// TIA Portal project "#08-法格800T(增加润滑参数设置与监控）" (V17)

(* hardware
DEVICE "S7-1200 station_1"  S7-1200 Station
   slot 0: "Rack_0"  S7-1200 Rack  Rack  V1.0
   slot 1: "PLC_1"  CPU 1215C DC/DC/DC  6ES7 215-1AG40-0XB0  V4.5
   slot 2: "DI 16x24VDC_1"  6ES7 221-1BH32-0XB0  V2.0
   slot 3: "DI 16x24VDC_2"  6ES7 221-1BH32-0XB0  V2.0
   slot 4: "DI 16x24VDC_3"  6ES7 221-1BH32-0XB0  V2.0
   slot 5: "DQ 16x24VDC_1"  SM 1222 DQ16 x 24VDC  6ES7 222-1BH32-0XB0  V2.0
   slot 101: "CM 1243-5"  CM 1243-5  6GK7 243-5DX30-0XE0  V1.3
DEVICE "ET 200SP station_1"  ET 200SP-Station
   slot 0: "机架_0"  Rack  6ES5 710-8MAx1
   slot 0: "IO device_1"  IM 155-6 PN ST  6ES7 155-6AU01-0BN0  V4.2
   slot 1: "DI 16x24VDC ST_1"  DI 16x24VDC ST  6ES7 131-6BH01-0BA0  V0.0
      slot 1: "DI 16x24VDC ST_1"  DI 16x24VDC ST
   slot 2: "DI 16x24VDC ST_6"  DI 16x24VDC ST  6ES7 131-6BH01-0BA0  V0.0
      slot 1: "DI 16x24VDC ST_6"  DI 16x24VDC ST
   slot 3: "DI 16x24VDC ST_5"  DI 16x24VDC ST  6ES7 131-6BH01-0BA0  V0.0
      slot 1: "DI 16x24VDC ST_5"  DI 16x24VDC ST
   slot 4: "DI 16x24VDC ST_4"  DI 16x24VDC ST  6ES7 131-6BH01-0BA0  V0.0
      slot 1: "DI 16x24VDC ST_4"  DI 16x24VDC ST
   slot 5: "DI 16x24VDC ST_3"  DI 16x24VDC ST  6ES7 131-6BH01-0BA0  V0.0
      slot 1: "DI 16x24VDC ST_3"  DI 16x24VDC ST
   slot 6: "DI 16x24VDC ST_2"  DI 16x24VDC ST  6ES7 131-6BH01-0BA0  V0.0
      slot 1: "DI 16x24VDC ST_2"  DI 16x24VDC ST
   slot 7: "DI 16x24VDC ST_7"  DI 16x24VDC ST  6ES7 131-6BH01-0BA0  V0.0
      slot 1: "DI 16x24VDC ST_7"  DI 16x24VDC ST
   slot 8: "DI 16x24VDC ST_9"  DI 16x24VDC ST  6ES7 131-6BH01-0BA0  V0.0
      slot 1: "DI 16x24VDC ST_9"  DI 16x24VDC ST
   slot 9: "DI 16x24VDC ST_8"  DI 16x24VDC ST  6ES7 131-6BH01-0BA0  V0.0
      slot 1: "DI 16x24VDC ST_8"  DI 16x24VDC ST
   slot 10: "DQ 16x24VDC/0.5A ST_2"  DQ 16x24VDC/0.5A ST  6ES7 132-6BH01-0BA0  V0.0
      slot 1: "DQ 16x24VDC/0.5A ST_2"  DQ 16x24VDC/0.5A ST
   slot 11: "DQ 16x24VDC/0.5A ST_1"  DQ 16x24VDC/0.5A ST  6ES7 132-6BH01-0BA0  V0.0
      slot 1: "DQ 16x24VDC/0.5A ST_1"  DQ 16x24VDC/0.5A ST
   slot 12: "服务器模块_1"  Server module  6ES7 193-6PA00-0AA0  V1.1
      slot 1: "服务器模块_1"  Server module
   slot 127: "BA 2xRJ45"  BA 2xRJ45  6ES7 193-6AR00-0AA0  V0.0
      slot 1: "Port_1"  X1 P1 R  6ES7 193-6AR00-0AA0  V0.0
      slot 2: "Port_2"  X1 P2 R  6ES7 193-6AR00-0AA0  V0.0
DEVICE "HMI_1"  TP900 Comfort
   slot 0: "HMI_1"  TP900 Comfort  6AV2 124-0JC01-0AX0  15.1.0.0
   slot 1: "HMI_RT_1"  TP900 Comfort  6AV2 124-0JC01-0AX0  15.1.0.0
   slot 5: "HMI_1.IE_CP_1"  PROFINET Interface  15.0.1.0
      slot 1: "PROFINET Interface_1"  PROFINET Interface
         slot 1: "Port_1"  Port
         slot 2: "Port_2"  Port
   slot 7: "HMI_1.MPI/DP_CP_1"  MPI/DP Interface  15.0.1.0
DEVICE "GSD device_2"  GSD.Device
   slot 0: "机架_0"  Rail
   slot 0: "横梁站"  P+F  Encoder  4.0
DEVICE "GSD device_1"  GSD.Device
   slot 0: "机架_0"  Rail
   slot 0: "滑块站"  P+F  Encoder  4.0
DEVICE "GSD device_3"  GSD.Device
   slot 0: "机架_0"  Rail
   slot 0: "气垫编码器"  P+F  Encoder  4.0
*)

// ===== PLC "PLC_1"  CPU 1215C DC/DC/DC =====

VAR_GLOBAL   // PLC tag table "默认变量表"
   "Tag_47(1)" AT %I6.1 : Bool;
   "Tag_48(1)" AT %I6.2 : Bool;
   "Tag_49(1)" AT %I6.3 : Bool;
   "Tag_50(1)" AT %I6.4 : Bool;
   "Tag_51(1)" AT %I6.5 : Bool;
   "Tag_52(1)" AT %I6.6 : Bool;
   "Tag_53(1)" AT %I6.7 : Bool;
   "Tag_54(1)" AT %I7.0 : Bool;
   "Tag_55(1)" AT %I7.1 : Bool;
   "Tag_56(1)" AT %I7.2 : Bool;
   "Tag_57(1)" AT %I7.3 : Bool;
   "Tag_58(1)" AT %I7.4 : Bool;
   "Tag_59" AT %I7.5 : Bool;
   "Tag_60" AT %I7.6 : Bool;
   "Tag_61(1)" AT %I7.7 : Bool;
   "左栅栏落下来检测" AT %Q13.1 : Bool;
   "备用(16)" AT %Q13.2 : Bool;
   "双阀控制1" AT %Q13.3 : Bool;
   "Tag_155" AT %Q13.4 : Bool;
   "双阀控制2" AT %Q13.5 : Bool;
   "Tag_157" AT %Q13.6 : Bool;
   "Tag_158" AT %Q13.7 : Bool;
   "过滤器堵塞" AT %M5.0 : Bool;
   "润滑油压正常" AT %M5.1 : Bool;
   "滑块调整允许" AT %M5.2 : Bool;
   "急停故障" AT %M6.0 : Bool;
   "液压保护故障" AT %M6.1 : Bool;
   "气压故障" AT %M6.2 : Bool;
   "设备故障" AT %M6.3 : Bool;
   "滑块调整允许(1)" AT %M6.4 : Bool;
   "滑块调整允许2(1)" AT %M6.5 : Bool;
   "气垫调整允许" AT %M6.6 : Bool;
   "工作台移动允许" AT %M7.0 : Bool;
   "工作台落到位" AT %M7.1 : Bool;
   "润滑油泵启动OK" AT %M5.5 : Bool;
   "10度" AT %M200.0 : Bool;
   "20度" AT %M200.1 : Bool;
   "30度" AT %M200.2 : Bool;
   "40度" AT %M200.3 : Bool;
   "50" AT %M200.4 : Bool;
   "60" AT %M200.5 : Bool;
   "70" AT %M200.6 : Bool;
   "80" AT %M200.7 : Bool;
   "90" AT %M201.0 : Bool;
   "100" AT %M201.1 : Bool;
   "110" AT %M201.2 : Bool;
   "120" AT %M201.3 : Bool;
   "130" AT %M201.4 : Bool;
   "140" AT %M201.5 : Bool;
   "150" AT %M201.6 : Bool;
   "160" AT %M201.7 : Bool;
   "170" AT %M202.0 : Bool;
   "180" AT %M202.1 : Bool;
   "190" AT %M202.2 : Bool;
   "200" AT %M202.3 : Bool;
   "210" AT %M202.4 : Bool;
   "220" AT %M202.5 : Bool;
   "230" AT %M202.6 : Bool;
   "240" AT %M202.7 : Bool;
   "250" AT %M203.0 : Bool;
   "260" AT %M203.1 : Bool;
   "270" AT %M203.2 : Bool;
   "280" AT %M203.3 : Bool;
   "290" AT %M203.4 : Bool;
   "300" AT %M203.5 : Bool;
   "310" AT %M203.6 : Bool;
   "320" AT %M203.7 : Bool;
   "330" AT %M204.0 : Bool;
   "340" AT %M204.1 : Bool;
   "350" AT %M204.2 : Bool;
   "360" AT %M204.3 : Bool;
   "上死点" AT %M204.4 : Bool;
   "制动监控" AT %M204.5 : Bool;
   "下死点" AT %M204.6 : Bool;
   "单次返回" AT %M204.7 : Bool;
   "光电保护位置" AT %M205.0 : Bool;
   "横梁编码器" AT %ID68 : DWord;
   "急停故障(1)" AT %M10.0 : Bool;
   "行程允许" AT %M14.0 : Bool;
   "寸动允许" AT %M14.1 : Bool;
   "寸动开始" AT %M14.2 : Bool;
   "单次允许" AT %M14.3 : Bool;
   "单次开始" AT %M14.4 : Bool;
   "双手按钮开点" AT %M14.5 : Bool;
   "双手按钮闭点" AT %M14.6 : Bool;
   "编码器闭点监控" AT %M14.7 : Bool;
   "编码器开点监控" AT %M15.0 : Bool;
   "编码器故障" AT %M15.1 : Bool;
   "工作台-夹紧OK" AT %M15.2 : Bool;
   "工作台放松OK" AT %M15.3 : Bool;
   "润滑故障" AT %M15.4 : Bool;
   "滑块软限位上" AT %M15.5 : Bool;
   "滑块软限位下" AT %M15.6 : Bool;
   "滑块调整自动向上" AT %M16.0 : Bool;
   "滑块调整自动向下" AT %M16.1 : Bool;
   "滑块调整自动选择" AT %M16.2 : Bool;
   "滑块手动调整" AT %M16.3 : Bool;
   "ECamdata _DB_D{10}滑块设定高度" AT %MD150 : Real;
   "备用(27)" AT %I21.4 : Bool;
   "备用(7)" AT %I21.3 : Bool;
   "润滑过滤检测" AT %I21.2 : Bool;
   "润滑油位检测" AT %I21.1 : Bool;
   "润滑故障复位" AT %I21.0 : Bool;
   "气垫手动润滑" AT %I20.7 : Bool;
   "平衡缸手动润滑" AT %I20.6 : Bool;   // OK
   "润滑启动按钮(1)" AT %I20.5 : Bool;   // OK
   "润滑停止按钮" AT %I20.4 : Bool;   // OK
   "备用(6)" AT %I20.3 : Bool;
   "气垫上调整(1)" AT %I20.2 : Bool;
   "滑块夹紧压力检测" AT %I20.1 : Bool;
   "后右夹紧器检测" AT %I20.0 : Bool;
   "备用(28)" AT %I21.5 : Bool;
   "后中夹紧器检测" AT %I19.7 : Bool;
   "前左夹紧器检测" AT %I19.5 : Bool;
   "前中夹紧器检测" AT %I19.4 : Bool;
   "前右夹紧器检测" AT %I19.3 : Bool;
   "气垫下降调整" AT %I19.2 : Bool;
   "滑块松开压力检测" AT %I19.1 : Bool;
   "150/AR液压保护压力" AT %I19.0 : Bool;
   "90/AR液压保护压力" AT %I18.7 : Bool;
   "100液压保护压力" AT %I18.6 : Bool;
   "135/AR液压保护压力" AT %I18.5 : Bool;
   "100/AR液压保护压力" AT %I18.4 : Bool;
   "液压保护选择开关1位" AT %I18.3 : Bool;   // OK
   "液压保护选择开关0位" AT %I18.2 : Bool;   // OK
   "工作台落下右边后检测" AT %I18.1 : Bool;
   "后左夹紧器检测" AT %I19.6 : Bool;
   "工作台落下左后检测" AT %I18.0 : Bool;
   "备用(8)" AT %I21.6 : Bool;
   "备用(10)" AT %I22.0 : Bool;
   "寸动" AT %I25.4 : Bool;   // OK
   "反转" AT %I25.3 : Bool;   // OK
   "右前双手选择" AT %I25.2 : Bool;   // OK
   "右后双手选择(1)" AT %I25.1 : Bool;   // OK
   "左后双手选择" AT %I25.0 : Bool;   // OK
   "单人/双人选择" AT %I24.7 : Bool;
   "离制油箱油温检测" AT %I24.6 : Bool;
   "左前双手选择" AT %I24.5 : Bool;   // OK
   "备用(15)" AT %I24.4 : Bool;
   "离合冷却过滤器检测" AT %I24.3 : Bool;
   "离制油箱油位检测" AT %I24.2 : Bool;
   "备用(14)" AT %I24.1 : Bool;
   "离制压力检测" AT %I24.0 : Bool;
   "备用(9)" AT %I21.7 : Bool;
   "离制过滤器检测" AT %I23.7 : Bool;
   "栅栏门向上？(1)" AT %I23.5 : Bool;
   "栅栏门向上？" AT %I23.4 : Bool;
   "备用(13)" AT %I23.3 : Bool;
   "备用(12)" AT %I23.2 : Bool;
   "前安全栓" AT %I23.1 : Bool;   // OK
   "后安全栓" AT %I23.0 : Bool;   // OK
   "左后急停按钮" AT %I22.7 : Bool;   // OK
   "右后急停按钮" AT %I22.6 : Bool;   // OK
   "左前急停按钮" AT %I22.5 : Bool;   // OK
   "右前急停按钮" AT %I22.4 : Bool;   // OK
   "备用(11)" AT %I22.3 : Bool;
   "气垫分油器检测" AT %I22.2 : Bool;
   "滑块分油器检测" AT %I22.1 : Bool;
   "备用(29)" AT %I23.6 : Bool;
   "工作台落下右前检测" AT %I17.7 : Bool;
   "工作台落下左前检测" AT %I17.6 : Bool;
   "工作台顶起右后检测" AT %I17.5 : Bool;
   "气垫冷却电机温度监测(启动）" AT %I13.3 : Bool;
   "气垫冷却电机温度监测(停止）" AT %I13.2 : Bool;
   "气垫冷却电机过热" AT %I13.1 : Bool;
   "主电机启动(1)" AT %I13.0 : Bool;   // OK
   "主电机停止" AT %I12.7 : Bool;   // OK
   "备用(26)" AT %I12.6 : Bool;
   "备用(25)" AT %I12.5 : Bool;
   "备用(24)" AT %I12.4 : Bool;
   "IMCO应力机" AT %I12.3 : Bool;
   "滑块调整传动检测？(1)" AT %I12.2 : Bool;
   "气垫压力检测" AT %I12.1 : Bool;
   "气垫排气" AT %I12.0 : Bool;
   "气垫油位检测" AT %I11.7 : Bool;
   "上极限" AT %I13.4 : Bool;
   "气垫左落下到位" AT %I11.6 : Bool;
   "备用" AT %I11.4 : Bool;
   "气垫调整下极限" AT %I11.3 : Bool;
   "气垫调整上极限" AT %I11.2 : Bool;
   "右气垫选择" AT %I11.1 : Bool;
   "气垫排气(1)" AT %I11.0 : Bool;
   "气垫选择开关" AT %I10.7 : Bool;
   "滑块调整传动检测？" AT %I10.6 : Bool;
   "平衡缸气压检测" AT %I10.5 : Bool;
   "滑块调整下极限" AT %I10.4 : Bool;
   "滑块调整上极限" AT %I10.3 : Bool;
   "滑块调整向下" AT %I10.2 : Bool;   // OK
   "滑块调整向上" AT %I10.1 : Bool;   // OK
   "滑块调整选择开关" AT %I10.0 : Bool;   // OK
   "备用(1)" AT %I11.5 : Bool;
   "下极限" AT %I13.5 : Bool;
   "出到位检测（小车）" AT %I13.6 : Bool;
   "移动工作台变速（小车）" AT %I13.7 : Bool;
   "工作台顶起左后检测" AT %I17.4 : Bool;
   "工作台顶起右前检测" AT %I17.3 : Bool;
   "工作台顶起左前检测" AT %I17.2 : Bool;
   "气垫上调整" AT %I17.1 : Bool;
   "外导轨切换检测？(1)" AT %I17.0 : Bool;
   "外导轨切换检测？" AT %I16.7 : Bool;
   "工作台右后落到位" AT %I16.6 : Bool;
   "工作台左后落到为" AT %I16.5 : Bool;
   "工作台右前落到为" AT %I16.4 : Bool;
   "工作台左前落到为" AT %I16.3 : Bool;
   "工作台开进到位" AT %I16.2 : Bool;
   "工作台右后顶起到位" AT %I16.1 : Bool;
   "工作台左后顶起到位" AT %I16.0 : Bool;
   "工作台右前顶起到位" AT %I15.7 : Bool;
   "工作台左前顶起到位" AT %I15.6 : Bool;
   "按钮站插入" AT %I15.5 : Bool;
   "左工作台按钮拔出" AT %I15.4 : Bool;
   "工作台顶起压力" AT %I15.3 : Bool;
   "备用(2)" AT %I15.2 : Bool;
   "循环停止" AT %I15.1 : Bool;   // OK
   "工作台开进" AT %I15.0 : Bool;   // OK
   "工作台开出" AT %I14.7 : Bool;   // OK
   "模具更换自动/手动选择" AT %I14.6 : Bool;   // OK
   "调整开关" AT %I14.5 : Bool;   // OK
   "工作台放松顶起" AT %I14.4 : Bool;   // OK
   "工作台落下夹紧(1)" AT %I14.3 : Bool;   // OK
   "备用(4)" AT %I14.2 : Bool;
   "备用(3)" AT %I14.1 : Bool;
   "工作台停止" AT %I14.0 : Bool;
   "单次" AT %I25.5 : Bool;   // OK
   "连续" AT %I25.6 : Bool;   // OK
   "备用(17)" AT %I25.7 : Bool;
   "左前双手 使用" AT %I26.0 : Bool;
   "模具移出指示" AT %Q12.2 : Bool;
   "飞轮停止指示灯" AT %Q12.1 : Bool;
   "主电机启动指示" AT %Q12.0 : Bool;
   "自动化气压" AT %Q11.7 : Bool;
   "气垫间歇润滑阀" AT %Q11.6 : Bool;
   "备用(35)" AT %Q11.5 : Bool;
   "工作台顶起" AT %Q11.4 : Bool;
   "工作台落下夹紧(2)" AT %Q11.3 : Bool;
   "工作台落下夹紧" AT %Q11.2 : Bool;
   "工作台放松顶起(1)" AT %Q11.1 : Bool;
   "液压保护负荷荷 阀-3#" AT %Q11.0 : Bool;
   "液压保护泵启动（卸载）阀-2#" AT %Q10.7 : Bool;
   "气动泵气源阀-1#" AT %Q10.6 : Bool;
   "模具装入指示" AT %Q12.3 : Bool;
   "右气垫气排阀" AT %Q10.5 : Bool;
   "气垫排气阀" AT %Q10.3 : Bool;
   "气垫进气阀" AT %Q10.2 : Bool;
   "平衡缸排气阀" AT %Q10.1 : Bool;
   "平衡缸进气阀" AT %Q10.0 : Bool;
   "Tag_109" AT %QW572 : Int;
   "Tag_108" AT %QW570 : Int;
   "Tag_20" AT %ID97 : DWord;
   "气垫编码器" AT %ID100 : DWord;
   "气垫编码器1" AT %ID96 : DWord;
   "气垫模拟量1" AT %IW82 : Int;
   "平衡器压力模拟量" AT %IW80 : Int;
   "气垫模拟量2" AT %IW84 : Int;
   "滑块编码器" AT %ID72 : DInt;
   "右气垫进气阀" AT %Q10.4 : Bool;
   "润滑电机工作指示" AT %Q12.4 : Bool;
   "液压保护正常指示" AT %Q12.5 : Bool;
   "液压保护卸荷指示" AT %Q12.6 : Bool;
   "Tag_22" AT %Q20.2 : Bool;
   "Tag_2" AT %Q20.6 : Bool;
   "主电机中间继电器" AT %Q3.7 : Bool;
   "主电机风扇运行" AT %Q3.6 : Bool;
   "滑块向下调整" AT %Q3.5 : Bool;
   "滑块向上调整" AT %Q3.4 : Bool;
   "单次连续继电器" AT %Q3.3 : Bool;
   "离合器油泵电机" AT %Q3.2 : Bool;
   "压机急停2" AT %Q3.1 : Bool;
   "压机急停1" AT %Q3.0 : Bool;
   "安全正常(1)" AT %Q2.7 : Bool;
   "润滑电机" AT %Q2.6 : Bool;
   "工作台变速" AT %Q2.5 : Bool;
   "工作骀电机反转" AT %Q2.4 : Bool;
   "工作台电机正转(1)" AT %Q2.3 : Bool;
   "变频器使能" AT %Q2.2 : Bool;
   "系统泵开始" AT %Q2.1 : Bool;
   "主电机正转运行" AT %Q2.0 : Bool;
   "主电机反转" AT %Q1.1 : Bool;
   "速度控制" AT %Q1.0 : Bool;
   "主电机运行" AT %Q0.7 : Bool;
   "气垫降" AT %Q0.6 : Bool;
   "气垫升" AT %Q0.5 : Bool;
   "单人操作" AT %Q0.4 : Bool;
   "飞轮制动阀" AT %Q0.3 : Bool;
   "平衡器间歇润滑阀" AT %Q0.2 : Bool;
   "气垫降(1)" AT %Q0.1 : Bool;
   "气垫升(1)" AT %Q0.0 : Bool;
   "变频器上电" AT %Q12.7 : Bool;
   "平衡缸压力模拟量(1)" AT %ID85 : DWord;
   "Tag_18(2)" AT %M1101.5 : Bool;
   "平衡缸压力模拟量" AT %ID84 : DWord;
   "备用(22)" AT %I5.6 : Bool;
   "Tag_15" AT %I1.4 : Bool;
   "Tag_14" AT %I1.3 : Bool;
   "Tag_13" AT %I1.2 : Bool;
   "Tag_12" AT %I1.1 : Bool;
   "Tag_11" AT %I1.0 : Bool;
   "Tag_10" AT %I0.7 : Bool;
   "Tag_9" AT %I0.6 : Bool;
   "Tag_8" AT %I0.5 : Bool;
   "1" AT %I0.4 : Bool;
   "Tag_6(1)" AT %I0.3 : Bool;
   "Tag_5(1)" AT %I0.2 : Bool;
   "Tag_4(1)" AT %I0.1 : Bool;
   "Tag_3" AT %I0.0 : Bool;
   "Tag_16" AT %I1.5 : Bool;
   "Tag_43" AT %I27.7 : Bool;
   "后双手1" AT %I27.5 : Bool;
   "前双手2" AT %I27.4 : Bool;
   "前双手1" AT %I27.3 : Bool;
   "Tag_38" AT %I27.2 : Bool;
   "Tag_37" AT %I27.1 : Bool;
   "Tag_36" AT %I27.0 : Bool;
   "右后双手 短接" AT %I26.7 : Bool;   // OK
   "右后双手 使用" AT %I26.6 : Bool;
   "备用(33)" AT %I26.5 : Bool;
   "双手后2" AT %I26.4 : Bool;
   "双手后1" AT %I26.3 : Bool;
   "双手前" AT %I26.2 : Bool;
   "左前双手 短接" AT %I26.1 : Bool;   // OK
   "后双手2" AT %I27.6 : Bool;
   "Tag_17" AT %I1.6 : Bool;
   "Tag_18(1)" AT %I1.7 : Bool;
   "电源接通" AT %I2.0 : Bool;
   "备用(21)" AT %I5.5 : Bool;
   "备用(20)" AT %I5.4 : Bool;
   "气垫调整空开(1)" AT %I5.3 : Bool;
   "离合器准确检测" AT %I5.2 : Bool;
   "横梁1分油器检测" AT %I5.1 : Bool;
   "平衡器分油器检测" AT %I5.0 : Bool;
   "飞轮制动松开检测" AT %I4.7 : Bool;
   "备用(18)" AT %I4.6 : Bool;
   "左后双手未使用" AT %I4.5 : Bool;
   "左后双手使用" AT %I4.4 : Bool;   // OK
   "右前双手未使用" AT %I4.3 : Bool;
   "右前双手使用" AT %I4.2 : Bool;   // OK
   "主电机温度检测(1)" AT %I4.1 : Bool;
   "主电机风扇流量检测(1)" AT %I4.0 : Bool;
   "离合器运行" AT %I3.7 : Bool;
   "离合器油泵空开" AT %I3.6 : Bool;
   "离制双阀反馈2" AT %I3.5 : Bool;
   "离制双阀反馈1" AT %I3.4 : Bool;
   "总复位" AT %I3.3 : Bool;
   "安全正常" AT %I3.2 : Bool;
   "栅栏门未来关闭" AT %I3.1 : Bool;
   "润滑电机空开" AT %I3.0 : Bool;
   "液压保护系统空开" AT %I2.7 : Bool;
   "开工作台变频器正常" AT %I2.6 : Bool;
   "主电机零速" AT %I2.5 : Bool;
   "主电机调速装置正常" AT %I2.4 : Bool;
   "主电机风扇空开" AT %I2.3 : Bool;
   "气垫调整空开" AT %I2.2 : Bool;
   "滑块调整电机空开" AT %I2.1 : Bool;
   "备用(23)" AT %I5.7 : Bool;
   "Tag_19(1)" AT %M1101.6 : Bool;
   "Tag_1" AT %M290.1 : Bool;
   "工作台落到位(1)" AT %M300.1 : Bool;
   "工作台放松顶起到位" AT %M300.2 : Bool;
   "工作台移动条件" AT %M210.3 : Bool;
   "液压保护正常" AT %M207.6 : Bool;
   "润滑正常" AT %M1000.4 : Bool;
   "滑块调整条件" AT %M208.2 : Bool;
   "上调整设定值" AT %M302.2 : Bool;
   "下调整设定值_1" AT %M302.3 : Bool;
   "滑块调整软上极限(2)" AT %M302.0 : Bool;
   "滑块调整软下极限(3)" AT %M302.1 : Bool;
   "滑块调整手动/自动" AT %M301.5 : Bool;
   "滑块调整手动" AT %M301.6 : Bool;
   "滑块调整自动" AT %M301.7 : Bool;
   "平衡器排气(1)" AT %M300.5 : Bool;
   "平衡器进气" AT %M300.4 : Bool;
   "Tag_18" AT %M300.3 : Bool;
   "润滑异常" AT %M1000.6 : Bool;
   "分计时器" AT %M4000.0 : Bool;
   "Tag_24" AT %M6000.0 : Bool;
   "Tag_62" AT %M1000.0 : Bool;
   "Tag_63" AT %M1000.1 : Bool;
   "Tag_64" AT %M1000.2 : Bool;
   "Tag_65" AT %M1000.3 : Bool;
   "Tag_46" AT %M5000.0 : Bool;
   "气垫间歇时间" AT %M1001.3 : Bool;
   "气垫打油时间" AT %M1001.4 : Bool;
   "Tag_14(1)" AT %M1101.1 : Bool;
   "Tag_75" AT %M209.1 : Bool;
   "Tag_4" AT %M1222.0 : Bool;
   "主分油器故障" AT %M1222.1 : Bool;
   "Tag_6" AT %M1222.2 : Bool;
   "滑块分油器故障" AT %M1222.3 : Bool;
   "Tag_7" AT %M1222.4 : Bool;
   "平衡缸润滑故障" AT %M1222.5 : Bool;
   "滑块向下调整条件" AT %M220.1 : Bool;
   "滑块向上调整条件" AT %M220.0 : Bool;
   "滑块调整电机空开(1)" AT %M220.2 : Bool;
   "右栅栏落下检测" AT %Q13.0 : Bool;
   "压机急停故障2" AT %M333.1 : Bool;
   "单次条件1" AT %M3500.2 : Bool;
   "单次条件2" AT %M3500.3 : Bool;
   "单次条件" AT %M3500.4 : Bool;
   "行程条件" AT %M3500.5 : Bool;
   "寸动条件" AT %M3500.6 : Bool;
   "寸动条件1" AT %M3500.7 : Bool;
   "Tag_5" AT %M1001.5 : Bool;
   "手动润滑延时" AT %M30.5 : Bool;
   "Tag_21" AT %M40.0 : Bool;
   "Tag_23" AT %M40.1 : Bool;
   "Tag_25" AT %M40.2 : Bool;
   "离制压力正常" AT %M3501.0 : Bool;
   "气垫编码器(1)" AT %ID78 : DWord;
   "选择关闭" AT %M330.0 : Bool;
   "气垫调整手动" AT %M330.2 : Bool;
   "气垫调整自动" AT %M330.3 : Bool;
   "气垫软上限位" AT %M330.5 : Bool;
   "气垫自动上调条件" AT %M330.6 : Bool;
   "气垫自动下调条件" AT %M330.7 : Bool;
   "Tag_26" AT %IB78 : Byte;
   "Tag_27" AT %M700.7 : Bool;
   "Tag_28" AT %M700.6 : Bool;
   "System_Byte" AT %MB1 : Byte;
   "FirstScan" AT %M1.0 : Bool;
   "DiagStatusUpdate" AT %M1.1 : Bool;
   "AlwaysTRUE" AT %M1.2 : Bool;
   "AlwaysFALSE" AT %M1.3 : Bool;
   "Clock_Byte" AT %MB0 : Byte;
   "Clock_10Hz" AT %M0.0 : Bool;
   "Clock_5Hz" AT %M0.1 : Bool;
   "Clock_2.5Hz" AT %M0.2 : Bool;
   "Clock_2Hz" AT %M0.3 : Bool;
   "Clock_1.25Hz" AT %M0.4 : Bool;
   "Clock_1Hz" AT %M0.5 : Bool;
   "Clock_0.625Hz" AT %M0.6 : Bool;
   "Clock_0.5Hz" AT %M0.7 : Bool;
END_VAR

VAR_GLOBAL   // PLC tag table "变量表"
   "气垫压力模拟量" AT %ID81 : DWord;
   "报警1" AT %M3000.0 : Bool;
   "报警2" AT %M3000.1 : Bool;
   "报警3" AT %M3000.2 : Bool;
   "报警4" AT %M3000.3 : Bool;
   "报警5" AT %M3000.4 : Bool;
   "报警6" AT %M3000.5 : Bool;
   "报警7" AT %M3000.6 : Bool;
   "报警8" AT %M3000.7 : Bool;
   "报警9" AT %M3001.0 : Bool;
   "报警10" AT %M3001.1 : Bool;
   "报警11" AT %M3001.2 : Bool;
   "报警12" AT %M3001.3 : Bool;
   "报警13" AT %M3001.4 : Bool;
   "报警14" AT %M3001.5 : Bool;
   "报警15" AT %M3001.6 : Bool;
   "报警16" AT %M3001.7 : Bool;
   "PLC报警变量组1" AT %MW3000 : Int;
   "PLC报警变量组2" AT %MW3002 : Int;
   "PLC报警变量组3" AT %MW3004 : Int;
   "报警17" AT %M3002.0 : Bool;
   "报警18" AT %M3002.1 : Bool;
   "报警19" AT %M3002.2 : Bool;
   "报警20" AT %M3002.3 : Bool;
   "报警21" AT %M3002.4 : Bool;
   "报警22" AT %M3002.5 : Bool;
   "报警23" AT %M3002.6 : Bool;
   "报警24" AT %M3002.7 : Bool;
   "报警25" AT %M3003.0 : Bool;
   "报警26" AT %M3003.1 : Bool;
   "报警27" AT %M3003.2 : Bool;
   "报警28" AT %M3003.3 : Bool;
   "报警29" AT %M3003.4 : Bool;
   "报警30" AT %M3003.5 : Bool;
   "报警31" AT %M3003.6 : Bool;
   "报警32" AT %M3003.7 : Bool;
   "报警33" AT %M3004.0 : Bool;
   "报警34" AT %M3004.1 : Bool;
   "报警35" AT %M3004.2 : Bool;
   "报警36" AT %M3004.3 : Bool;
   "报警37" AT %M3004.4 : Bool;
   "报警38" AT %M3004.5 : Bool;
   "报警39" AT %M3004.6 : Bool;
   "报警40" AT %M3004.7 : Bool;
   "报警41" AT %M3005.0 : Bool;
   "报警42" AT %M3005.1 : Bool;
   "报警43" AT %M3005.2 : Bool;
   "报警44" AT %M3005.3 : Bool;
   "报警45" AT %M3005.4 : Bool;
   "报警46" AT %M3005.5 : Bool;
   "报警47" AT %M3005.6 : Bool;
   "报警48" AT %M3005.7 : Bool;
   "Tag_1(1)" AT %M100.0 : Bool;
   "Tag_7(2)" AT %M100.1 : Bool;
   "异常报警1" AT %M1008.3 : Bool;
   "异常报警2" AT %M1008.4 : Bool;
   "液压保护开启条件" AT %M205.1 : Bool;
   "液压保护卸载" AT %M207.7 : Bool;
   "液压保护故障(1)" AT %M208.0 : Bool;
   "电动泵启动" AT %M205.2 : Bool;
   "液压保护上升沿" AT %M207.5 : Bool;
   "行程选择" AT %M207.3 : Bool;
   "急停故障(2)" AT %M300.0 : Bool;
   "压机故障2" AT %M388.1 : Bool;
   "Tag_19" AT %M301.0 : Bool;
   "Tag_77" AT %M388.2 : Bool;
   "主电机启动条件" AT %M1001.0 : Bool;
   "变频断电延时" AT %M1101.0 : Bool;
   "正转条件" AT %M1000.7 : Bool;
   "反转条件" AT %M1001.1 : Bool;
   "主电机启动延时" AT %M1100.4 : Bool;
   "Tag_7(1)" AT %M1100.2 : Bool;
   "Tag_11(1)" AT %M1100.6 : Bool;
   "Tag_10(1)" AT %M1100.5 : Bool;
   "主电机启动脉冲" AT %M1100.7 : Bool;
   "主电机调速" AT %M208.3 : Bool;
   "主电机故障报警" AT %M1001.2 : Bool;
   "计数开始" AT %M30.0 : Bool;
   "计数清零" AT %M30.1 : Bool;
   "产量到达" AT %M30.2 : Bool;
END_VAR

VAR_GLOBAL CONSTANT   // PLC tag table "变量表"
   "无(1)" : Pip := 65535;
   "自动更新(1)" : Pip := 0;
   "PIP 1(1)" : Pip := 1;
   "PIP 2(1)" : Pip := 2;
   "PIP 3(1)" : Pip := 3;
   "PIP 4(1)" : Pip := 4;
   "PIP OB 伺服(1)" : Pip := 32768;
   "Local~MC(1)" : Hw_SubModule := 51;
   "Local~Common(1)" : Hw_SubModule := 50;
   "Local~Device(1)" : Hw_Device := 32;
   "Local~Configuration(1)" : Hw_SubModule := 33;
   "Local~Exec(1)" : Hw_SubModule := 52;
   "Local(1)" : Hw_SubModule := 49;
   "Local~PROFINET_接口_1(1)" : Hw_Interface := 64;
   "Local~PROFINET_接口_1~端口_1(1)" : Hw_Interface := 65;
   "Local~HSC_1(1)" : Hw_Hsc := 257;
   "Local~HSC_2(1)" : Hw_Hsc := 258;
   "Local~HSC_3(1)" : Hw_Hsc := 259;
   "Local~HSC_4(1)" : Hw_Hsc := 260;
   "Local~HSC_5(1)" : Hw_Hsc := 261;
   "Local~HSC_6(1)" : Hw_Hsc := 262;
   "Local~AI_2_1" : Hw_SubModule := 263;
   "Local~DI_14_DQ_10_1(1)" : Hw_SubModule := 264;
   "Local~Pulse_1(1)" : Hw_Pwm := 265;
   "Local~Pulse_2(1)" : Hw_Pwm := 266;
   "Local~Pulse_3(1)" : Hw_Pwm := 267;
   "Local~Pulse_4(1)" : Hw_Pwm := 268;
   "Local~CM_1243-5~DP_接口(1)" : Hw_Interface := 269;
   "Local~CM_1243-5(1)" : Hw_SubModule := 271;
   "Local~PROFINET_IO-System(1)" : Hw_IoSystem := 272;
   "Local~DP-Mastersystem(1)" : Hw_IoSystem := 273;
   "Local~DI_16x24VDC_1(1)" : Hw_SubModule := 291;
   "Local~DI_16x24VDC_2(1)" : Hw_SubModule := 292;
   "Local~DQ_16x24VDC_1(1)" : Hw_SubModule := 293;
   "立柱右前操作站~Head" : Hw_Interface := 288;
   "立柱右前操作站~DPSlave" : Hw_DpSlave := 286;
   "立柱右前操作站~DI_32x24VDC_1" : Hw_SubModule := 289;
   "立柱右前操作站~AI_8x12BIT_1" : Hw_SubModule := 294;
   "立柱右前操作站~DI_32x24VDC_2" : Hw_SubModule := 295;
   "立柱右前操作站~DI_32x24VDC_3" : Hw_SubModule := 296;
   "立柱右前操作站~DI_32x24VDC_4" : Hw_SubModule := 297;
   "立柱右前操作站~DO_32x24VDC_0_5A_2" : Hw_SubModule := 299;
   "立柱右前操作站~DO_16x24VDC_0_5A_1" : Hw_SubModule := 290;
   "立柱右前操作站~DI_16x24VDC_1" : Hw_SubModule := 274;
   "横梁站~Head(1)" : Hw_Interface := 280;
   "横梁站~DPSlave(1)" : Hw_DpSlave := 278;
   "横梁站~P+F_Version_2_1_Singleturn_1(1)" : Hw_SubModule := 281;
   "OB_Main(1)" : OB_PCYCLE := 1;
   "OB_Cyclic interrupt" : OB_Cyclic := 30;
   "OB_RackStationFailure" : OB_Any := 86;
   "OB_Startup" : OB_STARTUP := 100;
   "滑块站~Head(1)" : Hw_Interface := 277;
   "滑块站~DPSlave(1)" : Hw_DpSlave := 275;
   "滑块站~32_Bit_Class_2_+_Speed_2_1" : Hw_SubModule := 282;
   "滑块站~32_Bit_Class_2_+_Speed_2_2" : Hw_SubModule := 283;
END_VAR

TYPE "用户数据类型_1"
   STRUCT
      Element_1 : Bool;
   END_STRUCT;
END_TYPE

// folder: 4.1_Line_Operation

TYPE "Operation_Mode"
   STRUCT
      Auto : Bool;
      Auto_Sim : Bool;
      APC : Bool;
      ATC : Bool;
      Man : Bool;
      Setup : Bool;
      工作模式 : UInt;
      零件表 : UInt;
   END_STRUCT;
END_TYPE

TYPE "4.1_Line_Operation"
   STRUCT
      Mode_Act : "Operation_Mode";
      Mode_Seting : "Operation_Mode";
      Recipes_Operation : "HMI_Recipe";
      HMI : Array[1..10] of "HMI_State";
   END_STRUCT;
END_TYPE

TYPE "HMI_Recipe"
   STRUCT
      Recipe : Struct
         Clear : Bool;
         Load : Bool;
         Save : Bool;
         Edit_No : Int;
         Recipe_Edit_Auth : Bool;
         Recipe_Edit_Wizard : Int;
         Load_Active : Bool;
         Save_Active : Bool;
         ii : Int;
         Load_Timer : IEC_TIMER;
         Save_Timer : IEC_TIMER;
      END_STRUCT;
      RecipeExport : Struct
         Done : Bool;
         Busy : Bool;
         Error : Bool;
         Status : Word;
      END_STRUCT;
      RecipeImport : Struct
         Done : Bool;
         Busy : Bool;
         Error : Bool;
         Status : Word;
      END_STRUCT;
   END_STRUCT;
END_TYPE

TYPE "HMI_State"
   STRUCT
      Command : Struct
         Doub_Part_Dropped_Mem : Bool;
         Part_Dropped_Mem : Bool;
         Part_Picker_Mem : Bool;
         Part_Done_Mem : Bool;
         Optim_Auth : Bool;
         Part_No_Chg_Auth : Bool;
      END_STRUCT;
      State : Struct
         Doub_Part_Dropped_Mem_1 : Bool;
         Part_Dropped_Mem_1 : Bool;
         Part_Picker_Mem_1 : Bool;
         Part_Done_Mem_1 : Bool;
      END_STRUCT;
   END_STRUCT;
END_TYPE

// folder: (top level)

DATA_BLOCK "横梁编码器 _DB"   // DB3
{ S7_Optimized_Access := 'TRUE' }
VERSION : 0.1
   VAR
      "0.0" : Struct
         "+0.0" : DWord;
         "+4.0" : DWord;
         "+8.0" : DWord;
         "+12.0" : DWord;
      END_STRUCT;
      横梁 : Int;
      滑块 : Int;
      滑块_1 : DWord;
      "+0.3" : Int;
      "+0.4" : Int;
      "+0.5" : Int;
      "+0.6" : Int;
      "+0.7" : Int;
   END_VAR
   VAR RETAIN
      "+0.8" : Int;
   END_VAR
   VAR
      "+0.9" : Int;
      "+0.10" : Int;
      "0.11" : Real;
      平衡器分油器检测 : Int;
      横梁分油器检测 : Int;
      滑块分油器检测 : Int;
      气垫分油器检测 : Int;
      "+0.15" : Int;
      "+0.16" : Int;
      "+0.17" : Int;
      "+0.18" : Int;
      "+0.19" : Int;
      "+0.20" : Int;
      "+0.21" : Int;
      "+0.22" : Int;
      "+0.23" : Int;
      "+0.24" : Int;
      "+0.25" : Int;
      "+0.26" : Int;
      "+0.27" : Int;
      "+0.28" : Int;
      "+0.29" : Int;
      "+0.30" : Int;
      平衡器打油次数 : Int;
      主分油器打油次数 : Int;
      滑块打油次数 : Int;
      气点垫打油次数 : Int;
      "+0.35" : Int;
      "+0.36" : Int;
      "+0.37" : Int;
      "+0.38" : Int;
      "+0.39" : Int;
      "+0.40" : Int;
      "+0.41" : Int;
      "+0.42" : Int;
      "+0.43" : Int;
      "+0.44" : Int;
      "+0.45" : Int;
      "+0.46" : Int;
      "+0.47" : Int;
      "+0.48" : Int;
   END_VAR
   VAR RETAIN
      AI : Array[0..10] of DInt;
      D : Array[0..10] of Real;
   END_VAR
   VAR
      AQD : Real;
      产量设定 : Int;
      D107 : Real;
   END_VAR
BEGIN
END_DATA_BLOCK

DATA_BLOCK "中间数据"   // DB6
{ S7_Optimized_Access := 'TRUE' }
VERSION : 0.1
   VAR RETAIN
      横梁润滑检测时长 : Time := T#1M;
      滑块润滑检测时长 : Time := T#1M;
      平衡器润滑检测时长 : Time := T#1M;
      横梁打油目标次数 : Int := 25;
      滑块打油目标次数 : Int := 30;
      平衡器打油目标次数 : Int := 2;
      平衡器润滑阀持续时间设定 : Time := T#5M;
      平衡器润滑阀间歇时间设定 : Time := T#100S;
   END_VAR
   VAR
      平衡器手动延时设定 : Time := T#5M;
      气垫润滑阀持续时间设定 : Time := T#5M;
      气垫润滑阀间歇时间设定 : Time := T#100S;
      气垫手动延时设定 : Time := T#5M;
      "当前打油次数-横梁" : Int;
      "当前打油次数-滑块" : Int;
      "当前打油次数-平衡器" : Int;
   END_VAR
BEGIN
END_DATA_BLOCK

DATA_BLOCK "ECamdata _DB"   // DB7
{ S7_Optimized_Access := 'TRUE' }
VERSION : 0.1
   VAR
      "0.0" : Struct
         "+0.0" : DWord;
         "+4.0" : DWord;
         "+8.0" : DWord;
         "+12.0" : DWord;
      END_STRUCT;
      横梁编码器 : Int;
      滑块编码器 : DInt;
      气垫编码器1 : DWord;
      气垫编码器2 : DWord;
      平衡器压力显示_3 : Int;
      电子凸轮编码器 : Int;
      "+0.5" : Real;
      电子凸轮编码器显示 : Int;
      "+0.7" : DInt;
      "+0.8" : Int;
      "+0.9" : Real;
      "+0.10_1" : Int;
      "+0.11" : Int;
      "+0.12" : Int;
      "+0.13" : Int;
      "+0.10" : Int;
      平衡器分油器检测 : Int;
      横梁分油器检测 : Int;
      滑块分油器检测 : Int;
      气垫分油器检测 : Int;
      "+0.15" : Int;
      "+0.16" : Int;
      "+0.17" : Int;
      "+0.18" : Int;
      "+0.19" : Int;
      "+0.20" : Int;
      "+0.21" : Int;
      "+0.22" : Int;
      "+0.23" : Int;
      "+0.24" : Int;
      "+0.25" : Int;
      "+0.26" : Int;
      "+0.27" : Int;
      "+0.28" : Int;
      "+0.29" : Int;
      "+0.30" : Int;
      平衡器打油次数 : Int;
      主分油器打油次数 : Int;
      滑块打油次数 : Int;
      气点垫打油次数 : Int;
      "+0.35" : Int;
      "+0.36" : Int;
      平衡器压力显示_2 : Real;
      平衡器压力显示_1 : Real;
      "+0.39" : Int;
      "+0.40" : Real;
      "+0.41" : Real;
      气垫模拟量 : Int;
      气垫模拟量_1 : Real;
      气垫模拟量_2 : Real;
      "+0.45" : DInt;
      "+0.46" : Int;
      "+0.47" : Real;
      "+0.48" : Int;
   END_VAR
   VAR RETAIN
      AI : Array[0..10] of DInt;
      D : Array[0..20] of Real;
   END_VAR
   VAR
      平衡器压力显示 : Real;
      AQD2 : Real;
      气垫模拟量显示1 : Real;
      气垫模拟量显示2 : Real;
      平衡器设置压力 : Real;
      气垫1压力设置 : Real;
      气垫2压力设置 : Real;
      D100 : Real;
      D101 : Int;
      D102 : Int;
      D103 : Real;
      D104 : Real;
      D105 : Real;
      D106 : Real;
      D107 : Int;
      D108 : Real;
      D109 : Real;
   END_VAR
   VAR RETAIN
      设置产量 : Int;
      当前产量 : Int;
      滑块位置 : Int;
   END_VAR
   VAR
      气垫位置 : Int;
   END_VAR
   VAR RETAIN
      D200 : DInt;
      D201 : Int;
   END_VAR
BEGIN
END_DATA_BLOCK

DATA_BLOCK "气垫编码器数据"   // DB28
{ S7_Optimized_Access := 'TRUE' }
VERSION : 0.1
   VAR
      编码器原始数据 : DInt;
      气垫设定值 : Int;
      "缩放比例（待测量）" : DInt := 10000;
      "高度补偿（待测量）" : Int := 200;
      缩放后值 : Int;
      气垫当前值 : Int;
      气垫高度 : Int;
      气垫设定值_1 : DInt;
      "123" : Bool;
   END_VAR
BEGIN
END_DATA_BLOCK

DATA_BLOCK "Timer"   // DB29
{ S7_Optimized_Access := 'TRUE' }
VERSION : 0.1
   VAR
      横梁润滑检测计时 : IEC_TIMER;
      滑块润滑检测计时 : IEC_TIMER;
      气垫润滑检测计时 : IEC_TIMER;
      平衡器润滑检测计时 : IEC_TIMER;
      润滑初始化计时器 : IEC_TIMER;
      气垫润滑持续计时 : IEC_TIMER;
      气垫润滑间歇计时 : IEC_TIMER;
      气垫手动延时计时 : IEC_TIMER;
      手动润滑持续计时 : IEC_TIMER;
      平衡器润滑持续计时 : IEC_TIMER;
      平衡器润滑间歇计时 : IEC_TIMER;
      平衡器手动延时计时 : IEC_TIMER;
      主电机指示灯延时 : IEC_TIMER;
   END_VAR
BEGIN
END_DATA_BLOCK

DATA_BLOCK "Counter"   // DB30
{ S7_Optimized_Access := 'TRUE' }
VERSION : 0.1
   VAR
      横梁润滑检测计数 : IEC_COUNTER;
   END_VAR
   VAR RETAIN
      滑块润滑检测计数 : IEC_COUNTER;
      气垫润滑检测计数 : IEC_COUNTER;
      平衡器润滑检测计数 : IEC_COUNTER;
   END_VAR
BEGIN
END_DATA_BLOCK

DATA_BLOCK "辅助中继"   // DB31
{ S7_Optimized_Access := 'TRUE' }
VERSION : 0.1
   VAR
      平衡器润滑 : Bool;
      气垫润滑 : Bool;
      横梁润滑故障 : Bool;
      滑块润滑故障 : Bool;
      气垫润滑故障 : Bool;
      平衡器润滑故障 : Bool;
      润滑空开异常 : Bool;
      润滑过滤异常 : Bool;
      分油器检测正常 : Bool;
      润滑初始化成功 : Bool;
      润滑初始化失败 : Bool;
      "打油计数到-横梁" : Bool;
      "打油计数到-滑块" : Bool;
      "打油计数到-平衡器" : Bool;
   END_VAR
BEGIN
END_DATA_BLOCK

// folder: 04_HMI_Comand_Config

DATA_BLOCK "Line_OP"   // DB10
{ S7_Optimized_Access := 'TRUE' }
VERSION : 0.1
BEGIN
END_DATA_BLOCK

// folder: System blocks/Program resources

DATA_BLOCK "IEC_Timer_0_DB"   // DB1
{ S7_Optimized_Access := 'TRUE' }
AUTHOR : Simatic
FAMILY : IEC
NAME : IEC_TMR
VERSION : 1.0
// stored: InstanceOfName IEC_TIMER
"IEC_TIMER"
BEGIN
END_DATA_BLOCK

DATA_BLOCK "当前产量"   // DB2
{ S7_Optimized_Access := 'TRUE' }
AUTHOR : Simatic
FAMILY : IEC
NAME : CNTR
VERSION : 1.0
// stored: InstanceOfName IEC_COUNTER
"IEC_COUNTER"
BEGIN
END_DATA_BLOCK

DATA_BLOCK "IEC_Timer_0_DB_1"   // DB4
{ S7_Optimized_Access := 'TRUE' }
AUTHOR : Simatic
FAMILY : IEC
NAME : IEC_TMR
VERSION : 1.0
// stored: InstanceOfName IEC_TIMER
"IEC_TIMER"
BEGIN
END_DATA_BLOCK

DATA_BLOCK "IEC_Timer_0_DB_2"   // DB5
{ S7_Optimized_Access := 'TRUE' }
AUTHOR : Simatic
FAMILY : IEC
NAME : IEC_TMR
VERSION : 1.0
// stored: InstanceOfName IEC_TIMER
"IEC_TIMER"
BEGIN
END_DATA_BLOCK

DATA_BLOCK "IEC_Timer_0_DB_9"   // DB8
{ S7_Optimized_Access := 'TRUE' }
AUTHOR : Simatic
FAMILY : IEC
NAME : IEC_TMR
VERSION : 1.0
// stored: InstanceOfName IEC_TIMER
"IEC_TIMER"
BEGIN
END_DATA_BLOCK

DATA_BLOCK "IEC_Timer_0_DB_13"   // DB20
{ S7_Optimized_Access := 'TRUE' }
AUTHOR : Simatic
FAMILY : IEC
NAME : IEC_TMR
VERSION : 1.0
// stored: InstanceOfName IEC_TIMER
"IEC_TIMER"
BEGIN
END_DATA_BLOCK

DATA_BLOCK "清零防误触延时"   // DB27
{ S7_Optimized_Access := 'TRUE' }
AUTHOR : Simatic
FAMILY : IEC
NAME : IEC_TMR
VERSION : 1.0
// stored: InstanceOfName IEC_TIMER
"IEC_TIMER"
BEGIN
END_DATA_BLOCK

// folder: (top level)

FUNCTION "行程控制" : Void   // FC1, LAD
{ S7_Optimized_Access := 'TRUE' }
VERSION : 0.1
BEGIN

REGION Network 1
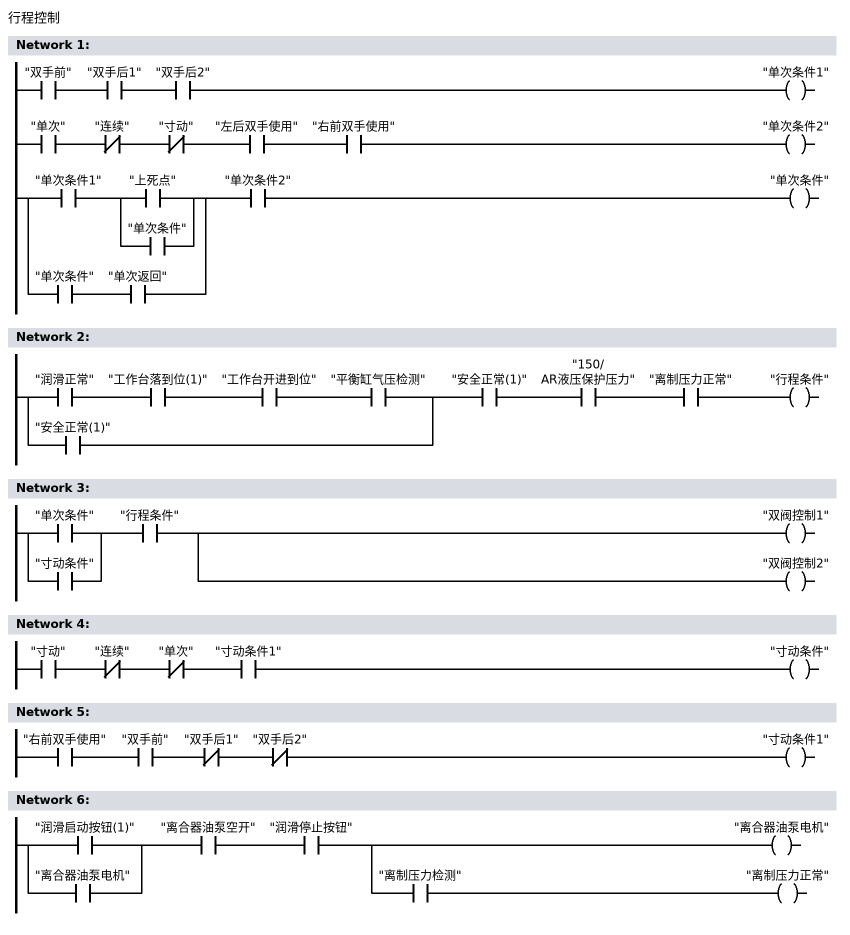
   RUNG wire#powerrail
      Contact( "双手前" )
      Contact( "双手后1" )
      Contact( "双手后2" )
      Coil( "单次条件1" )
   END_RUNG
   RUNG wire#powerrail
      Contact( "单次" )
      I_Contact( "连续" )
      I_Contact( "寸动" )
      Contact( "左后双手使用" )
      Contact( "右前双手使用" )
      Coil( "单次条件2" )
   END_RUNG
   RUNG wire#powerrail
      Contact( "单次条件1" )
      wire#w1
      Contact( "上死点" )
      wire#w2
      Contact( "单次条件2" )
      Coil( "单次条件" )
   END_RUNG
   RUNG wire#w1
      Contact( "单次条件" )
   END_RUNG wire#w2
   RUNG wire#powerrail
      Contact( "单次条件" )
      Contact( "单次返回" )
   END_RUNG wire#w2
   // the same network as SCL:
   "单次条件1" := "双手前" AND "双手后1" AND "双手后2";
   "单次条件2" := "单次" AND NOT "连续" AND NOT "寸动" AND "左后双手使用" AND "右前双手使用";
   "单次条件" := (("单次条件1" AND ("上死点" OR "单次条件")) OR ("单次条件" AND "单次返回")) AND "单次条件2";
END_REGION

REGION Network 2
   RUNG wire#powerrail
      Contact( "润滑正常" )
      Contact( "工作台落到位(1)" )
      Contact( "工作台开进到位" )
      Contact( "平衡缸气压检测" )
      wire#w1
      Contact( "安全正常(1)" )
      Contact( "150/AR液压保护压力" )
      Contact( "离制压力正常" )
      Coil( "行程条件" )
   END_RUNG
   RUNG wire#powerrail
      Contact( "安全正常(1)" )
   END_RUNG wire#w1
   // the same network as SCL:
   "行程条件" := (("润滑正常" AND "工作台落到位(1)" AND "工作台开进到位" AND "平衡缸气压检测") OR "安全正常(1)") AND "安全正常(1)" AND "150/AR液压保护压力" AND "离制压力正常";
END_REGION

REGION Network 3
   RUNG wire#powerrail
      Contact( "单次条件" )
      wire#w1
      Contact( "行程条件" )
      wire#w2
      Coil( "双阀控制1" )
   END_RUNG
   RUNG wire#powerrail
      Contact( "寸动条件" )
   END_RUNG wire#w1
   RUNG wire#w2
      Coil( "双阀控制2" )
   END_RUNG
   // the same network as SCL:
   "双阀控制1" := ("单次条件" OR "寸动条件") AND "行程条件";
   "双阀控制2" := "双阀控制1";
END_REGION

REGION Network 4
   RUNG wire#powerrail
      Contact( "寸动" )
      I_Contact( "连续" )
      I_Contact( "单次" )
      Contact( "寸动条件1" )
      Coil( "寸动条件" )
   END_RUNG
   // the same network as SCL:
   "寸动条件" := "寸动" AND NOT "连续" AND NOT "单次" AND "寸动条件1";
END_REGION

REGION Network 5
   RUNG wire#powerrail
      Contact( "右前双手使用" )
      Contact( "双手前" )
      I_Contact( "双手后1" )
      I_Contact( "双手后2" )
      Coil( "寸动条件1" )
   END_RUNG
   // the same network as SCL:
   "寸动条件1" := "右前双手使用" AND "双手前" AND NOT "双手后1" AND NOT "双手后2";
END_REGION

REGION Network 6
   RUNG wire#powerrail
      Contact( "润滑启动按钮(1)" )
      wire#w1
      Contact( "离合器油泵空开" )
      Contact( "润滑停止按钮" )
      wire#w2
      Coil( "离合器油泵电机" )
   END_RUNG
   RUNG wire#powerrail
      Contact( "离合器油泵电机" )
   END_RUNG wire#w1
   RUNG wire#w2
      Contact( "离制压力检测" )
      Coil( "离制压力正常" )
   END_RUNG
   // the same network as SCL:
   "离合器油泵电机" := ("润滑启动按钮(1)" OR "离合器油泵电机") AND "离合器油泵空开" AND "润滑停止按钮";
   "离制压力正常" := "离合器油泵电机" AND "离制压力检测";
END_REGION
END_FUNCTION

FUNCTION "横梁编码器调制" : Void   // FC2, LAD
{ S7_Optimized_Access := 'TRUE' }
VERSION : 0.1
BEGIN

REGION Network 1
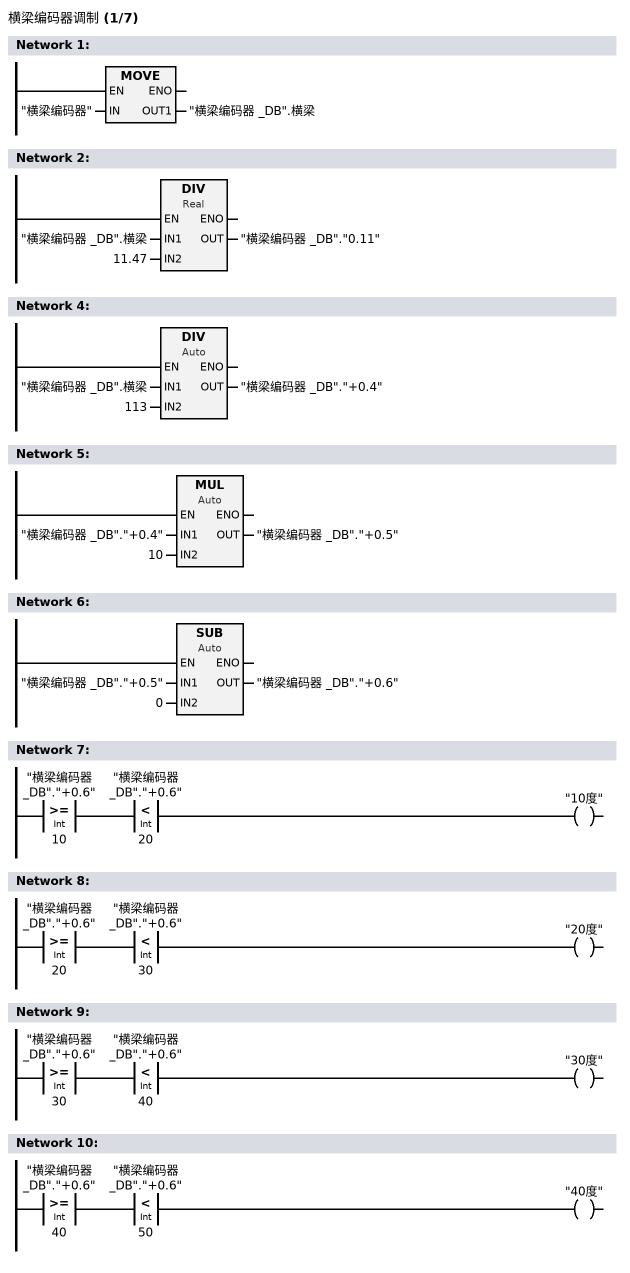
   RUNG wire#powerrail
      Move(in := "横梁编码器", out1 => "横梁编码器 _DB".横梁)
   END_RUNG
   // the same network as SCL:
   "横梁编码器 _DB".横梁 := "横梁编码器";
END_REGION

REGION Network 2
   RUNG wire#powerrail
      { S7_Templates := "SrcType := Real" } Div(in1 := "横梁编码器 _DB".横梁, in2 := 11.47, out => "横梁编码器 _DB"."0.11")
   END_RUNG
   // the same network as SCL:
   "横梁编码器 _DB"."0.11" := "横梁编码器 _DB".横梁 / 11.47;
END_REGION

REGION Network 4
   RUNG wire#powerrail
      Div(in1 := "横梁编码器 _DB".横梁, in2 := 113, out => "横梁编码器 _DB"."+0.4")
   END_RUNG
   // the same network as SCL:
   "横梁编码器 _DB"."+0.4" := "横梁编码器 _DB".横梁 / 113;
END_REGION

REGION Network 5
   RUNG wire#powerrail
      Mul(in1 := "横梁编码器 _DB"."+0.4", in2 := 10, out => "横梁编码器 _DB"."+0.5")
   END_RUNG
   // the same network as SCL:
   "横梁编码器 _DB"."+0.5" := "横梁编码器 _DB"."+0.4" * 10;
END_REGION

REGION Network 6
   RUNG wire#powerrail
      Sub(in1 := "横梁编码器 _DB"."+0.5", in2 := 0, out => "横梁编码器 _DB"."+0.6")
   END_RUNG
   // the same network as SCL:
   "横梁编码器 _DB"."+0.6" := "横梁编码器 _DB"."+0.5" - 0;
END_REGION

REGION Network 7
   RUNG wire#powerrail
      { S7_Templates := "SrcType := Int" } GE_Contact(in1 := "横梁编码器 _DB"."+0.6", in2 := 10)
      { S7_Templates := "SrcType := Int" } LT_Contact(in1 := "横梁编码器 _DB"."+0.6", in2 := 20)
      Coil( "10度" )
   END_RUNG
   // the same network as SCL:
   "10度" := ("横梁编码器 _DB"."+0.6" >= 10) AND ("横梁编码器 _DB"."+0.6" < 20);
END_REGION

REGION Network 8
   RUNG wire#powerrail
      { S7_Templates := "SrcType := Int" } GE_Contact(in1 := "横梁编码器 _DB"."+0.6", in2 := 20)
      { S7_Templates := "SrcType := Int" } LT_Contact(in1 := "横梁编码器 _DB"."+0.6", in2 := 30)
      Coil( "20度" )
   END_RUNG
   // the same network as SCL:
   "20度" := ("横梁编码器 _DB"."+0.6" >= 20) AND ("横梁编码器 _DB"."+0.6" < 30);
END_REGION

REGION Network 9
   RUNG wire#powerrail
      { S7_Templates := "SrcType := Int" } GE_Contact(in1 := "横梁编码器 _DB"."+0.6", in2 := 30)
      { S7_Templates := "SrcType := Int" } LT_Contact(in1 := "横梁编码器 _DB"."+0.6", in2 := 40)
      Coil( "30度" )
   END_RUNG
   // the same network as SCL:
   "30度" := ("横梁编码器 _DB"."+0.6" >= 30) AND ("横梁编码器 _DB"."+0.6" < 40);
END_REGION

REGION Network 10
   RUNG wire#powerrail
      { S7_Templates := "SrcType := Int" } GE_Contact(in1 := "横梁编码器 _DB"."+0.6", in2 := 40)
      { S7_Templates := "SrcType := Int" } LT_Contact(in1 := "横梁编码器 _DB"."+0.6", in2 := 50)
      Coil( "40度" )
   END_RUNG
   // the same network as SCL:
   "40度" := ("横梁编码器 _DB"."+0.6" >= 40) AND ("横梁编码器 _DB"."+0.6" < 50);
END_REGION

REGION Network 11
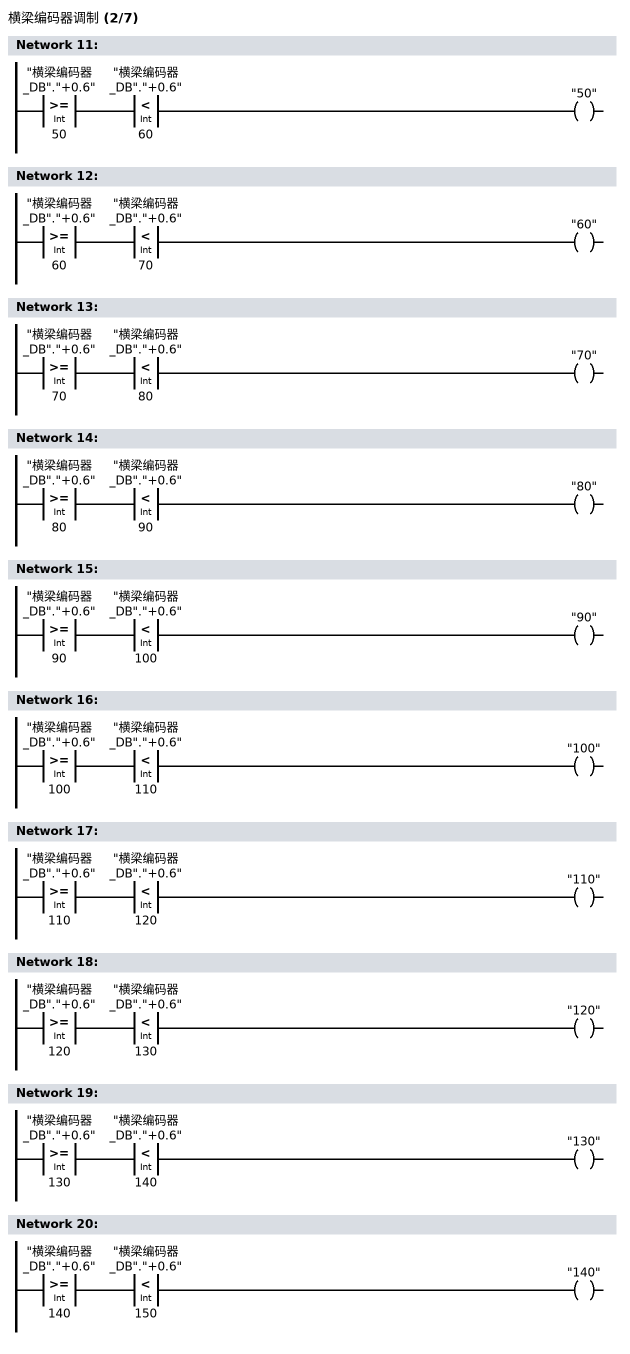
   RUNG wire#powerrail
      { S7_Templates := "SrcType := Int" } GE_Contact(in1 := "横梁编码器 _DB"."+0.6", in2 := 50)
      { S7_Templates := "SrcType := Int" } LT_Contact(in1 := "横梁编码器 _DB"."+0.6", in2 := 60)
      Coil( "50" )
   END_RUNG
   // the same network as SCL:
   "50" := ("横梁编码器 _DB"."+0.6" >= 50) AND ("横梁编码器 _DB"."+0.6" < 60);
END_REGION

REGION Network 12
   RUNG wire#powerrail
      { S7_Templates := "SrcType := Int" } GE_Contact(in1 := "横梁编码器 _DB"."+0.6", in2 := 60)
      { S7_Templates := "SrcType := Int" } LT_Contact(in1 := "横梁编码器 _DB"."+0.6", in2 := 70)
      Coil( "60" )
   END_RUNG
   // the same network as SCL:
   "60" := ("横梁编码器 _DB"."+0.6" >= 60) AND ("横梁编码器 _DB"."+0.6" < 70);
END_REGION

REGION Network 13
   RUNG wire#powerrail
      { S7_Templates := "SrcType := Int" } GE_Contact(in1 := "横梁编码器 _DB"."+0.6", in2 := 70)
      { S7_Templates := "SrcType := Int" } LT_Contact(in1 := "横梁编码器 _DB"."+0.6", in2 := 80)
      Coil( "70" )
   END_RUNG
   // the same network as SCL:
   "70" := ("横梁编码器 _DB"."+0.6" >= 70) AND ("横梁编码器 _DB"."+0.6" < 80);
END_REGION

REGION Network 14
   RUNG wire#powerrail
      { S7_Templates := "SrcType := Int" } GE_Contact(in1 := "横梁编码器 _DB"."+0.6", in2 := 80)
      { S7_Templates := "SrcType := Int" } LT_Contact(in1 := "横梁编码器 _DB"."+0.6", in2 := 90)
      Coil( "80" )
   END_RUNG
   // the same network as SCL:
   "80" := ("横梁编码器 _DB"."+0.6" >= 80) AND ("横梁编码器 _DB"."+0.6" < 90);
END_REGION

REGION Network 15
   RUNG wire#powerrail
      { S7_Templates := "SrcType := Int" } GE_Contact(in1 := "横梁编码器 _DB"."+0.6", in2 := 90)
      { S7_Templates := "SrcType := Int" } LT_Contact(in1 := "横梁编码器 _DB"."+0.6", in2 := 100)
      Coil( "90" )
   END_RUNG
   // the same network as SCL:
   "90" := ("横梁编码器 _DB"."+0.6" >= 90) AND ("横梁编码器 _DB"."+0.6" < 100);
END_REGION

REGION Network 16
   RUNG wire#powerrail
      { S7_Templates := "SrcType := Int" } GE_Contact(in1 := "横梁编码器 _DB"."+0.6", in2 := 100)
      { S7_Templates := "SrcType := Int" } LT_Contact(in1 := "横梁编码器 _DB"."+0.6", in2 := 110)
      Coil( "100" )
   END_RUNG
   // the same network as SCL:
   "100" := ("横梁编码器 _DB"."+0.6" >= 100) AND ("横梁编码器 _DB"."+0.6" < 110);
END_REGION

REGION Network 17
   RUNG wire#powerrail
      { S7_Templates := "SrcType := Int" } GE_Contact(in1 := "横梁编码器 _DB"."+0.6", in2 := 110)
      { S7_Templates := "SrcType := Int" } LT_Contact(in1 := "横梁编码器 _DB"."+0.6", in2 := 120)
      Coil( "110" )
   END_RUNG
   // the same network as SCL:
   "110" := ("横梁编码器 _DB"."+0.6" >= 110) AND ("横梁编码器 _DB"."+0.6" < 120);
END_REGION

REGION Network 18
   RUNG wire#powerrail
      { S7_Templates := "SrcType := Int" } GE_Contact(in1 := "横梁编码器 _DB"."+0.6", in2 := 120)
      { S7_Templates := "SrcType := Int" } LT_Contact(in1 := "横梁编码器 _DB"."+0.6", in2 := 130)
      Coil( "120" )
   END_RUNG
   // the same network as SCL:
   "120" := ("横梁编码器 _DB"."+0.6" >= 120) AND ("横梁编码器 _DB"."+0.6" < 130);
END_REGION

REGION Network 19
   RUNG wire#powerrail
      { S7_Templates := "SrcType := Int" } GE_Contact(in1 := "横梁编码器 _DB"."+0.6", in2 := 130)
      { S7_Templates := "SrcType := Int" } LT_Contact(in1 := "横梁编码器 _DB"."+0.6", in2 := 140)
      Coil( "130" )
   END_RUNG
   // the same network as SCL:
   "130" := ("横梁编码器 _DB"."+0.6" >= 130) AND ("横梁编码器 _DB"."+0.6" < 140);
END_REGION

REGION Network 20
   RUNG wire#powerrail
      { S7_Templates := "SrcType := Int" } GE_Contact(in1 := "横梁编码器 _DB"."+0.6", in2 := 140)
      { S7_Templates := "SrcType := Int" } LT_Contact(in1 := "横梁编码器 _DB"."+0.6", in2 := 150)
      Coil( "140" )
   END_RUNG
   // the same network as SCL:
   "140" := ("横梁编码器 _DB"."+0.6" >= 140) AND ("横梁编码器 _DB"."+0.6" < 150);
END_REGION

REGION Network 21
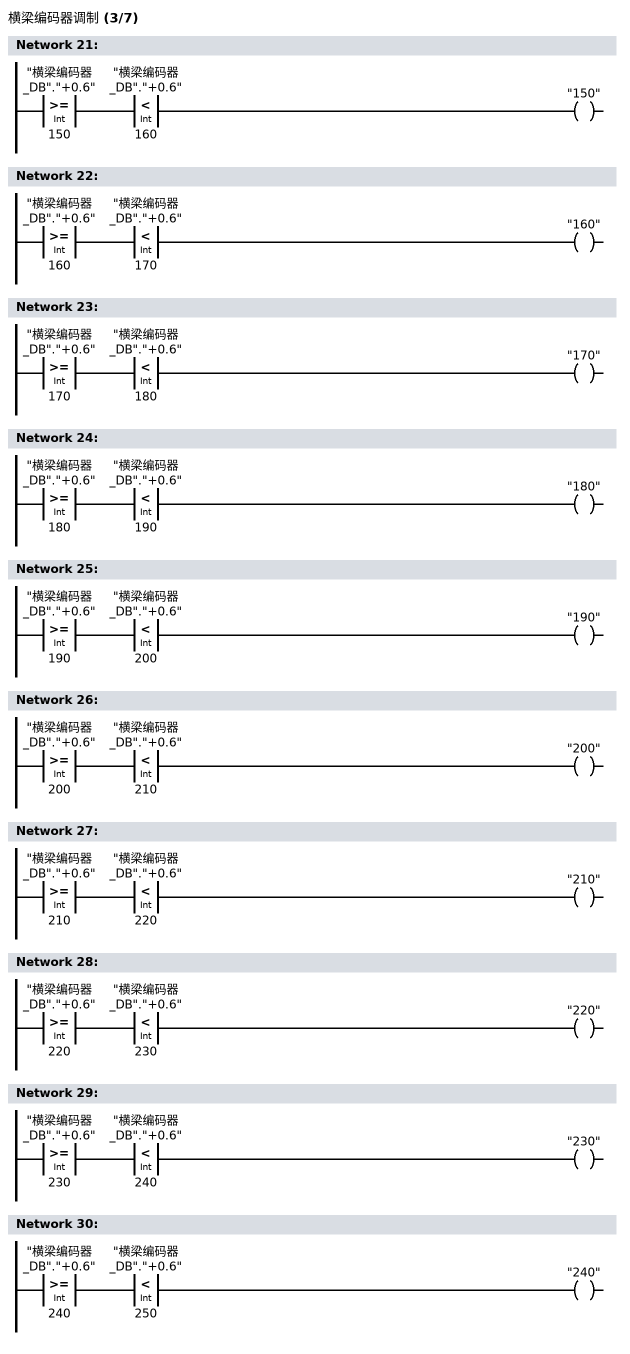
   RUNG wire#powerrail
      { S7_Templates := "SrcType := Int" } GE_Contact(in1 := "横梁编码器 _DB"."+0.6", in2 := 150)
      { S7_Templates := "SrcType := Int" } LT_Contact(in1 := "横梁编码器 _DB"."+0.6", in2 := 160)
      Coil( "150" )
   END_RUNG
   // the same network as SCL:
   "150" := ("横梁编码器 _DB"."+0.6" >= 150) AND ("横梁编码器 _DB"."+0.6" < 160);
END_REGION

REGION Network 22
   RUNG wire#powerrail
      { S7_Templates := "SrcType := Int" } GE_Contact(in1 := "横梁编码器 _DB"."+0.6", in2 := 160)
      { S7_Templates := "SrcType := Int" } LT_Contact(in1 := "横梁编码器 _DB"."+0.6", in2 := 170)
      Coil( "160" )
   END_RUNG
   // the same network as SCL:
   "160" := ("横梁编码器 _DB"."+0.6" >= 160) AND ("横梁编码器 _DB"."+0.6" < 170);
END_REGION

REGION Network 23
   RUNG wire#powerrail
      { S7_Templates := "SrcType := Int" } GE_Contact(in1 := "横梁编码器 _DB"."+0.6", in2 := 170)
      { S7_Templates := "SrcType := Int" } LT_Contact(in1 := "横梁编码器 _DB"."+0.6", in2 := 180)
      Coil( "170" )
   END_RUNG
   // the same network as SCL:
   "170" := ("横梁编码器 _DB"."+0.6" >= 170) AND ("横梁编码器 _DB"."+0.6" < 180);
END_REGION

REGION Network 24
   RUNG wire#powerrail
      { S7_Templates := "SrcType := Int" } GE_Contact(in1 := "横梁编码器 _DB"."+0.6", in2 := 180)
      { S7_Templates := "SrcType := Int" } LT_Contact(in1 := "横梁编码器 _DB"."+0.6", in2 := 190)
      Coil( "180" )
   END_RUNG
   // the same network as SCL:
   "180" := ("横梁编码器 _DB"."+0.6" >= 180) AND ("横梁编码器 _DB"."+0.6" < 190);
END_REGION

REGION Network 25
   RUNG wire#powerrail
      { S7_Templates := "SrcType := Int" } GE_Contact(in1 := "横梁编码器 _DB"."+0.6", in2 := 190)
      { S7_Templates := "SrcType := Int" } LT_Contact(in1 := "横梁编码器 _DB"."+0.6", in2 := 200)
      Coil( "190" )
   END_RUNG
   // the same network as SCL:
   "190" := ("横梁编码器 _DB"."+0.6" >= 190) AND ("横梁编码器 _DB"."+0.6" < 200);
END_REGION

REGION Network 26
   RUNG wire#powerrail
      { S7_Templates := "SrcType := Int" } GE_Contact(in1 := "横梁编码器 _DB"."+0.6", in2 := 200)
      { S7_Templates := "SrcType := Int" } LT_Contact(in1 := "横梁编码器 _DB"."+0.6", in2 := 210)
      Coil( "200" )
   END_RUNG
   // the same network as SCL:
   "200" := ("横梁编码器 _DB"."+0.6" >= 200) AND ("横梁编码器 _DB"."+0.6" < 210);
END_REGION

REGION Network 27
   RUNG wire#powerrail
      { S7_Templates := "SrcType := Int" } GE_Contact(in1 := "横梁编码器 _DB"."+0.6", in2 := 210)
      { S7_Templates := "SrcType := Int" } LT_Contact(in1 := "横梁编码器 _DB"."+0.6", in2 := 220)
      Coil( "210" )
   END_RUNG
   // the same network as SCL:
   "210" := ("横梁编码器 _DB"."+0.6" >= 210) AND ("横梁编码器 _DB"."+0.6" < 220);
END_REGION

REGION Network 28
   RUNG wire#powerrail
      { S7_Templates := "SrcType := Int" } GE_Contact(in1 := "横梁编码器 _DB"."+0.6", in2 := 220)
      { S7_Templates := "SrcType := Int" } LT_Contact(in1 := "横梁编码器 _DB"."+0.6", in2 := 230)
      Coil( "220" )
   END_RUNG
   // the same network as SCL:
   "220" := ("横梁编码器 _DB"."+0.6" >= 220) AND ("横梁编码器 _DB"."+0.6" < 230);
END_REGION

REGION Network 29
   RUNG wire#powerrail
      { S7_Templates := "SrcType := Int" } GE_Contact(in1 := "横梁编码器 _DB"."+0.6", in2 := 230)
      { S7_Templates := "SrcType := Int" } LT_Contact(in1 := "横梁编码器 _DB"."+0.6", in2 := 240)
      Coil( "230" )
   END_RUNG
   // the same network as SCL:
   "230" := ("横梁编码器 _DB"."+0.6" >= 230) AND ("横梁编码器 _DB"."+0.6" < 240);
END_REGION

REGION Network 30
   RUNG wire#powerrail
      { S7_Templates := "SrcType := Int" } GE_Contact(in1 := "横梁编码器 _DB"."+0.6", in2 := 240)
      { S7_Templates := "SrcType := Int" } LT_Contact(in1 := "横梁编码器 _DB"."+0.6", in2 := 250)
      Coil( "240" )
   END_RUNG
   // the same network as SCL:
   "240" := ("横梁编码器 _DB"."+0.6" >= 240) AND ("横梁编码器 _DB"."+0.6" < 250);
END_REGION

REGION Network 31
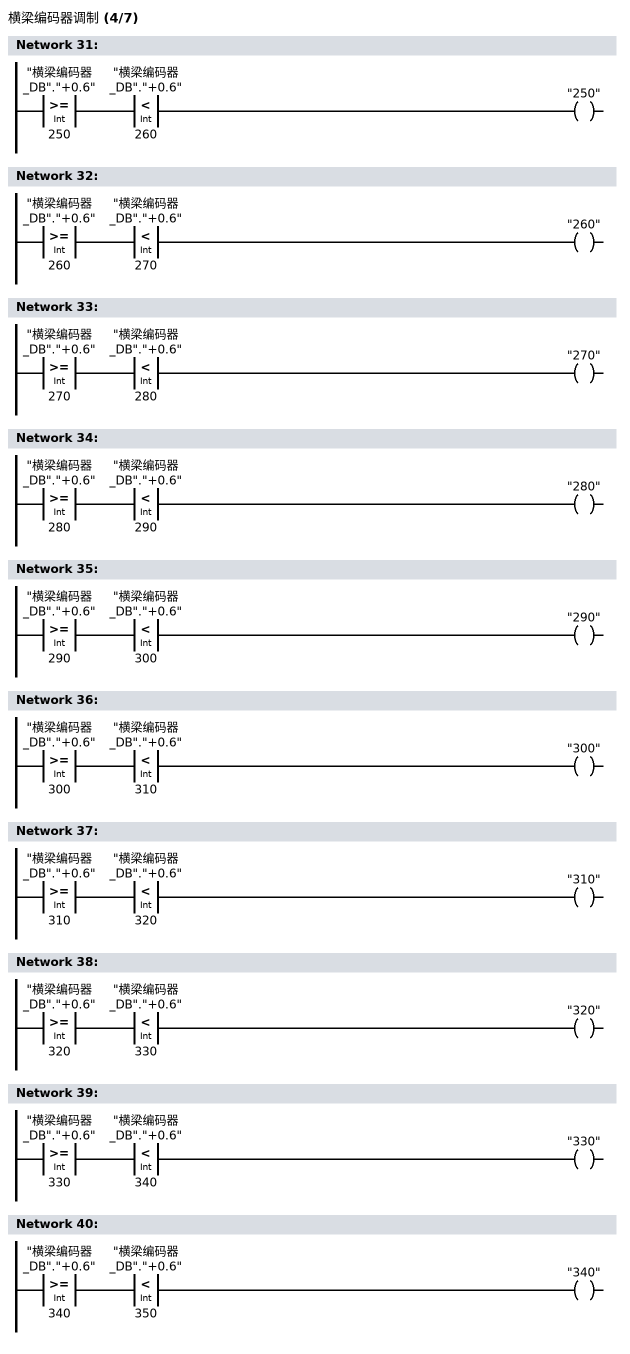
   RUNG wire#powerrail
      { S7_Templates := "SrcType := Int" } GE_Contact(in1 := "横梁编码器 _DB"."+0.6", in2 := 250)
      { S7_Templates := "SrcType := Int" } LT_Contact(in1 := "横梁编码器 _DB"."+0.6", in2 := 260)
      Coil( "250" )
   END_RUNG
   // the same network as SCL:
   "250" := ("横梁编码器 _DB"."+0.6" >= 250) AND ("横梁编码器 _DB"."+0.6" < 260);
END_REGION

REGION Network 32
   RUNG wire#powerrail
      { S7_Templates := "SrcType := Int" } GE_Contact(in1 := "横梁编码器 _DB"."+0.6", in2 := 260)
      { S7_Templates := "SrcType := Int" } LT_Contact(in1 := "横梁编码器 _DB"."+0.6", in2 := 270)
      Coil( "260" )
   END_RUNG
   // the same network as SCL:
   "260" := ("横梁编码器 _DB"."+0.6" >= 260) AND ("横梁编码器 _DB"."+0.6" < 270);
END_REGION

REGION Network 33
   RUNG wire#powerrail
      { S7_Templates := "SrcType := Int" } GE_Contact(in1 := "横梁编码器 _DB"."+0.6", in2 := 270)
      { S7_Templates := "SrcType := Int" } LT_Contact(in1 := "横梁编码器 _DB"."+0.6", in2 := 280)
      Coil( "270" )
   END_RUNG
   // the same network as SCL:
   "270" := ("横梁编码器 _DB"."+0.6" >= 270) AND ("横梁编码器 _DB"."+0.6" < 280);
END_REGION

REGION Network 34
   RUNG wire#powerrail
      { S7_Templates := "SrcType := Int" } GE_Contact(in1 := "横梁编码器 _DB"."+0.6", in2 := 280)
      { S7_Templates := "SrcType := Int" } LT_Contact(in1 := "横梁编码器 _DB"."+0.6", in2 := 290)
      Coil( "280" )
   END_RUNG
   // the same network as SCL:
   "280" := ("横梁编码器 _DB"."+0.6" >= 280) AND ("横梁编码器 _DB"."+0.6" < 290);
END_REGION

REGION Network 35
   RUNG wire#powerrail
      { S7_Templates := "SrcType := Int" } GE_Contact(in1 := "横梁编码器 _DB"."+0.6", in2 := 290)
      { S7_Templates := "SrcType := Int" } LT_Contact(in1 := "横梁编码器 _DB"."+0.6", in2 := 300)
      Coil( "290" )
   END_RUNG
   // the same network as SCL:
   "290" := ("横梁编码器 _DB"."+0.6" >= 290) AND ("横梁编码器 _DB"."+0.6" < 300);
END_REGION

REGION Network 36
   RUNG wire#powerrail
      { S7_Templates := "SrcType := Int" } GE_Contact(in1 := "横梁编码器 _DB"."+0.6", in2 := 300)
      { S7_Templates := "SrcType := Int" } LT_Contact(in1 := "横梁编码器 _DB"."+0.6", in2 := 310)
      Coil( "300" )
   END_RUNG
   // the same network as SCL:
   "300" := ("横梁编码器 _DB"."+0.6" >= 300) AND ("横梁编码器 _DB"."+0.6" < 310);
END_REGION

REGION Network 37
   RUNG wire#powerrail
      { S7_Templates := "SrcType := Int" } GE_Contact(in1 := "横梁编码器 _DB"."+0.6", in2 := 310)
      { S7_Templates := "SrcType := Int" } LT_Contact(in1 := "横梁编码器 _DB"."+0.6", in2 := 320)
      Coil( "310" )
   END_RUNG
   // the same network as SCL:
   "310" := ("横梁编码器 _DB"."+0.6" >= 310) AND ("横梁编码器 _DB"."+0.6" < 320);
END_REGION

REGION Network 38
   RUNG wire#powerrail
      { S7_Templates := "SrcType := Int" } GE_Contact(in1 := "横梁编码器 _DB"."+0.6", in2 := 320)
      { S7_Templates := "SrcType := Int" } LT_Contact(in1 := "横梁编码器 _DB"."+0.6", in2 := 330)
      Coil( "320" )
   END_RUNG
   // the same network as SCL:
   "320" := ("横梁编码器 _DB"."+0.6" >= 320) AND ("横梁编码器 _DB"."+0.6" < 330);
END_REGION

REGION Network 39
   RUNG wire#powerrail
      { S7_Templates := "SrcType := Int" } GE_Contact(in1 := "横梁编码器 _DB"."+0.6", in2 := 330)
      { S7_Templates := "SrcType := Int" } LT_Contact(in1 := "横梁编码器 _DB"."+0.6", in2 := 340)
      Coil( "330" )
   END_RUNG
   // the same network as SCL:
   "330" := ("横梁编码器 _DB"."+0.6" >= 330) AND ("横梁编码器 _DB"."+0.6" < 340);
END_REGION

REGION Network 40
   RUNG wire#powerrail
      { S7_Templates := "SrcType := Int" } GE_Contact(in1 := "横梁编码器 _DB"."+0.6", in2 := 340)
      { S7_Templates := "SrcType := Int" } LT_Contact(in1 := "横梁编码器 _DB"."+0.6", in2 := 350)
      Coil( "340" )
   END_RUNG
   // the same network as SCL:
   "340" := ("横梁编码器 _DB"."+0.6" >= 340) AND ("横梁编码器 _DB"."+0.6" < 350);
END_REGION

REGION Network 41
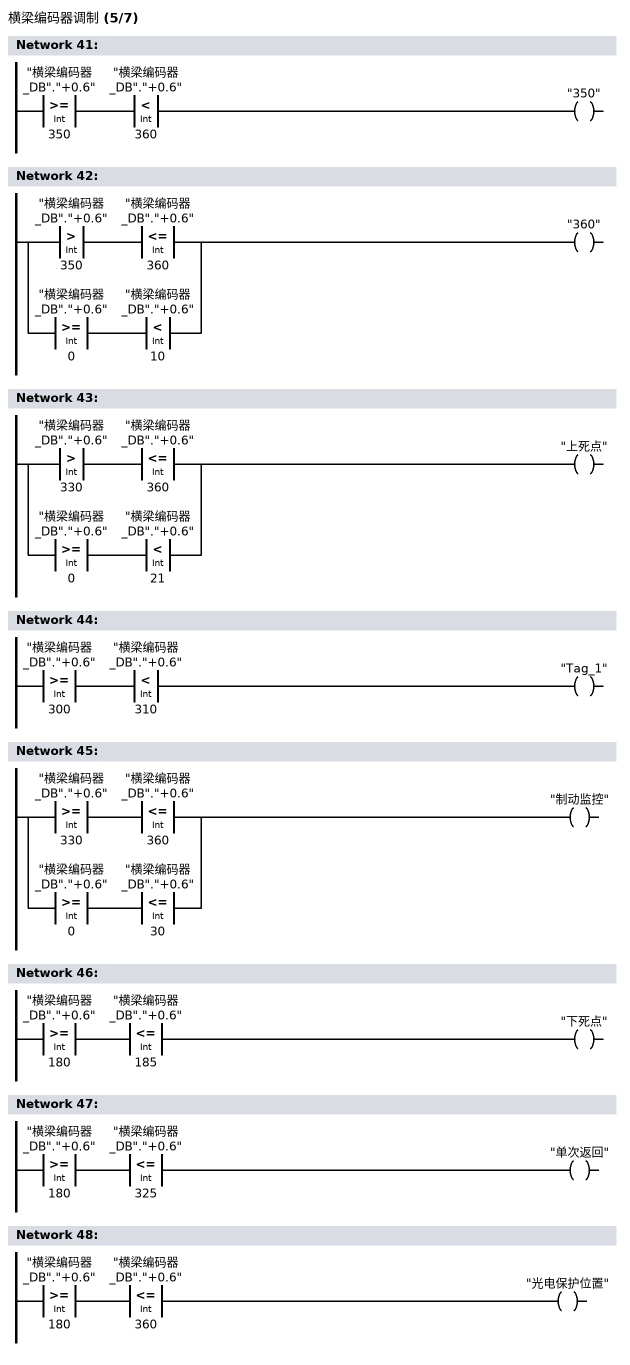
   RUNG wire#powerrail
      { S7_Templates := "SrcType := Int" } GE_Contact(in1 := "横梁编码器 _DB"."+0.6", in2 := 350)
      { S7_Templates := "SrcType := Int" } LT_Contact(in1 := "横梁编码器 _DB"."+0.6", in2 := 360)
      Coil( "350" )
   END_RUNG
   // the same network as SCL:
   "350" := ("横梁编码器 _DB"."+0.6" >= 350) AND ("横梁编码器 _DB"."+0.6" < 360);
END_REGION

REGION Network 42
   RUNG wire#powerrail
      { S7_Templates := "SrcType := Int" } GT_Contact(in1 := "横梁编码器 _DB"."+0.6", in2 := 350)
      { S7_Templates := "SrcType := Int" } LE_Contact(in1 := "横梁编码器 _DB"."+0.6", in2 := 360)
      wire#w1
      Coil( "360" )
   END_RUNG
   RUNG wire#powerrail
      { S7_Templates := "SrcType := Int" } GE_Contact(in1 := "横梁编码器 _DB"."+0.6", in2 := 0)
      { S7_Templates := "SrcType := Int" } LT_Contact(in1 := "横梁编码器 _DB"."+0.6", in2 := 10)
   END_RUNG wire#w1
   // the same network as SCL:
   "360" := (("横梁编码器 _DB"."+0.6" > 350) AND ("横梁编码器 _DB"."+0.6" <= 360)) OR (("横梁编码器 _DB"."+0.6" >= 0) AND ("横梁编码器 _DB"."+0.6" < 10));
END_REGION

REGION Network 43
   RUNG wire#powerrail
      { S7_Templates := "SrcType := Int" } GT_Contact(in1 := "横梁编码器 _DB"."+0.6", in2 := 330)
      { S7_Templates := "SrcType := Int" } LE_Contact(in1 := "横梁编码器 _DB"."+0.6", in2 := 360)
      wire#w1
      Coil( "上死点" )
   END_RUNG
   RUNG wire#powerrail
      { S7_Templates := "SrcType := Int" } GE_Contact(in1 := "横梁编码器 _DB"."+0.6", in2 := 0)
      { S7_Templates := "SrcType := Int" } LT_Contact(in1 := "横梁编码器 _DB"."+0.6", in2 := 21)
   END_RUNG wire#w1
   // the same network as SCL:
   "上死点" := (("横梁编码器 _DB"."+0.6" > 330) AND ("横梁编码器 _DB"."+0.6" <= 360)) OR (("横梁编码器 _DB"."+0.6" >= 0) AND ("横梁编码器 _DB"."+0.6" < 21));
END_REGION

REGION Network 44
   RUNG wire#powerrail
      { S7_Templates := "SrcType := Int" } GE_Contact(in1 := "横梁编码器 _DB"."+0.6", in2 := 300)
      { S7_Templates := "SrcType := Int" } LT_Contact(in1 := "横梁编码器 _DB"."+0.6", in2 := 310)
      Coil( "Tag_1" )
   END_RUNG
   // the same network as SCL:
   "Tag_1" := ("横梁编码器 _DB"."+0.6" >= 300) AND ("横梁编码器 _DB"."+0.6" < 310);
END_REGION

REGION Network 45
   RUNG wire#powerrail
      { S7_Templates := "SrcType := Int" } GE_Contact(in1 := "横梁编码器 _DB"."+0.6", in2 := 330)
      { S7_Templates := "SrcType := Int" } LE_Contact(in1 := "横梁编码器 _DB"."+0.6", in2 := 360)
      wire#w1
      Coil( "制动监控" )
   END_RUNG
   RUNG wire#powerrail
      { S7_Templates := "SrcType := Int" } GE_Contact(in1 := "横梁编码器 _DB"."+0.6", in2 := 0)
      { S7_Templates := "SrcType := Int" } LE_Contact(in1 := "横梁编码器 _DB"."+0.6", in2 := 30)
   END_RUNG wire#w1
   // the same network as SCL:
   "制动监控" := (("横梁编码器 _DB"."+0.6" >= 330) AND ("横梁编码器 _DB"."+0.6" <= 360)) OR (("横梁编码器 _DB"."+0.6" >= 0) AND ("横梁编码器 _DB"."+0.6" <= 30));
END_REGION

REGION Network 46
   RUNG wire#powerrail
      { S7_Templates := "SrcType := Int" } GE_Contact(in1 := "横梁编码器 _DB"."+0.6", in2 := 180)
      { S7_Templates := "SrcType := Int" } LE_Contact(in1 := "横梁编码器 _DB"."+0.6", in2 := 185)
      Coil( "下死点" )
   END_RUNG
   // the same network as SCL:
   "下死点" := ("横梁编码器 _DB"."+0.6" >= 180) AND ("横梁编码器 _DB"."+0.6" <= 185);
END_REGION

REGION Network 47
   RUNG wire#powerrail
      { S7_Templates := "SrcType := Int" } GE_Contact(in1 := "横梁编码器 _DB"."+0.6", in2 := 180)
      { S7_Templates := "SrcType := Int" } LE_Contact(in1 := "横梁编码器 _DB"."+0.6", in2 := 325)
      Coil( "单次返回" )
   END_RUNG
   // the same network as SCL:
   "单次返回" := ("横梁编码器 _DB"."+0.6" >= 180) AND ("横梁编码器 _DB"."+0.6" <= 325);
END_REGION

REGION Network 48
   RUNG wire#powerrail
      { S7_Templates := "SrcType := Int" } GE_Contact(in1 := "横梁编码器 _DB"."+0.6", in2 := 180)
      { S7_Templates := "SrcType := Int" } LE_Contact(in1 := "横梁编码器 _DB"."+0.6", in2 := 360)
      Coil( "光电保护位置" )
   END_RUNG
   // the same network as SCL:
   "光电保护位置" := ("横梁编码器 _DB"."+0.6" >= 180) AND ("横梁编码器 _DB"."+0.6" <= 360);
END_REGION

REGION Network 49
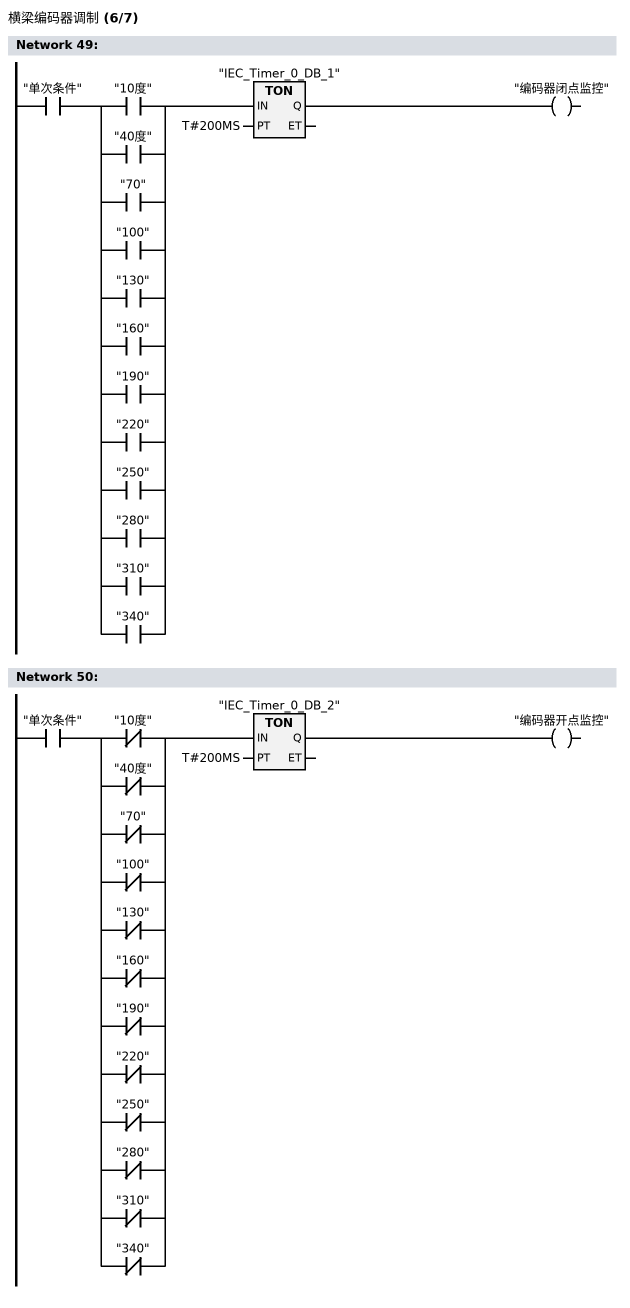
   "IEC_Timer_0_DB_1".TON(IN := "单次条件" AND ("10度" OR "40度" OR "70" OR "100" OR "130" OR "160" OR "190" OR "220" OR "250" OR "280" OR "310" OR "340"),
                          PT := T#200MS);
   "编码器闭点监控" := "IEC_Timer_0_DB_1".Q;
END_REGION

REGION Network 50
   "IEC_Timer_0_DB_2".TON(IN := "单次条件" AND (NOT "10度" OR NOT "40度" OR NOT "70" OR NOT "100" OR NOT "130" OR NOT "160" OR NOT "190" OR NOT "220" OR NOT "250" OR NOT "280" OR NOT "310" OR NOT "340"),
                          PT := T#200MS);
   "编码器开点监控" := "IEC_Timer_0_DB_2".Q;
END_REGION

REGION Network 51
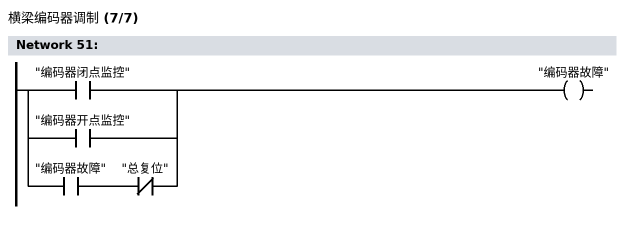
   RUNG wire#powerrail
      Contact( "编码器闭点监控" )
      wire#w1
      Coil( "编码器故障" )
   END_RUNG
   RUNG wire#powerrail
      Contact( "编码器开点监控" )
   END_RUNG wire#w1
   RUNG wire#powerrail
      Contact( "编码器故障" )
      I_Contact( "总复位" )
   END_RUNG wire#w1
   // the same network as SCL:
   "编码器故障" := "编码器闭点监控" OR "编码器开点监控" OR ("编码器故障" AND NOT "总复位");
END_REGION
END_FUNCTION

FUNCTION "10-润滑" : Void   // FC3, LAD
{ S7_Optimized_Access := 'TRUE' }
VERSION : 0.1
   VAR_TEMP
      主分油器打油次数 : DB_ANY;
   END_VAR
BEGIN

REGION Network 1: 润滑启动
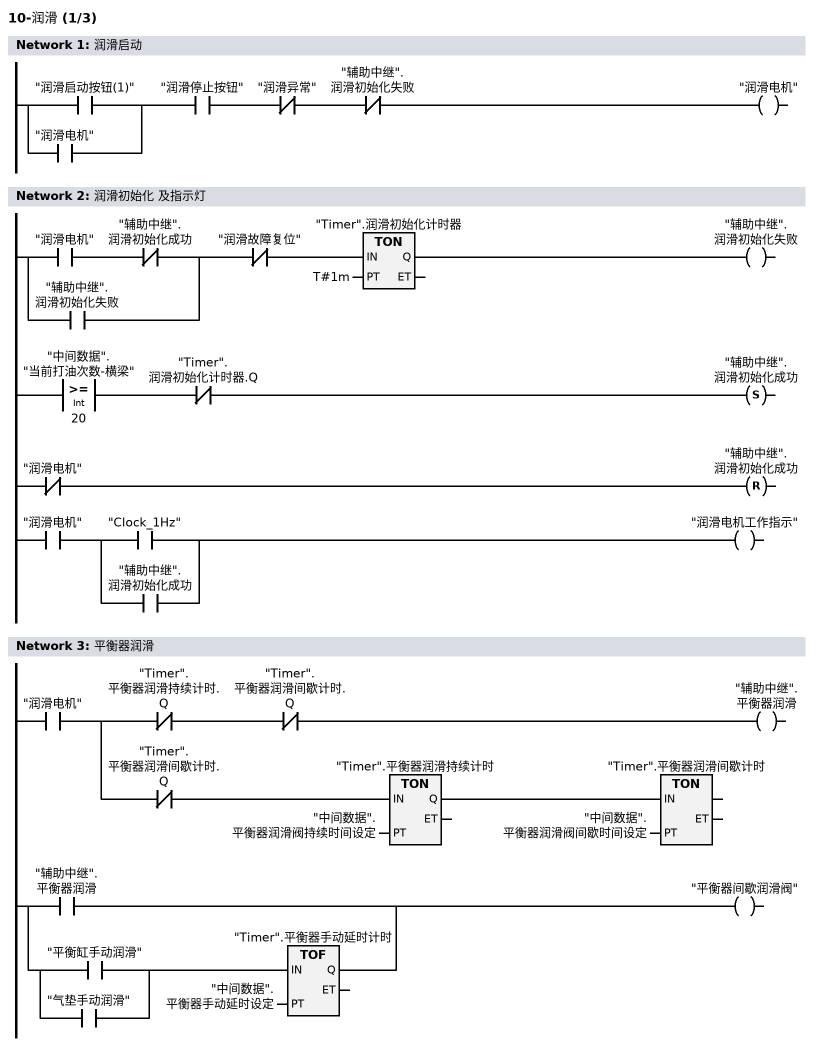
   RUNG wire#powerrail
      Contact( "润滑启动按钮(1)" )
      wire#w1
      Contact( "润滑停止按钮" )
      I_Contact( "润滑异常" )
      I_Contact( "辅助中继".润滑初始化失败 )
      Coil( "润滑电机" )
   END_RUNG
   RUNG wire#powerrail
      Contact( "润滑电机" )
   END_RUNG wire#w1
   // the same network as SCL:
   "润滑电机" := ("润滑启动按钮(1)" OR "润滑电机") AND "润滑停止按钮" AND NOT "润滑异常" AND NOT "辅助中继".润滑初始化失败;
END_REGION

REGION Network 2: 润滑初始化 及指示灯
   "Timer".润滑初始化计时器.TON(IN := (("润滑电机" AND NOT "辅助中继".润滑初始化成功) OR "辅助中继".润滑初始化失败) AND NOT "润滑故障复位", PT := T#1m);
   "辅助中继".润滑初始化失败 := "Timer".润滑初始化计时器.Q;
   IF ("中间数据"."当前打油次数-横梁" >= 20) AND NOT "Timer".润滑初始化计时器.Q THEN "辅助中继".润滑初始化成功 := TRUE; END_IF;
   IF NOT "润滑电机" THEN "辅助中继".润滑初始化成功 := FALSE; END_IF;
   "润滑电机工作指示" := "润滑电机" AND ("Clock_1Hz" OR "辅助中继".润滑初始化成功);
END_REGION

REGION Network 3: 平衡器润滑
   "辅助中继".平衡器润滑 := "润滑电机" AND NOT "Timer".平衡器润滑持续计时.Q AND NOT "Timer".平衡器润滑间歇计时.Q;
   "Timer".平衡器润滑持续计时.TON(IN := "润滑电机" AND NOT "Timer".平衡器润滑间歇计时.Q, PT := "中间数据".平衡器润滑阀持续时间设定);
   "Timer".平衡器润滑间歇计时.TON(IN := "Timer".平衡器润滑持续计时.Q, PT := "中间数据".平衡器润滑阀间歇时间设定);
   "Timer".平衡器手动延时计时.TOF(IN := "平衡缸手动润滑" OR "气垫手动润滑", PT := "中间数据".平衡器手动延时设定);
   "平衡器间歇润滑阀" := "辅助中继".平衡器润滑 OR "Timer".平衡器手动延时计时.Q;
END_REGION

REGION Network 4: 气垫润滑
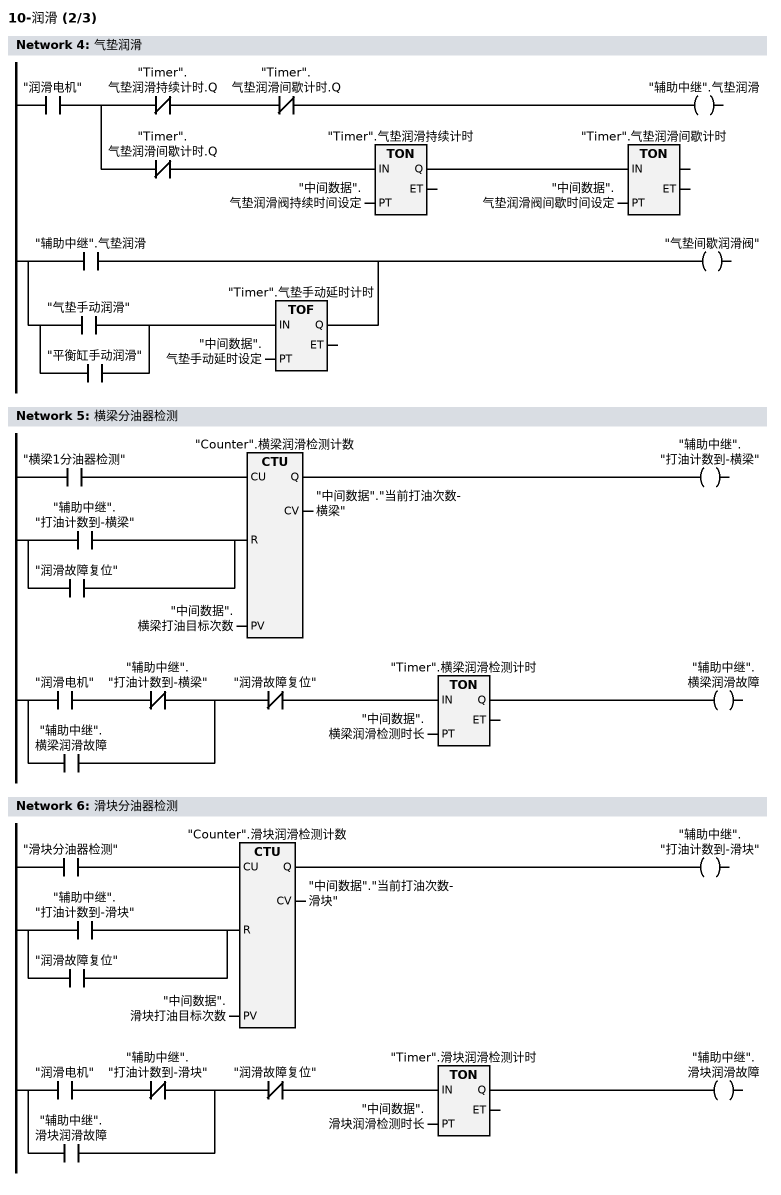
   "辅助中继".气垫润滑 := "润滑电机" AND NOT "Timer".气垫润滑持续计时.Q AND NOT "Timer".气垫润滑间歇计时.Q;
   "Timer".气垫润滑持续计时.TON(IN := "润滑电机" AND NOT "Timer".气垫润滑间歇计时.Q, PT := "中间数据".气垫润滑阀持续时间设定);
   "Timer".气垫润滑间歇计时.TON(IN := "Timer".气垫润滑持续计时.Q, PT := "中间数据".气垫润滑阀间歇时间设定);
   "Timer".气垫手动延时计时.TOF(IN := "气垫手动润滑" OR "平衡缸手动润滑", PT := "中间数据".气垫手动延时设定);
   "气垫间歇润滑阀" := "辅助中继".气垫润滑 OR "Timer".气垫手动延时计时.Q;
END_REGION

REGION Network 5: 横梁分油器检测
   "Counter".横梁润滑检测计数.CTU(CU := "横梁1分油器检测",
                          R := "辅助中继"."打油计数到-横梁" OR "润滑故障复位",
                          PV := "中间数据".横梁打油目标次数,
                          CV => "中间数据"."当前打油次数-横梁");
   "辅助中继"."打油计数到-横梁" := "Counter".横梁润滑检测计数.Q;
   "Timer".横梁润滑检测计时.TON(IN := (("润滑电机" AND NOT "辅助中继"."打油计数到-横梁") OR "辅助中继".横梁润滑故障) AND NOT "润滑故障复位",
                        PT := "中间数据".横梁润滑检测时长);
   "辅助中继".横梁润滑故障 := "Timer".横梁润滑检测计时.Q;
END_REGION

REGION Network 6: 滑块分油器检测
   "Counter".滑块润滑检测计数.CTU(CU := "滑块分油器检测",
                          R := "辅助中继"."打油计数到-滑块" OR "润滑故障复位",
                          PV := "中间数据".滑块打油目标次数,
                          CV => "中间数据"."当前打油次数-滑块");
   "辅助中继"."打油计数到-滑块" := "Counter".滑块润滑检测计数.Q;
   "Timer".滑块润滑检测计时.TON(IN := (("润滑电机" AND NOT "辅助中继"."打油计数到-滑块") OR "辅助中继".滑块润滑故障) AND NOT "润滑故障复位",
                        PT := "中间数据".滑块润滑检测时长);
   "辅助中继".滑块润滑故障 := "Timer".滑块润滑检测计时.Q;
END_REGION

REGION Network 7: 平衡器分油器检测
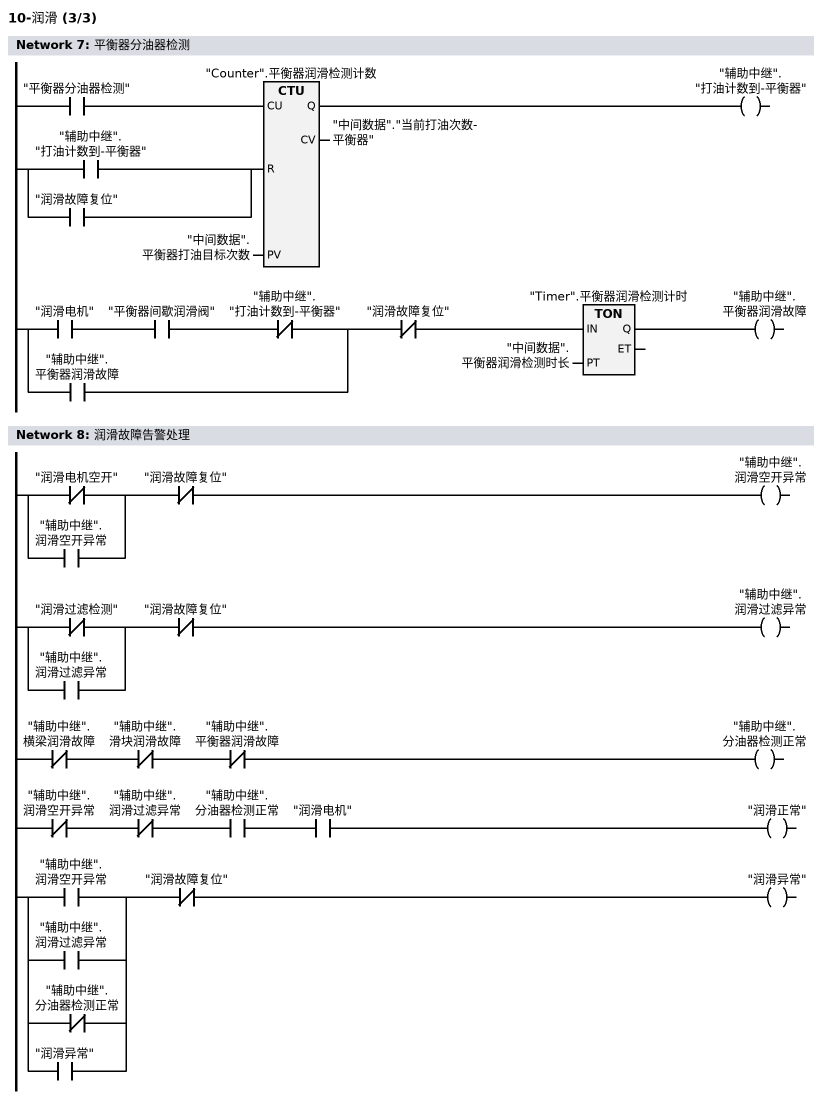
   "Counter".平衡器润滑检测计数.CTU(CU := "平衡器分油器检测",
                           R := "辅助中继"."打油计数到-平衡器" OR "润滑故障复位",
                           PV := "中间数据".平衡器打油目标次数,
                           CV => "中间数据"."当前打油次数-平衡器");
   "辅助中继"."打油计数到-平衡器" := "Counter".平衡器润滑检测计数.Q;
   "Timer".平衡器润滑检测计时.TON(IN := (("润滑电机" AND "平衡器间歇润滑阀" AND NOT "辅助中继"."打油计数到-平衡器") OR "辅助中继".平衡器润滑故障) AND NOT "润滑故障复位",
                         PT := "中间数据".平衡器润滑检测时长);
   "辅助中继".平衡器润滑故障 := "Timer".平衡器润滑检测计时.Q;
END_REGION

REGION Network 8: 润滑故障告警处理
   RUNG wire#powerrail
      I_Contact( "润滑电机空开" )
      wire#w1
      I_Contact( "润滑故障复位" )
      Coil( "辅助中继".润滑空开异常 )
   END_RUNG
   RUNG wire#powerrail
      Contact( "辅助中继".润滑空开异常 )
   END_RUNG wire#w1
   RUNG wire#powerrail
      I_Contact( "润滑过滤检测" )
      wire#w2
      I_Contact( "润滑故障复位" )
      Coil( "辅助中继".润滑过滤异常 )
   END_RUNG
   RUNG wire#powerrail
      Contact( "辅助中继".润滑过滤异常 )
   END_RUNG wire#w2
   RUNG wire#powerrail
      I_Contact( "辅助中继".横梁润滑故障 )
      I_Contact( "辅助中继".滑块润滑故障 )
      I_Contact( "辅助中继".平衡器润滑故障 )
      Coil( "辅助中继".分油器检测正常 )
   END_RUNG
   RUNG wire#powerrail
      I_Contact( "辅助中继".润滑空开异常 )
      I_Contact( "辅助中继".润滑过滤异常 )
      Contact( "辅助中继".分油器检测正常 )
      Contact( "润滑电机" )
      Coil( "润滑正常" )
   END_RUNG
   RUNG wire#powerrail
      Contact( "辅助中继".润滑空开异常 )
      wire#w3
      I_Contact( "润滑故障复位" )
      Coil( "润滑异常" )
   END_RUNG
   RUNG wire#powerrail
      Contact( "辅助中继".润滑过滤异常 )
   END_RUNG wire#w3
   RUNG wire#powerrail
      I_Contact( "辅助中继".分油器检测正常 )
   END_RUNG wire#w3
   RUNG wire#powerrail
      Contact( "润滑异常" )
   END_RUNG wire#w3
   // the same network as SCL:
   "辅助中继".润滑空开异常 := (NOT "润滑电机空开" OR "辅助中继".润滑空开异常) AND NOT "润滑故障复位";
   "辅助中继".润滑过滤异常 := (NOT "润滑过滤检测" OR "辅助中继".润滑过滤异常) AND NOT "润滑故障复位";
   "辅助中继".分油器检测正常 := NOT "辅助中继".横梁润滑故障 AND NOT "辅助中继".滑块润滑故障 AND NOT "辅助中继".平衡器润滑故障;
   "润滑正常" := NOT "辅助中继".润滑空开异常 AND NOT "辅助中继".润滑过滤异常 AND "辅助中继".分油器检测正常 AND "润滑电机";
   "润滑异常" := ("辅助中继".润滑空开异常 OR "辅助中继".润滑过滤异常 OR NOT "辅助中继".分油器检测正常 OR "润滑异常") AND NOT "润滑故障复位";
END_REGION
END_FUNCTION

FUNCTION "移动工作台" : Void   // FC4, LAD
{ S7_Optimized_Access := 'TRUE' }
VERSION : 0.1
BEGIN

REGION Network 1
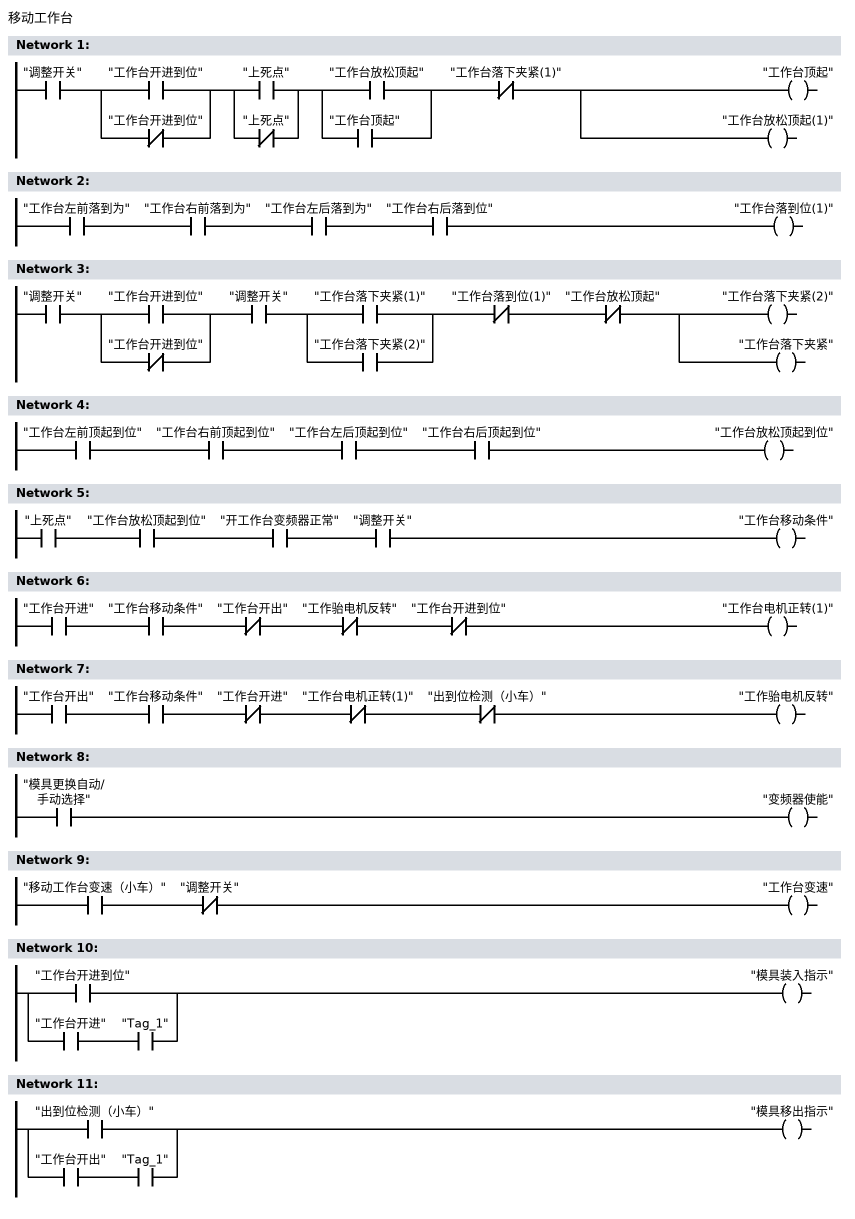
   RUNG wire#powerrail
      Contact( "调整开关" )
      wire#w1
      Contact( "工作台开进到位" )
      wire#w2
      Contact( "上死点" )
      wire#w3
      Contact( "工作台放松顶起" )
      wire#w4
      I_Contact( "工作台落下夹紧(1)" )
      wire#w5
      Coil( "工作台顶起" )
   END_RUNG
   RUNG wire#w1
      I_Contact( "工作台开进到位" )
   END_RUNG wire#w2
   RUNG wire#w2
      I_Contact( "上死点" )
   END_RUNG wire#w3
   RUNG wire#w3
      Contact( "工作台顶起" )
   END_RUNG wire#w4
   RUNG wire#w5
      Coil( "工作台放松顶起(1)" )
   END_RUNG
   // the same network as SCL:
   "工作台顶起" := "调整开关" AND ("工作台开进到位" OR NOT "工作台开进到位") AND ("上死点" OR NOT "上死点") AND ("工作台放松顶起" OR "工作台顶起") AND NOT "工作台落下夹紧(1)";
   "工作台放松顶起(1)" := "工作台顶起";
END_REGION

REGION Network 2
   RUNG wire#powerrail
      Contact( "工作台左前落到为" )
      Contact( "工作台右前落到为" )
      Contact( "工作台左后落到为" )
      Contact( "工作台右后落到位" )
      Coil( "工作台落到位(1)" )
   END_RUNG
   // the same network as SCL:
   "工作台落到位(1)" := "工作台左前落到为" AND "工作台右前落到为" AND "工作台左后落到为" AND "工作台右后落到位";
END_REGION

REGION Network 3
   RUNG wire#powerrail
      Contact( "调整开关" )
      wire#w1
      Contact( "工作台开进到位" )
      wire#w2
      Contact( "调整开关" )
      wire#w3
      Contact( "工作台落下夹紧(1)" )
      wire#w4
      I_Contact( "工作台落到位(1)" )
      I_Contact( "工作台放松顶起" )
      wire#w5
      Coil( "工作台落下夹紧(2)" )
   END_RUNG
   RUNG wire#w1
      I_Contact( "工作台开进到位" )
   END_RUNG wire#w2
   RUNG wire#w3
      Contact( "工作台落下夹紧(2)" )
   END_RUNG wire#w4
   RUNG wire#w5
      Coil( "工作台落下夹紧" )
   END_RUNG
   // the same network as SCL:
   "工作台落下夹紧(2)" := "调整开关" AND ("工作台开进到位" OR NOT "工作台开进到位") AND "调整开关" AND ("工作台落下夹紧(1)" OR "工作台落下夹紧(2)") AND NOT "工作台落到位(1)" AND NOT "工作台放松顶起";
   "工作台落下夹紧" := "工作台落下夹紧(2)";
END_REGION

REGION Network 4
   RUNG wire#powerrail
      Contact( "工作台左前顶起到位" )
      Contact( "工作台右前顶起到位" )
      Contact( "工作台左后顶起到位" )
      Contact( "工作台右后顶起到位" )
      Coil( "工作台放松顶起到位" )
   END_RUNG
   // the same network as SCL:
   "工作台放松顶起到位" := "工作台左前顶起到位" AND "工作台右前顶起到位" AND "工作台左后顶起到位" AND "工作台右后顶起到位";
END_REGION

REGION Network 5
   RUNG wire#powerrail
      Contact( "上死点" )
      Contact( "工作台放松顶起到位" )
      Contact( "开工作台变频器正常" )
      Contact( "调整开关" )
      Coil( "工作台移动条件" )
   END_RUNG
   // the same network as SCL:
   "工作台移动条件" := "上死点" AND "工作台放松顶起到位" AND "开工作台变频器正常" AND "调整开关";
END_REGION

REGION Network 6
   RUNG wire#powerrail
      Contact( "工作台开进" )
      Contact( "工作台移动条件" )
      I_Contact( "工作台开出" )
      I_Contact( "工作骀电机反转" )
      I_Contact( "工作台开进到位" )
      Coil( "工作台电机正转(1)" )
   END_RUNG
   // the same network as SCL:
   "工作台电机正转(1)" := "工作台开进" AND "工作台移动条件" AND NOT "工作台开出" AND NOT "工作骀电机反转" AND NOT "工作台开进到位";
END_REGION

REGION Network 7
   RUNG wire#powerrail
      Contact( "工作台开出" )
      Contact( "工作台移动条件" )
      I_Contact( "工作台开进" )
      I_Contact( "工作台电机正转(1)" )
      I_Contact( "出到位检测（小车）" )
      Coil( "工作骀电机反转" )
   END_RUNG
   // the same network as SCL:
   "工作骀电机反转" := "工作台开出" AND "工作台移动条件" AND NOT "工作台开进" AND NOT "工作台电机正转(1)" AND NOT "出到位检测（小车）";
END_REGION

REGION Network 8
   RUNG wire#powerrail
      Contact( "模具更换自动/手动选择" )
      Coil( "变频器使能" )
   END_RUNG
   // the same network as SCL:
   "变频器使能" := "模具更换自动/手动选择";
END_REGION

REGION Network 9
   RUNG wire#powerrail
      Contact( "移动工作台变速（小车）" )
      I_Contact( "调整开关" )
      Coil( "工作台变速" )
   END_RUNG
   // the same network as SCL:
   "工作台变速" := "移动工作台变速（小车）" AND NOT "调整开关";
END_REGION

REGION Network 10
   RUNG wire#powerrail
      Contact( "工作台开进到位" )
      wire#w1
      Coil( "模具装入指示" )
   END_RUNG
   RUNG wire#powerrail
      Contact( "工作台开进" )
      Contact( "Tag_1" )
   END_RUNG wire#w1
   // the same network as SCL:
   "模具装入指示" := "工作台开进到位" OR ("工作台开进" AND "Tag_1");
END_REGION

REGION Network 11
   RUNG wire#powerrail
      Contact( "出到位检测（小车）" )
      wire#w1
      Coil( "模具移出指示" )
   END_RUNG
   RUNG wire#powerrail
      Contact( "工作台开出" )
      Contact( "Tag_1" )
   END_RUNG wire#w1
   // the same network as SCL:
   "模具移出指示" := "出到位检测（小车）" OR ("工作台开出" AND "Tag_1");
END_REGION
END_FUNCTION

FUNCTION "液压保护平衡器" : Void   // FC5, LAD
{ S7_Optimized_Access := 'TRUE' }
VERSION : 0.1
BEGIN

REGION Network 1
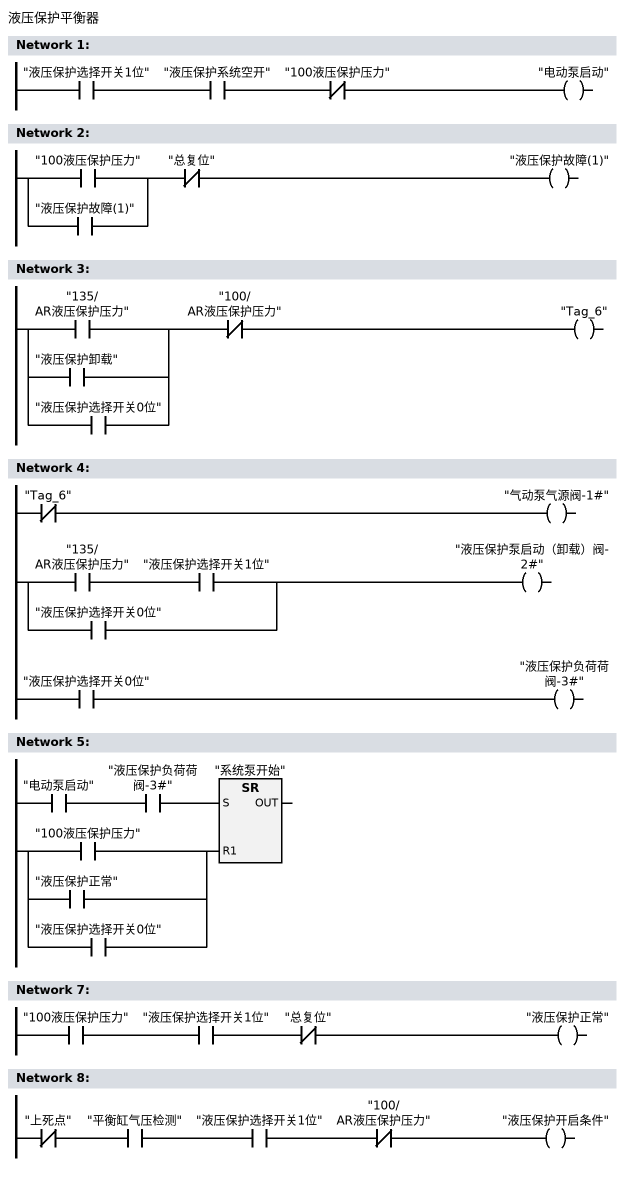
   RUNG wire#powerrail
      Contact( "液压保护选择开关1位" )
      Contact( "液压保护系统空开" )
      I_Contact( "100液压保护压力" )
      Coil( "电动泵启动" )
   END_RUNG
   // the same network as SCL:
   "电动泵启动" := "液压保护选择开关1位" AND "液压保护系统空开" AND NOT "100液压保护压力";
END_REGION

REGION Network 2
   RUNG wire#powerrail
      Contact( "100液压保护压力" )
      wire#w1
      I_Contact( "总复位" )
      Coil( "液压保护故障(1)" )
   END_RUNG
   RUNG wire#powerrail
      Contact( "液压保护故障(1)" )
   END_RUNG wire#w1
   // the same network as SCL:
   "液压保护故障(1)" := ("100液压保护压力" OR "液压保护故障(1)") AND NOT "总复位";
END_REGION

REGION Network 3
   RUNG wire#powerrail
      Contact( "135/AR液压保护压力" )
      wire#w1
      I_Contact( "100/AR液压保护压力" )
      Coil( "Tag_6" )
   END_RUNG
   RUNG wire#powerrail
      Contact( "液压保护卸载" )
   END_RUNG wire#w1
   RUNG wire#powerrail
      Contact( "液压保护选择开关0位" )
   END_RUNG wire#w1
   // the same network as SCL:
   "Tag_6" := ("135/AR液压保护压力" OR "液压保护卸载" OR "液压保护选择开关0位") AND NOT "100/AR液压保护压力";
END_REGION

REGION Network 4
   RUNG wire#powerrail
      I_Contact( "Tag_6" )
      Coil( "气动泵气源阀-1#" )
   END_RUNG
   RUNG wire#powerrail
      Contact( "135/AR液压保护压力" )
      Contact( "液压保护选择开关1位" )
      wire#w1
      Coil( "液压保护泵启动（卸载）阀-2#" )
   END_RUNG
   RUNG wire#powerrail
      Contact( "液压保护选择开关0位" )
   END_RUNG wire#w1
   RUNG wire#powerrail
      Contact( "液压保护选择开关0位" )
      Coil( "液压保护负荷荷 阀-3#" )
   END_RUNG
   // the same network as SCL:
   "气动泵气源阀-1#" := NOT "Tag_6";
   "液压保护泵启动（卸载）阀-2#" := ("135/AR液压保护压力" AND "液压保护选择开关1位") OR "液压保护选择开关0位";
   "液压保护负荷荷 阀-3#" := "液压保护选择开关0位";
END_REGION

REGION Network 5
   RUNG wire#powerrail
      Contact( "电动泵启动" )
      Contact( "液压保护负荷荷 阀-3#" )
      S_SR(operand := "系统泵开始", r1 := wire#w1)
   END_RUNG
   RUNG wire#powerrail
      Contact( "100液压保护压力" )
   END_RUNG wire#w1
   RUNG wire#powerrail
      Contact( "液压保护正常" )
   END_RUNG wire#w1
   RUNG wire#powerrail
      Contact( "液压保护选择开关0位" )
   END_RUNG wire#w1
   // the same network as SCL:
   IF "电动泵启动" AND "液压保护负荷荷 阀-3#" THEN
       "系统泵开始" := TRUE;   // SR flip-flop
   END_IF;
   IF "100液压保护压力" OR "液压保护正常" OR "液压保护选择开关0位" THEN "系统泵开始" := FALSE; END_IF;
END_REGION

REGION Network 7
   RUNG wire#powerrail
      Contact( "100液压保护压力" )
      Contact( "液压保护选择开关1位" )
      I_Contact( "总复位" )
      Coil( "液压保护正常" )
   END_RUNG
   // the same network as SCL:
   "液压保护正常" := "100液压保护压力" AND "液压保护选择开关1位" AND NOT "总复位";
END_REGION

REGION Network 8
   RUNG wire#powerrail
      I_Contact( "上死点" )
      Contact( "平衡缸气压检测" )
      Contact( "液压保护选择开关1位" )
      I_Contact( "100/AR液压保护压力" )
      Coil( "液压保护开启条件" )
   END_RUNG
   // the same network as SCL:
   "液压保护开启条件" := NOT "上死点" AND "平衡缸气压检测" AND "液压保护选择开关1位" AND NOT "100/AR液压保护压力";
END_REGION
END_FUNCTION

FUNCTION "主电机" : Void   // FC6, LAD
{ S7_Optimized_Access := 'TRUE' }
VERSION : 0.1
BEGIN

REGION Network 1
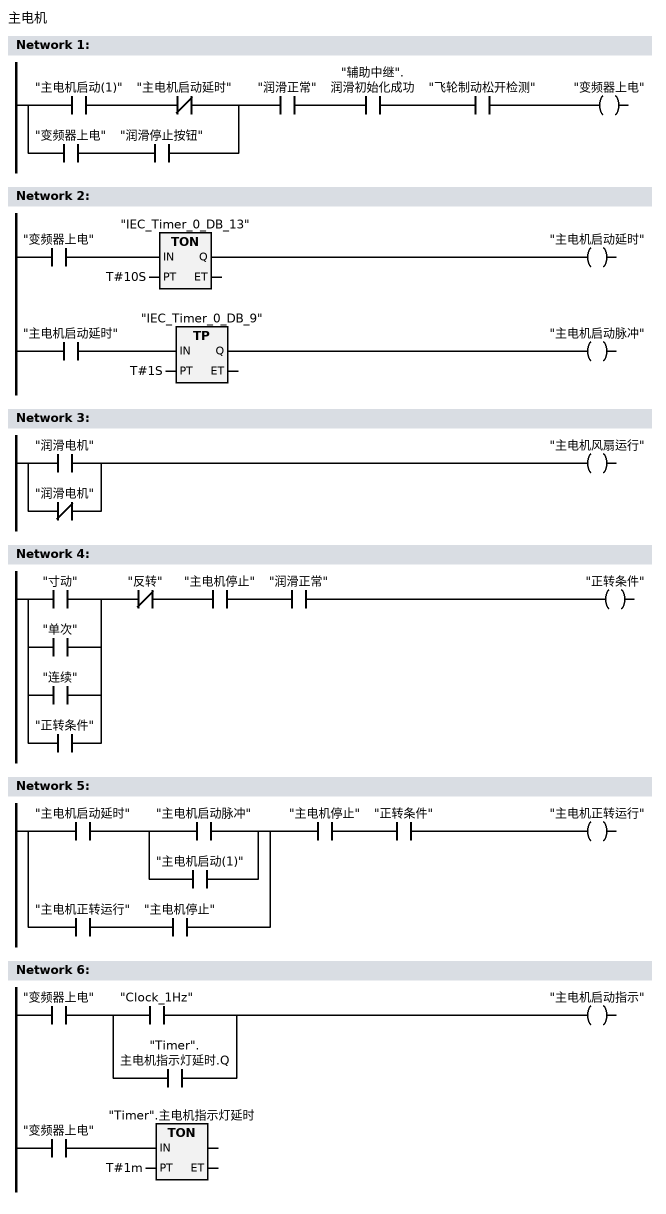
   RUNG wire#powerrail
      Contact( "主电机启动(1)" )
      I_Contact( "主电机启动延时" )
      wire#w1
      Contact( "润滑正常" )
      Contact( "辅助中继".润滑初始化成功 )
      Contact( "飞轮制动松开检测" )
      Coil( "变频器上电" )
   END_RUNG
   RUNG wire#powerrail
      Contact( "变频器上电" )
      Contact( "润滑停止按钮" )
   END_RUNG wire#w1
   // the same network as SCL:
   "变频器上电" := (("主电机启动(1)" AND NOT "主电机启动延时") OR ("变频器上电" AND "润滑停止按钮")) AND "润滑正常" AND "辅助中继".润滑初始化成功 AND "飞轮制动松开检测";
END_REGION

REGION Network 2
   "IEC_Timer_0_DB_13".TON(IN := "变频器上电", PT := T#10S);
   "主电机启动延时" := "IEC_Timer_0_DB_13".Q;
   "IEC_Timer_0_DB_9".TP(IN := "主电机启动延时", PT := T#1S);
   "主电机启动脉冲" := "IEC_Timer_0_DB_9".Q;
END_REGION

REGION Network 3
   RUNG wire#powerrail
      Contact( "润滑电机" )
      wire#w1
      Coil( "主电机风扇运行" )
   END_RUNG
   RUNG wire#powerrail
      I_Contact( "润滑电机" )
   END_RUNG wire#w1
   // the same network as SCL:
   "主电机风扇运行" := "润滑电机" OR NOT "润滑电机";
END_REGION

REGION Network 4
   RUNG wire#powerrail
      Contact( "寸动" )
      wire#w1
      I_Contact( "反转" )
      Contact( "主电机停止" )
      Contact( "润滑正常" )
      Coil( "正转条件" )
   END_RUNG
   RUNG wire#powerrail
      Contact( "单次" )
   END_RUNG wire#w1
   RUNG wire#powerrail
      Contact( "连续" )
   END_RUNG wire#w1
   RUNG wire#powerrail
      Contact( "正转条件" )
   END_RUNG wire#w1
   // the same network as SCL:
   "正转条件" := ("寸动" OR "单次" OR "连续" OR "正转条件") AND NOT "反转" AND "主电机停止" AND "润滑正常";
END_REGION

REGION Network 5
   RUNG wire#powerrail
      Contact( "主电机启动延时" )
      wire#w1
      Contact( "主电机启动脉冲" )
      wire#w2
      Contact( "主电机停止" )
      Contact( "正转条件" )
      Coil( "主电机正转运行" )
   END_RUNG
   RUNG wire#w1
      Contact( "主电机启动(1)" )
   END_RUNG wire#w2
   RUNG wire#powerrail
      Contact( "主电机正转运行" )
      Contact( "主电机停止" )
   END_RUNG wire#w2
   // the same network as SCL:
   "主电机正转运行" := (("主电机启动延时" AND ("主电机启动脉冲" OR "主电机启动(1)")) OR ("主电机正转运行" AND "主电机停止")) AND "主电机停止" AND "正转条件";
END_REGION

REGION Network 6
   "主电机启动指示" := "变频器上电" AND ("Clock_1Hz" OR "Timer".主电机指示灯延时.Q);
   "Timer".主电机指示灯延时.TON(IN := "变频器上电", PT := T#1m);
END_REGION
END_FUNCTION

FUNCTION "滑块调整" : Void   // FC7, LAD
{ S7_Optimized_Access := 'TRUE' }
VERSION : 0.1
BEGIN

REGION Network 1
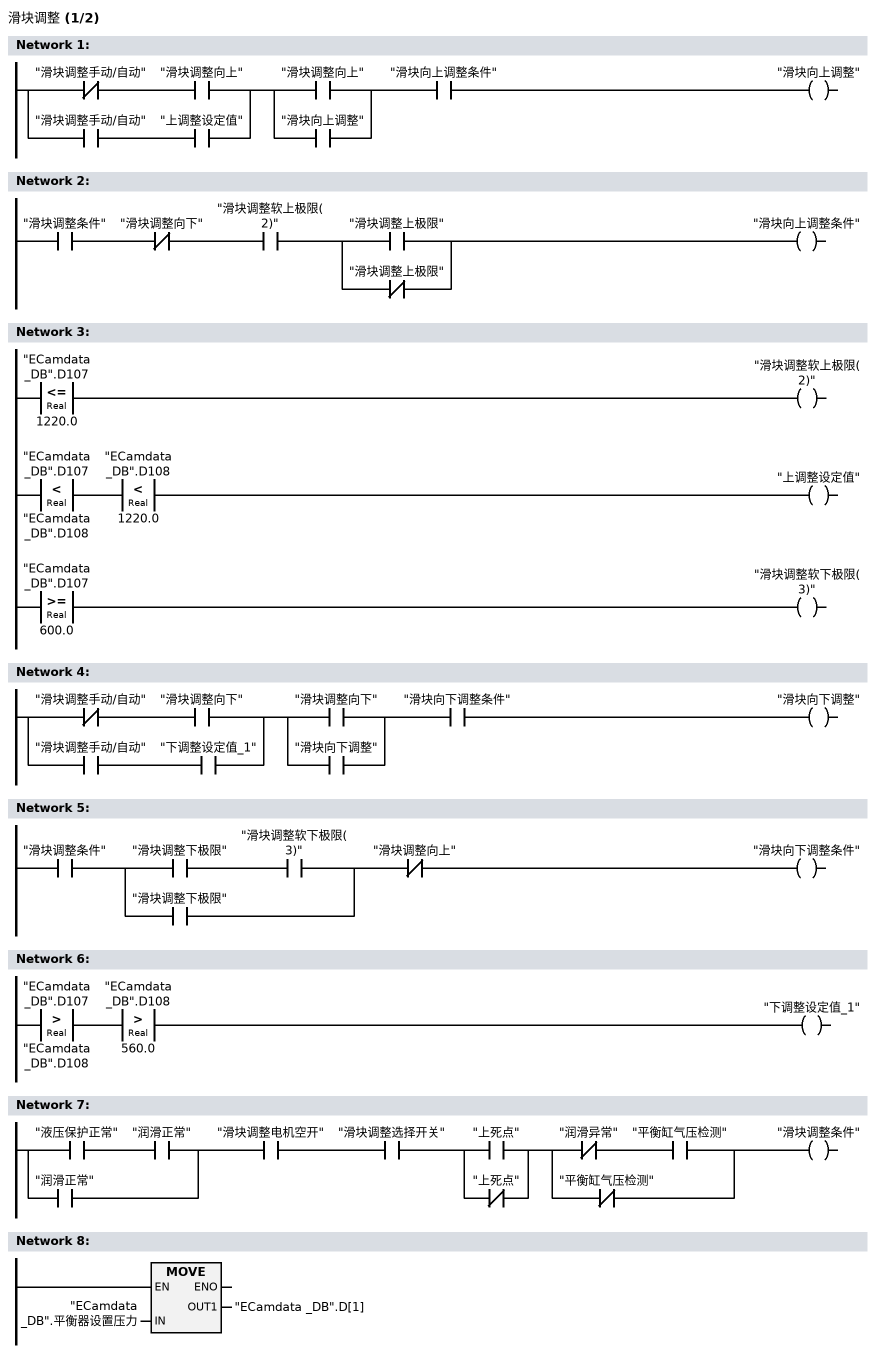
   RUNG wire#powerrail
      I_Contact( "滑块调整手动/自动" )
      Contact( "滑块调整向上" )
      wire#w1
      Contact( "滑块调整向上" )
      wire#w2
      Contact( "滑块向上调整条件" )
      Coil( "滑块向上调整" )
   END_RUNG
   RUNG wire#powerrail
      Contact( "滑块调整手动/自动" )
      Contact( "上调整设定值" )
   END_RUNG wire#w1
   RUNG wire#w1
      Contact( "滑块向上调整" )
   END_RUNG wire#w2
   // the same network as SCL:
   "滑块向上调整" := ((NOT "滑块调整手动/自动" AND "滑块调整向上") OR ("滑块调整手动/自动" AND "上调整设定值")) AND ("滑块调整向上" OR "滑块向上调整") AND "滑块向上调整条件";
END_REGION

REGION Network 2
   RUNG wire#powerrail
      Contact( "滑块调整条件" )
      I_Contact( "滑块调整向下" )
      Contact( "滑块调整软上极限(2)" )
      wire#w1
      Contact( "滑块调整上极限" )
      wire#w2
      Coil( "滑块向上调整条件" )
   END_RUNG
   RUNG wire#w1
      I_Contact( "滑块调整上极限" )
   END_RUNG wire#w2
   // the same network as SCL:
   "滑块向上调整条件" := "滑块调整条件" AND NOT "滑块调整向下" AND "滑块调整软上极限(2)" AND ("滑块调整上极限" OR NOT "滑块调整上极限");
END_REGION

REGION Network 3
   RUNG wire#powerrail
      { S7_Templates := "SrcType := Real" } LE_Contact(in1 := "ECamdata _DB".D107, in2 := 1220.0)
      Coil( "滑块调整软上极限(2)" )
   END_RUNG
   RUNG wire#powerrail
      { S7_Templates := "SrcType := Real" } LT_Contact(in1 := "ECamdata _DB".D107, in2 := "ECamdata _DB".D108)
      { S7_Templates := "SrcType := Real" } LT_Contact(in1 := "ECamdata _DB".D108, in2 := 1220.0)
      Coil( "上调整设定值" )
   END_RUNG
   RUNG wire#powerrail
      { S7_Templates := "SrcType := Real" } GE_Contact(in1 := "ECamdata _DB".D107, in2 := 600.0)
      Coil( "滑块调整软下极限(3)" )
   END_RUNG
   // the same network as SCL:
   "滑块调整软上极限(2)" := "ECamdata _DB".D107 <= 1220.0;
   "上调整设定值" := ("ECamdata _DB".D107 < "ECamdata _DB".D108) AND ("ECamdata _DB".D108 < 1220.0);
   "滑块调整软下极限(3)" := "ECamdata _DB".D107 >= 600.0;
END_REGION

REGION Network 4
   RUNG wire#powerrail
      I_Contact( "滑块调整手动/自动" )
      Contact( "滑块调整向下" )
      wire#w1
      Contact( "滑块调整向下" )
      wire#w2
      Contact( "滑块向下调整条件" )
      Coil( "滑块向下调整" )
   END_RUNG
   RUNG wire#powerrail
      Contact( "滑块调整手动/自动" )
      Contact( "下调整设定值_1" )
   END_RUNG wire#w1
   RUNG wire#w1
      Contact( "滑块向下调整" )
   END_RUNG wire#w2
   // the same network as SCL:
   "滑块向下调整" := ((NOT "滑块调整手动/自动" AND "滑块调整向下") OR ("滑块调整手动/自动" AND "下调整设定值_1")) AND ("滑块调整向下" OR "滑块向下调整") AND "滑块向下调整条件";
END_REGION

REGION Network 5
   RUNG wire#powerrail
      Contact( "滑块调整条件" )
      wire#w1
      Contact( "滑块调整下极限" )
      Contact( "滑块调整软下极限(3)" )
      wire#w2
      I_Contact( "滑块调整向上" )
      Coil( "滑块向下调整条件" )
   END_RUNG
   RUNG wire#w1
      Contact( "滑块调整下极限" )
   END_RUNG wire#w2
   // the same network as SCL:
   "滑块向下调整条件" := "滑块调整条件" AND (("滑块调整下极限" AND "滑块调整软下极限(3)") OR "滑块调整下极限") AND NOT "滑块调整向上";
END_REGION

REGION Network 6
   RUNG wire#powerrail
      { S7_Templates := "SrcType := Real" } GT_Contact(in1 := "ECamdata _DB".D107, in2 := "ECamdata _DB".D108)
      { S7_Templates := "SrcType := Real" } GT_Contact(in1 := "ECamdata _DB".D108, in2 := 560.0)
      Coil( "下调整设定值_1" )
   END_RUNG
   // the same network as SCL:
   "下调整设定值_1" := ("ECamdata _DB".D107 > "ECamdata _DB".D108) AND ("ECamdata _DB".D108 > 560.0);
END_REGION

REGION Network 7
   RUNG wire#powerrail
      Contact( "液压保护正常" )
      Contact( "润滑正常" )
      wire#w1
      Contact( "滑块调整电机空开" )
      Contact( "滑块调整选择开关" )
      wire#w2
      Contact( "上死点" )
      wire#w3
      I_Contact( "润滑异常" )
      Contact( "平衡缸气压检测" )
      wire#w4
      Coil( "滑块调整条件" )
   END_RUNG
   RUNG wire#powerrail
      Contact( "润滑正常" )
   END_RUNG wire#w1
   RUNG wire#w2
      I_Contact( "上死点" )
   END_RUNG wire#w3
   RUNG wire#w3
      I_Contact( "平衡缸气压检测" )
   END_RUNG wire#w4
   // the same network as SCL:
   "滑块调整条件" := (("液压保护正常" AND "润滑正常") OR "润滑正常") AND "滑块调整电机空开" AND "滑块调整选择开关" AND ("上死点" OR NOT "上死点") AND ((NOT "润滑异常" AND "平衡缸气压检测") OR NOT "平衡缸气压检测");
END_REGION

REGION Network 8
   RUNG wire#powerrail
      Move(in := "ECamdata _DB".平衡器设置压力, out1 => "ECamdata _DB".D[1])
   END_RUNG
   // the same network as SCL:
   "ECamdata _DB".D[1] := "ECamdata _DB".平衡器设置压力;
END_REGION

REGION Network 9
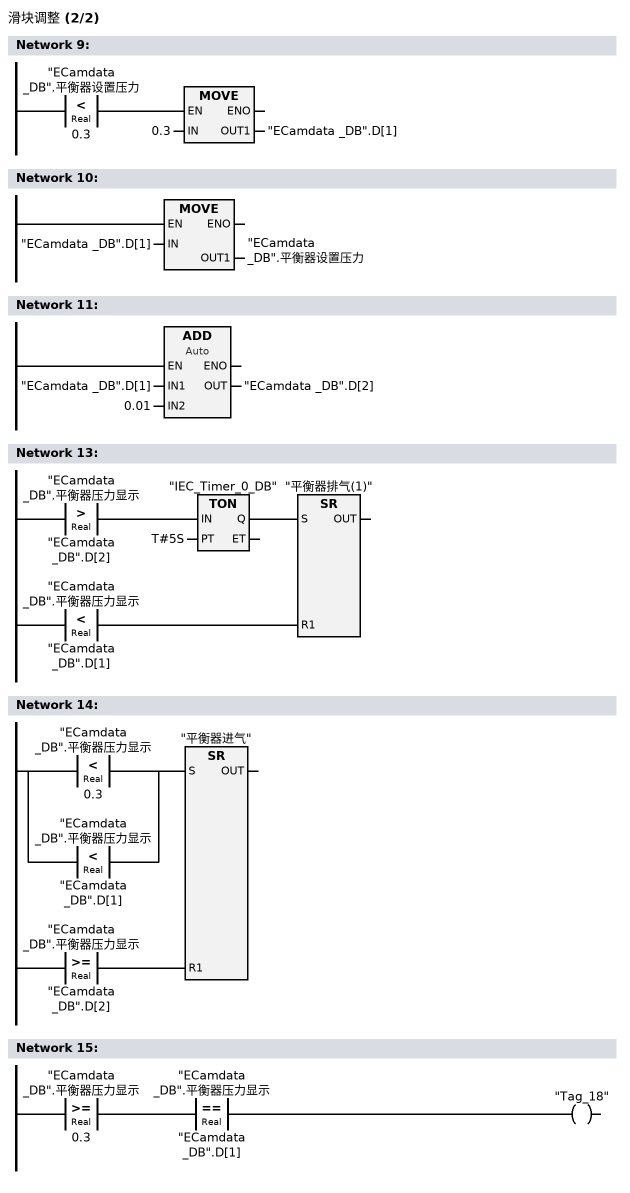
   RUNG wire#powerrail
      { S7_Templates := "SrcType := Real" } LT_Contact(in1 := "ECamdata _DB".平衡器设置压力, in2 := 0.3)
      Move(in := 0.3, out1 => "ECamdata _DB".D[1])
   END_RUNG
   // the same network as SCL:
   IF "ECamdata _DB".平衡器设置压力 < 0.3 THEN "ECamdata _DB".D[1] := 0.3; END_IF;
END_REGION

REGION Network 10
   RUNG wire#powerrail
      Move(in := "ECamdata _DB".D[1], out1 => "ECamdata _DB".平衡器设置压力)
   END_RUNG
   // the same network as SCL:
   "ECamdata _DB".平衡器设置压力 := "ECamdata _DB".D[1];
END_REGION

REGION Network 11
   RUNG wire#powerrail
      Add(in1 := "ECamdata _DB".D[1], in2 := 0.01, out => "ECamdata _DB".D[2])
   END_RUNG
   // the same network as SCL:
   "ECamdata _DB".D[2] := "ECamdata _DB".D[1] + 0.01;
END_REGION

REGION Network 13
   "IEC_Timer_0_DB".TON(IN := "ECamdata _DB".平衡器压力显示 > "ECamdata _DB".D[2], PT := T#5S);
   IF "IEC_Timer_0_DB".Q THEN
       "平衡器排气(1)" := TRUE;   // SR flip-flop
   END_IF;
   IF "ECamdata _DB".平衡器压力显示 < "ECamdata _DB".D[1] THEN "平衡器排气(1)" := FALSE; END_IF;
END_REGION

REGION Network 14
   RUNG wire#powerrail
      { S7_Templates := "SrcType := Real" } LT_Contact(in1 := "ECamdata _DB".平衡器压力显示, in2 := 0.3)
      wire#w1
      S_SR(operand := "平衡器进气", r1 := wire#w2)
   END_RUNG
   RUNG wire#powerrail
      { S7_Templates := "SrcType := Real" } LT_Contact(in1 := "ECamdata _DB".平衡器压力显示, in2 := "ECamdata _DB".D[1])
   END_RUNG wire#w1
   RUNG wire#powerrail
      { S7_Templates := "SrcType := Real" } GE_Contact(in1 := "ECamdata _DB".平衡器压力显示, in2 := "ECamdata _DB".D[2])
   END_RUNG wire#w2
   // the same network as SCL:
   IF ("ECamdata _DB".平衡器压力显示 < 0.3) OR ("ECamdata _DB".平衡器压力显示 < "ECamdata _DB".D[1]) THEN
       "平衡器进气" := TRUE;   // SR flip-flop
   END_IF;
   IF "ECamdata _DB".平衡器压力显示 >= "ECamdata _DB".D[2] THEN "平衡器进气" := FALSE; END_IF;
END_REGION

REGION Network 15
   RUNG wire#powerrail
      { S7_Templates := "SrcType := Real" } GE_Contact(in1 := "ECamdata _DB".平衡器压力显示, in2 := 0.3)
      { S7_Templates := "SrcType := Real" } EQ_Contact(in1 := "ECamdata _DB".平衡器压力显示, in2 := "ECamdata _DB".D[1])
      Coil( "Tag_18" )
   END_RUNG
   // the same network as SCL:
   "Tag_18" := ("ECamdata _DB".平衡器压力显示 >= 0.3) AND ("ECamdata _DB".平衡器压力显示 = "ECamdata _DB".D[1]);
END_REGION
END_FUNCTION

FUNCTION "产品计数" : Void   // FC8, LAD
{ S7_Optimized_Access := 'TRUE' }
VERSION : 0.1
   VAR_TEMP
      气垫位置 : DB_ANY;
   END_VAR
BEGIN

REGION Network 1
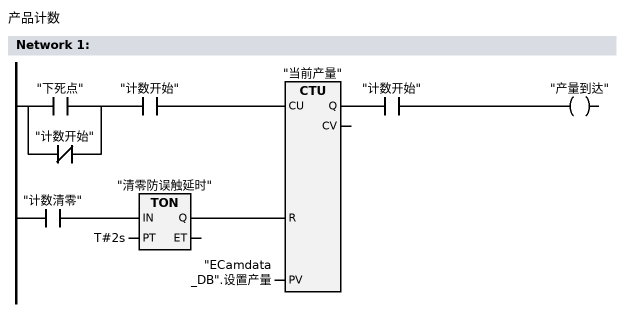
   "清零防误触延时".TON(IN := "计数清零", PT := T#2s);
   "当前产量".CTU(CU := ("下死点" OR NOT "计数开始") AND "计数开始", R := "清零防误触延时".Q, PV := "ECamdata _DB".设置产量);
   "产量到达" := "当前产量".Q AND "计数开始";
END_REGION
END_FUNCTION

FUNCTION "滑块编码器调制" : Void   // FC9, LAD
{ S7_Optimized_Access := 'TRUE' }
VERSION : 0.1
// 滑块编码器
   VAR_TEMP
      D102 : Real;
      D103 : Real;
   END_VAR
BEGIN

REGION Network 1
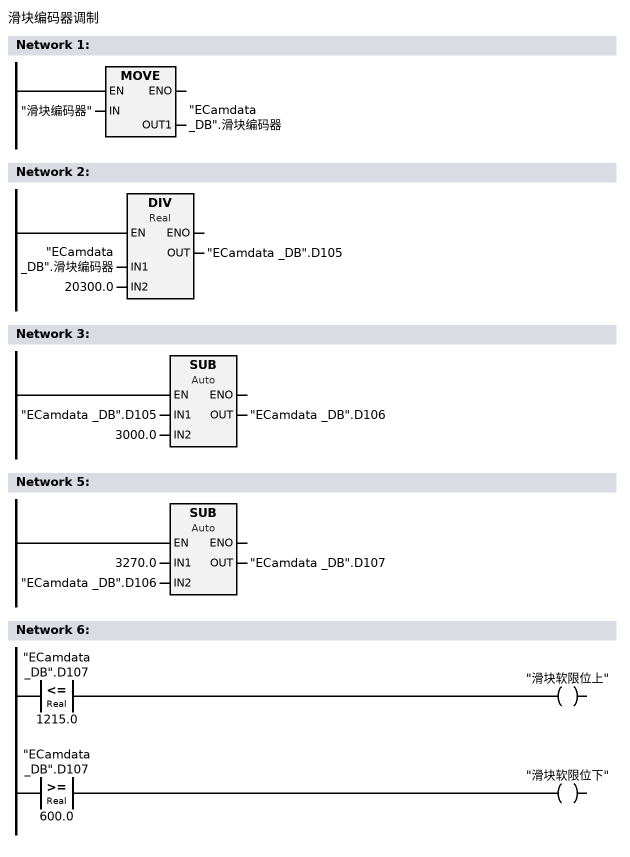
   RUNG wire#powerrail
      Move(in := "滑块编码器", out1 => "ECamdata _DB".滑块编码器)
   END_RUNG
   // the same network as SCL:
   "ECamdata _DB".滑块编码器 := "滑块编码器";
END_REGION

REGION Network 2
   RUNG wire#powerrail
      { S7_Templates := "SrcType := Real" } Div(in1 := "ECamdata _DB".滑块编码器, in2 := 20300.0, out => "ECamdata _DB".D105)
   END_RUNG
   // the same network as SCL:
   "ECamdata _DB".D105 := "ECamdata _DB".滑块编码器 / 20300.0;
END_REGION

REGION Network 3
   RUNG wire#powerrail
      Sub(in1 := "ECamdata _DB".D105, in2 := 3000.0, out => "ECamdata _DB".D106)
   END_RUNG
   // the same network as SCL:
   "ECamdata _DB".D106 := "ECamdata _DB".D105 - 3000.0;
END_REGION

REGION Network 5
   RUNG wire#powerrail
      Sub(in1 := 3270.0, in2 := "ECamdata _DB".D106, out => "ECamdata _DB".D107)
   END_RUNG
   // the same network as SCL:
   "ECamdata _DB".D107 := 3270.0 - "ECamdata _DB".D106;
END_REGION

REGION Network 6
   RUNG wire#powerrail
      { S7_Templates := "SrcType := Real" } LE_Contact(in1 := "ECamdata _DB".D107, in2 := 1215.0)
      Coil( "滑块软限位上" )
   END_RUNG
   RUNG wire#powerrail
      { S7_Templates := "SrcType := Real" } GE_Contact(in1 := "ECamdata _DB".D107, in2 := 600.0)
      Coil( "滑块软限位下" )
   END_RUNG
   // the same network as SCL:
   "滑块软限位上" := "ECamdata _DB".D107 <= 1215.0;
   "滑块软限位下" := "ECamdata _DB".D107 >= 600.0;
END_REGION
END_FUNCTION

FUNCTION "安全" : Void   // FC10, LAD
{ S7_Optimized_Access := 'TRUE' }
VERSION : 0.1
   VAR_TEMP
      压机故障2 : Bool;
   END_VAR
BEGIN

REGION Network 1
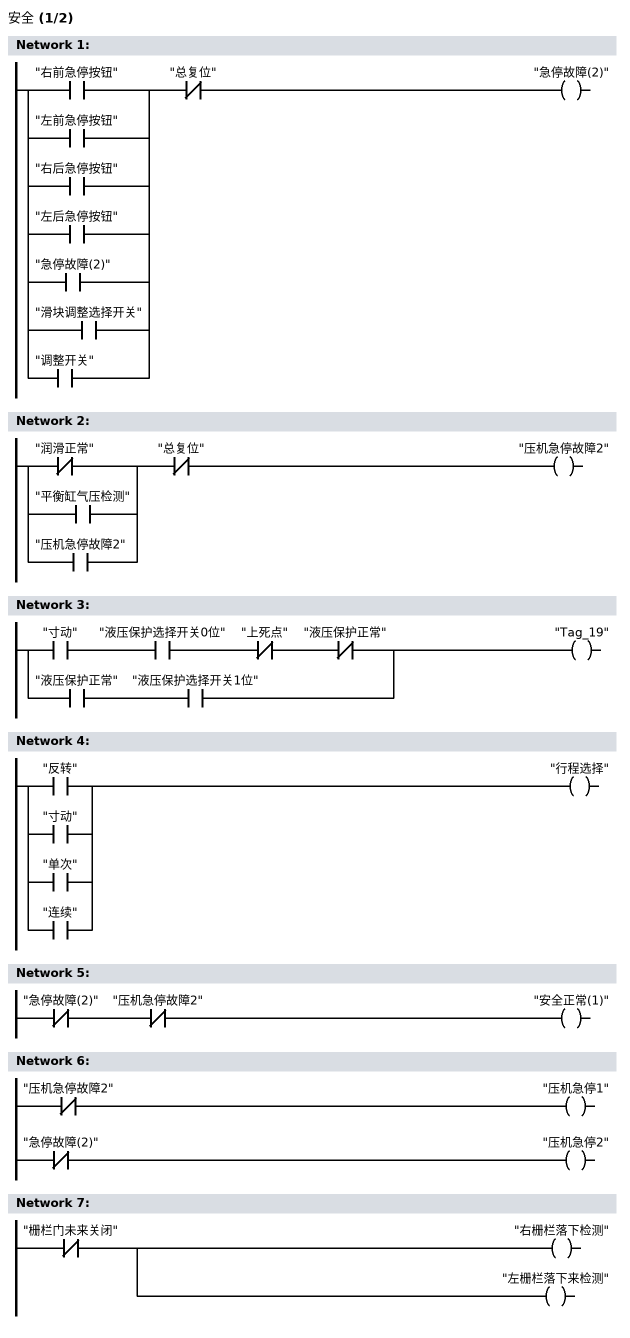
   RUNG wire#powerrail
      Contact( "右前急停按钮" )
      wire#w1
      I_Contact( "总复位" )
      Coil( "急停故障(2)" )
   END_RUNG
   RUNG wire#powerrail
      Contact( "左前急停按钮" )
   END_RUNG wire#w1
   RUNG wire#powerrail
      Contact( "右后急停按钮" )
   END_RUNG wire#w1
   RUNG wire#powerrail
      Contact( "左后急停按钮" )
   END_RUNG wire#w1
   RUNG wire#powerrail
      Contact( "急停故障(2)" )
   END_RUNG wire#w1
   RUNG wire#powerrail
      Contact( "滑块调整选择开关" )
   END_RUNG wire#w1
   RUNG wire#powerrail
      Contact( "调整开关" )
   END_RUNG wire#w1
   // the same network as SCL:
   "急停故障(2)" := ("右前急停按钮" OR "左前急停按钮" OR "右后急停按钮" OR "左后急停按钮" OR "急停故障(2)" OR "滑块调整选择开关" OR "调整开关") AND NOT "总复位";
END_REGION

REGION Network 2
   RUNG wire#powerrail
      I_Contact( "润滑正常" )
      wire#w1
      I_Contact( "总复位" )
      Coil( "压机急停故障2" )
   END_RUNG
   RUNG wire#powerrail
      Contact( "平衡缸气压检测" )
   END_RUNG wire#w1
   RUNG wire#powerrail
      Contact( "压机急停故障2" )
   END_RUNG wire#w1
   // the same network as SCL:
   "压机急停故障2" := (NOT "润滑正常" OR "平衡缸气压检测" OR "压机急停故障2") AND NOT "总复位";
END_REGION

REGION Network 3
   RUNG wire#powerrail
      Contact( "寸动" )
      Contact( "液压保护选择开关0位" )
      I_Contact( "上死点" )
      I_Contact( "液压保护正常" )
      wire#w1
      Coil( "Tag_19" )
   END_RUNG
   RUNG wire#powerrail
      Contact( "液压保护正常" )
      Contact( "液压保护选择开关1位" )
   END_RUNG wire#w1
   // the same network as SCL:
   "Tag_19" := ("寸动" AND "液压保护选择开关0位" AND NOT "上死点" AND NOT "液压保护正常") OR ("液压保护正常" AND "液压保护选择开关1位");
END_REGION

REGION Network 4
   RUNG wire#powerrail
      Contact( "反转" )
      wire#w1
      Coil( "行程选择" )
   END_RUNG
   RUNG wire#powerrail
      Contact( "寸动" )
   END_RUNG wire#w1
   RUNG wire#powerrail
      Contact( "单次" )
   END_RUNG wire#w1
   RUNG wire#powerrail
      Contact( "连续" )
   END_RUNG wire#w1
   // the same network as SCL:
   "行程选择" := "反转" OR "寸动" OR "单次" OR "连续";
END_REGION

REGION Network 5
   RUNG wire#powerrail
      I_Contact( "急停故障(2)" )
      I_Contact( "压机急停故障2" )
      Coil( "安全正常(1)" )
   END_RUNG
   // the same network as SCL:
   "安全正常(1)" := NOT "急停故障(2)" AND NOT "压机急停故障2";
END_REGION

REGION Network 6
   RUNG wire#powerrail
      I_Contact( "压机急停故障2" )
      Coil( "压机急停1" )
   END_RUNG
   RUNG wire#powerrail
      I_Contact( "急停故障(2)" )
      Coil( "压机急停2" )
   END_RUNG
   // the same network as SCL:
   "压机急停1" := NOT "压机急停故障2";
   "压机急停2" := NOT "急停故障(2)";
END_REGION

REGION Network 7
   RUNG wire#powerrail
      I_Contact( "栅栏门未来关闭" )
      wire#w1
      Coil( "右栅栏落下检测" )
   END_RUNG
   RUNG wire#w1
      Coil( "左栅栏落下来检测" )
   END_RUNG
   // the same network as SCL:
   "右栅栏落下检测" := NOT "栅栏门未来关闭";
   "左栅栏落下来检测" := NOT "栅栏门未来关闭";
END_REGION

REGION Network 8
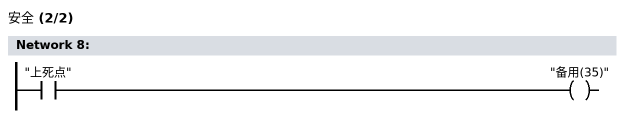
   RUNG wire#powerrail
      Contact( "上死点" )
      Coil( "备用(35)" )
   END_RUNG
   // the same network as SCL:
   "备用(35)" := "上死点";
END_REGION
END_FUNCTION

FUNCTION "气垫调整" : Void   // FC11, LAD
{ S7_Optimized_Access := 'TRUE' }
VERSION : 0.1
   VAR_TEMP   // added for the SCL form of the ladder/FBD networks
      _w1 : Bool;
   END_VAR
BEGIN

REGION Network 1
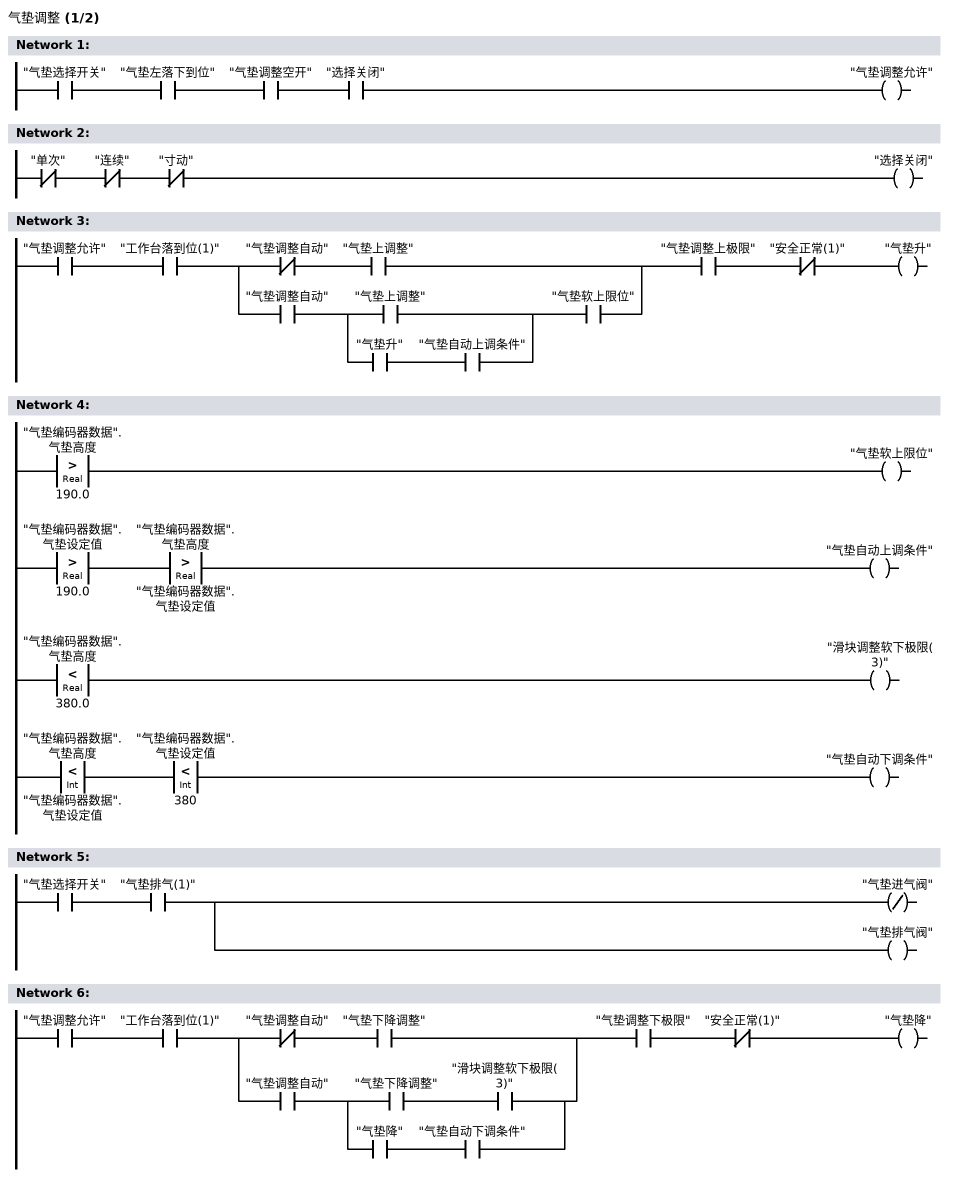
   RUNG wire#powerrail
      Contact( "气垫选择开关" )
      Contact( "气垫左落下到位" )
      Contact( "气垫调整空开" )
      Contact( "选择关闭" )
      Coil( "气垫调整允许" )
   END_RUNG
   // the same network as SCL:
   "气垫调整允许" := "气垫选择开关" AND "气垫左落下到位" AND "气垫调整空开" AND "选择关闭";
END_REGION

REGION Network 2
   RUNG wire#powerrail
      I_Contact( "单次" )
      I_Contact( "连续" )
      I_Contact( "寸动" )
      Coil( "选择关闭" )
   END_RUNG
   // the same network as SCL:
   "选择关闭" := NOT "单次" AND NOT "连续" AND NOT "寸动";
END_REGION

REGION Network 3
   RUNG wire#powerrail
      Contact( "气垫调整允许" )
      Contact( "工作台落到位(1)" )
      wire#w1
      I_Contact( "气垫调整自动" )
      Contact( "气垫上调整" )
      wire#w2
      Contact( "气垫调整上极限" )
      I_Contact( "安全正常(1)" )
      Coil( "气垫升" )
   END_RUNG
   RUNG wire#w1
      Contact( "气垫调整自动" )
      wire#w3
      Contact( "气垫上调整" )
      wire#w4
      Contact( "气垫软上限位" )
   END_RUNG wire#w2
   RUNG wire#w3
      Contact( "气垫升" )
      Contact( "气垫自动上调条件" )
   END_RUNG wire#w4
   // the same network as SCL:
   "气垫升" := "气垫调整允许" AND "工作台落到位(1)" AND ((NOT "气垫调整自动" AND "气垫上调整") OR ("气垫调整自动" AND ("气垫上调整" OR ("气垫升" AND "气垫自动上调条件")) AND "气垫软上限位")) AND "气垫调整上极限" AND NOT "安全正常(1)";
END_REGION

REGION Network 4
   RUNG wire#powerrail
      { S7_Templates := "SrcType := Real" } GT_Contact(in1 := "气垫编码器数据".气垫高度, in2 := 190.0)
      Coil( "气垫软上限位" )
   END_RUNG
   RUNG wire#powerrail
      { S7_Templates := "SrcType := Real" } GT_Contact(in1 := "气垫编码器数据".气垫设定值, in2 := 190.0)
      { S7_Templates := "SrcType := Real" } GT_Contact(in1 := "气垫编码器数据".气垫高度, in2 := "气垫编码器数据".气垫设定值)
      Coil( "气垫自动上调条件" )
   END_RUNG
   RUNG wire#powerrail
      { S7_Templates := "SrcType := Real" } LT_Contact(in1 := "气垫编码器数据".气垫高度, in2 := 380.0)
      Coil( "滑块调整软下极限(3)" )
   END_RUNG
   RUNG wire#powerrail
      { S7_Templates := "SrcType := Int" } LT_Contact(in1 := "气垫编码器数据".气垫高度, in2 := "气垫编码器数据".气垫设定值)
      { S7_Templates := "SrcType := Int" } LT_Contact(in1 := "气垫编码器数据".气垫设定值, in2 := 380)
      Coil( "气垫自动下调条件" )
   END_RUNG
   // the same network as SCL:
   "气垫软上限位" := "气垫编码器数据".气垫高度 > 190.0;
   "气垫自动上调条件" := ("气垫编码器数据".气垫设定值 > 190.0) AND ("气垫编码器数据".气垫高度 > "气垫编码器数据".气垫设定值);
   "滑块调整软下极限(3)" := "气垫编码器数据".气垫高度 < 380.0;
   "气垫自动下调条件" := ("气垫编码器数据".气垫高度 < "气垫编码器数据".气垫设定值) AND ("气垫编码器数据".气垫设定值 < 380);
END_REGION

REGION Network 5
   RUNG wire#powerrail
      Contact( "气垫选择开关" )
      Contact( "气垫排气(1)" )
      wire#w1
      I_Coil( "气垫进气阀" )
   END_RUNG
   RUNG wire#w1
      Coil( "气垫排气阀" )
   END_RUNG
   // the same network as SCL:
   #_w1 := "气垫选择开关" AND "气垫排气(1)";
   "气垫进气阀" := NOT #_w1;
   "气垫排气阀" := #_w1;
END_REGION

REGION Network 6
   RUNG wire#powerrail
      Contact( "气垫调整允许" )
      Contact( "工作台落到位(1)" )
      wire#w1
      I_Contact( "气垫调整自动" )
      Contact( "气垫下降调整" )
      wire#w2
      Contact( "气垫调整下极限" )
      I_Contact( "安全正常(1)" )
      Coil( "气垫降" )
   END_RUNG
   RUNG wire#w1
      Contact( "气垫调整自动" )
      wire#w3
      Contact( "气垫下降调整" )
      Contact( "滑块调整软下极限(3)" )
   END_RUNG wire#w2
   RUNG wire#w3
      Contact( "气垫降" )
      Contact( "气垫自动下调条件" )
   END_RUNG wire#w2
   // the same network as SCL:
   "气垫降" := "气垫调整允许" AND "工作台落到位(1)" AND ((NOT "气垫调整自动" AND "气垫下降调整") OR ("气垫调整自动" AND (("气垫下降调整" AND "滑块调整软下极限(3)") OR ("气垫降" AND "气垫自动下调条件")))) AND "气垫调整下极限" AND NOT "安全正常(1)";
END_REGION

REGION Network 7
   // 按位相与，清零前8bit状态位
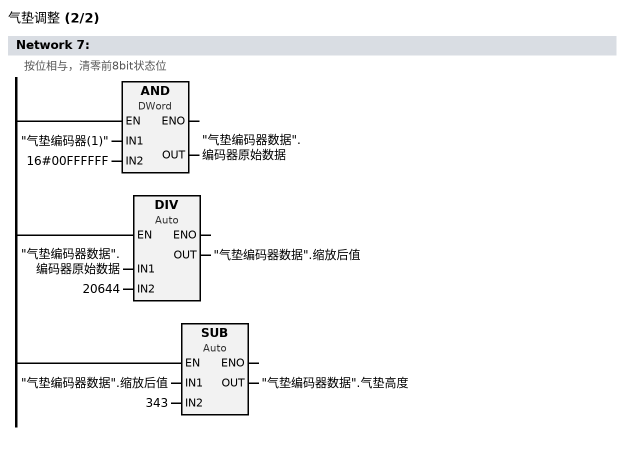
   RUNG wire#powerrail
      { S7_Templates := "SrcType := DWord" } And(in1 := "气垫编码器(1)", in2 := 16#00FFFFFF, out => "气垫编码器数据".编码器原始数据)
   END_RUNG
   RUNG wire#powerrail
      Div(in1 := "气垫编码器数据".编码器原始数据, in2 := 20644, out => "气垫编码器数据".缩放后值)
   END_RUNG
   RUNG wire#powerrail
      Sub(in1 := "气垫编码器数据".缩放后值, in2 := 343, out => "气垫编码器数据".气垫高度)
   END_RUNG
   // the same network as SCL:
   "气垫编码器数据".编码器原始数据 := "气垫编码器(1)" AND 16#00FFFFFF;
   "气垫编码器数据".缩放后值 := "气垫编码器数据".编码器原始数据 / 20644;
   "气垫编码器数据".气垫高度 := "气垫编码器数据".缩放后值 - 343;
END_REGION
END_FUNCTION

ORGANIZATION_BLOCK "IO测试"   // OB125, LAD, ProgramCycle
TITLE = "Main Program Sweep (Cycle)"
{ S7_Optimized_Access := 'TRUE' }
VERSION : 0.1
   VAR_INPUT
      Initial_Call : Bool;   // Initial call of this OB
      Remanence : Bool;   // =True, if remanent data are available
   END_VAR
BEGIN

REGION Network 1
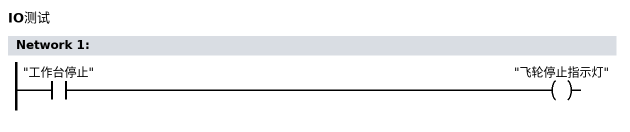
   RUNG wire#powerrail
      Contact( "工作台停止" )
      Coil( "飞轮停止指示灯" )
   END_RUNG
   // the same network as SCL:
   "飞轮停止指示灯" := "工作台停止";
END_REGION
END_ORGANIZATION_BLOCK

ORGANIZATION_BLOCK "Main"   // OB129, LAD, ProgramCycle
TITLE = "Main Program Sweep (Cycle)"
{ S7_Optimized_Access := 'TRUE' }
VERSION : 0.1
   VAR_INPUT
      Initial_Call : Bool;   // Initial call of this OB
      Remanence : Bool;   // =True, if remanent data are available
   END_VAR
BEGIN

REGION Network 1
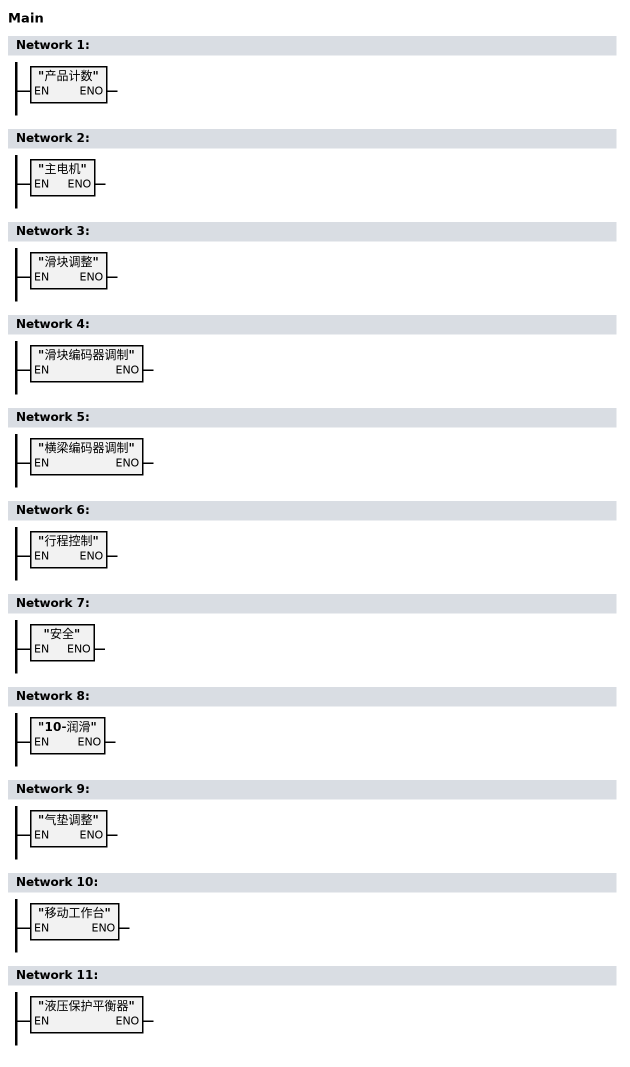
   RUNG wire#powerrail
      "产品计数"()
   END_RUNG
   // the same network as SCL:
   "产品计数"();
END_REGION

REGION Network 2
   RUNG wire#powerrail
      "主电机"()
   END_RUNG
   // the same network as SCL:
   "主电机"();
END_REGION

REGION Network 3
   RUNG wire#powerrail
      "滑块调整"()
   END_RUNG
   // the same network as SCL:
   "滑块调整"();
END_REGION

REGION Network 4
   RUNG wire#powerrail
      "滑块编码器调制"()
   END_RUNG
   // the same network as SCL:
   "滑块编码器调制"();
END_REGION

REGION Network 5
   RUNG wire#powerrail
      "横梁编码器调制"()
   END_RUNG
   // the same network as SCL:
   "横梁编码器调制"();
END_REGION

REGION Network 6
   RUNG wire#powerrail
      "行程控制"()
   END_RUNG
   // the same network as SCL:
   "行程控制"();
END_REGION

REGION Network 7
   RUNG wire#powerrail
      "安全"()
   END_RUNG
   // the same network as SCL:
   "安全"();
END_REGION

REGION Network 8
   RUNG wire#powerrail
      "10-润滑"()
   END_RUNG
   // the same network as SCL:
   "10-润滑"();
END_REGION

REGION Network 9
   RUNG wire#powerrail
      "气垫调整"()
   END_RUNG
   // the same network as SCL:
   "气垫调整"();
END_REGION

REGION Network 10
   RUNG wire#powerrail
      "移动工作台"()
   END_RUNG
   // the same network as SCL:
   "移动工作台"();
END_REGION

REGION Network 11
   RUNG wire#powerrail
      "液压保护平衡器"()
   END_RUNG
   // the same network as SCL:
   "液压保护平衡器"();
END_REGION
END_ORGANIZATION_BLOCK

(* ===== HMI "HMI_RT_1" =====
system functions are stored by id; their names below are inferred from use
connection "HMI_连接_1": ETHERNET, S7_1200_OMS

HMI tags "默认变量表"
   "360" : Bool = PLC 360 AT %M204.3, 100 ms
   "10度" : Bool = PLC 10度 AT %M200.0, 100 ms
   "20度" : Bool = PLC 20度 AT %M200.1, 100 ms
   "30度" : Bool = PLC 30度 AT %M200.2, 100 ms
   "40度" : Bool = PLC 40度 AT %M200.3, 100 ms
   "50" : Bool = PLC 50 AT %M200.4, 100 ms
   "60" : Bool = PLC 60 AT %M200.5, 100 ms
   "70" : Bool = PLC 70 AT %M200.6, 100 ms
   "80" : Bool = PLC 80 AT %M200.7, 100 ms
   "90" : Bool = PLC 90 AT %M201.0, 100 ms
   "100" : Bool = PLC 100 AT %M201.1, 100 ms
   "110" : Bool = PLC 110 AT %M201.2, 100 ms
   "120" : Bool = PLC 120 AT %M201.3, 100 ms
   "130" : Bool = PLC 130 AT %M201.4, 100 ms
   "140" : Bool = PLC 140 AT %M201.5, 100 ms
   "150" : Bool = PLC 150 AT %M201.6, 100 ms
   "160" : Bool = PLC 160 AT %M201.7, 100 ms
   "170" : Bool = PLC 170 AT %M202.0, 100 ms
   "180" : Bool = PLC 180 AT %M202.1, 100 ms
   "190" : Bool = PLC 190 AT %M202.2, 100 ms
   "200" : Bool = PLC 200 AT %M202.3, 100 ms
   "210" : Bool = PLC 210 AT %M202.4, 100 ms
   "220" : Bool = PLC 220 AT %M202.5, 100 ms
   "230" : Bool = PLC 230 AT %M202.6, 100 ms
   "240" : Bool = PLC 240 AT %M202.7, 100 ms
   "250" : Bool = PLC 250 AT %M203.0, 100 ms
   "260" : Bool = PLC 260 AT %M203.1, 100 ms
   "270" : Bool = PLC 270 AT %M203.2, 100 ms
   "280" : Bool = PLC 280 AT %M203.3, 100 ms
   "290" : Bool = PLC 290 AT %M203.4, 100 ms
   "300" : Bool = PLC 300 AT %M203.5, 100 ms
   "310" : Bool = PLC 310 AT %M203.6, 100 ms
   "320" : Bool = PLC 320 AT %M203.7, 100 ms
   "330" : Bool = PLC 330 AT %M204.0, 100 ms
   "340" : Bool = PLC 340 AT %M204.1, 100 ms
   "350" : Bool = PLC 350 AT %M204.2, 100 ms
   "工作台落到位前" : Bool = PLC "Tag_57(1)" AT %I7.3, 1 s
   "工作台落到位后" : Bool = PLC "Tag_58(1)" AT %I7.4, 1 s
   "工作台夹紧阀(1)" : Bool = PLC 左栅栏落下来检测 AT %Q13.1, 1 s
   "平衡缸气压检测" : Bool = PLC 平衡缸气压检测 AT %I10.5, 1 s
   "润滑油泵启动OK" : Bool = PLC 润滑油泵启动OK AT %M5.5, 1 s
   "润滑油压正常" : Bool = PLC 润滑油压正常 AT %M5.1, 1 s
   "液压保护故障" : Bool = PLC 液压保护故障 AT %M6.1, 1 s
   "横梁编码器" : DWord = PLC 横梁编码器 AT %ID68, 1 s
   "ECamdata _DB_+0.7" : DInt = PLC 滑块编码器 AT %ID72, 1 s
   "横梁编码器 _DB_+0.6" : Int = PLC "横梁编码器 _DB"."+0.6", 1 s
   "工作台放松阀(1)" : Bool = PLC "备用(16)" AT %Q13.2, 1 s
   "工作台落到位" : Bool = PLC 工作台落到位 AT %M7.1, 1 s
   "工作台-夹紧OK" : Bool = PLC "工作台-夹紧OK" AT %M15.2, 1 s
   "工作台放松OK" : Bool = PLC 工作台放松OK AT %M15.3, 1 s
   "横梁编码器 _DB_0.11" : Real = PLC "横梁编码器 _DB"."0.11", 1 s
   "滑块调整自动选择" : Bool = PLC 滑块调整自动选择 AT %M16.2, 1 s
   "ECamdata _DB_+0.36" : Int = PLC "ECamdata _DB"."+0.36", 100 ms
   "ECamdata _DB_+0.47" : Real = PLC "ECamdata _DB"."+0.47", 100 ms
   "ECamdata _DB_+0.6" : Int = PLC "ECamdata _DB".电子凸轮编码器显示, 100 ms
   "ECamdata _DB_AQD" : Real = PLC "ECamdata _DB".平衡器压力显示, 100 ms
   "ECamdata _DB_AQD2" : Real = PLC "ECamdata _DB".AQD2, 100 ms
   "ECamdata _DB_AQD3" : Real = PLC "ECamdata _DB".气垫模拟量显示1, 100 ms
   "ECamdata _DB_D{0}" : Real = PLC "ECamdata _DB".D[0], 100 ms
   "ECamdata _DB_D{1}" : Real = PLC "ECamdata _DB".D[1], 100 ms
   "ECamdata _DB_D{10}滑块设定高度" : Real = PLC "ECamdata _DB".D[10], 100 ms
   "ECamdata _DB_D{11}" : Real = PLC "ECamdata _DB".D[11], 100 ms
   "ECamdata _DB_D{6}" : Real = PLC "ECamdata _DB".D[6], 100 ms
   "ECamdata _DB_D{7}" : Real = PLC "ECamdata _DB".D[7], 100 ms
   "ECamdata _DB_D{9}" : Real = PLC "ECamdata _DB".D[9], 100 ms
   "ECamdata _DB_D102" : Int = PLC "ECamdata _DB".D102, 100 ms
   "ECamdata _DB_D107" : Int = PLC "ECamdata _DB".D107, 100 ms
   "ECamdata _DB_D108" : Real = PLC "ECamdata _DB".D108, 1 s
   "ECamdata _DB_当前产量" : Int = PLC "ECamdata _DB".当前产量, 1 s
   "ECamdata _DB_滑块打油次数" : Int = PLC "ECamdata _DB".滑块打油次数, 100 ms
   "ECamdata _DB_平衡器设置压力" : Real = PLC "ECamdata _DB".平衡器设置压力, 100 ms
   "ECamdata _DB_气垫2压力设置" : Real = PLC "ECamdata _DB".气垫2压力设置, 100 ms
   "ECamdata _DB_气垫模拟量显示1" : Real = PLC "ECamdata _DB".气垫模拟量显示2, 100 ms
   "ECamdata _DB_气垫压力设置" : Real = PLC "ECamdata _DB".气垫1压力设置, 100 ms
   "ECamdata _DB_设置产量" : Int = PLC "ECamdata _DB".设置产量, 1 s
   "ECamdata _DB_主分油器打油次数" : Int = PLC "ECamdata _DB".主分油器打油次数, 100 ms
   "滑块调整手动/自动" : Bool = PLC "滑块调整手动/自动" AT %M301.5, 100 ms
   "ECamdata _DB_D{10}滑块设定高度(1)" : Real = PLC "ECamdata _DB_D{10}滑块设定高度" AT %MD150, 1 s
   "横梁编码器 _DB_+0.8" : Int = PLC "横梁编码器 _DB"."+0.8", 1 s
   "PLC报警变量组1" : Int = PLC PLC报警变量组1 AT %MW3000, 1 s
   "PLC报警变量组2" : Int = PLC PLC报警变量组2 AT %MW3002, 1 s
   "上极限" : Bool = PLC 上极限 AT %I13.4, 1 s
   "工作台顶起" : Bool = PLC 工作台顶起 AT %Q11.4, 1 s
   "液压保护正常" : Bool = PLC 液压保护正常 AT %M207.6, 1 s
   "润滑正常" : Bool = PLC 润滑正常 AT %M1000.4, 1 s
   "滑块调整电机空开" : Bool = PLC 滑块调整电机空开 AT %I2.1, 1 s
   "滑块调整选择开关" : Bool = PLC 滑块调整选择开关 AT %I10.0, 1 s
   "上死点" : Bool = PLC 上死点 AT %M204.4, 100 ms
   "滑块调整上极限" : Bool = PLC 滑块调整上极限 AT %I10.3, 1 s
   "滑块调整下极限" : Bool = PLC 滑块调整下极限 AT %I10.4, 1 s
   "滑块调整向上" : Bool = PLC 滑块调整向上 AT %I10.1, 1 s
   "滑块调整向下" : Bool = PLC 滑块调整向下 AT %I10.2, 1 s
   "急停故障(2)" : Bool = PLC "急停故障(2)" AT %M300.0, 1 s
   "行程选择" : Bool = PLC 行程选择 AT %M207.3, 1 s
   "左后双手使用" : Bool = PLC 左后双手使用 AT %I4.4, 1 s
   "右前双手选择" : Bool = PLC 右前双手选择 AT %I25.2, 1 s
   "工作台放松顶起" : Bool = PLC 工作台放松顶起 AT %I14.4, 1 s
   "调整开关" : Bool = PLC 调整开关 AT %I14.5, 1 s
   "工作台顶起压力" : Bool = PLC 工作台顶起压力 AT %I15.3, 1 s
   "工作台顶起右前检测" : Bool = PLC 工作台顶起右前检测 AT %I17.3, 1 s
   "工作台顶起左后检测" : Bool = PLC 工作台顶起左后检测 AT %I17.4, 1 s
   "工作台落下右边后检测" : Bool = PLC 工作台落下右边后检测 AT %I18.1, 1 s
   "工作台落下右前检测" : Bool = PLC 工作台落下右前检测 AT %I17.7, 1 s
   "工作台落下左前检测" : Bool = PLC 工作台落下左前检测 AT %I17.6, 1 s
   "工作台落下左后检测" : Bool = PLC 工作台落下左后检测 AT %I18.0, 1 s
   "开工作台变频器正常" : Bool = PLC 开工作台变频器正常 AT %I2.6, 1 s
   "工作台开进" : Bool = PLC 工作台开进 AT %I15.0, 1 s
   "工作台开进到位" : Bool = PLC 工作台开进到位 AT %I16.2, 1 s
   "工作台开出" : Bool = PLC 工作台开出 AT %I14.7, 1 s
   "工作台左前顶起到位" : Bool = PLC 工作台左前顶起到位 AT %I15.6, 1 s
   "工作台右前顶起到位" : Bool = PLC 工作台右前顶起到位 AT %I15.7, 1 s
   "工作台左后顶起到位" : Bool = PLC 工作台左后顶起到位 AT %I16.0, 1 s
   "工作台右后顶起到位" : Bool = PLC 工作台右后顶起到位 AT %I16.1, 1 s
   "工作台落下夹紧(1)" : Bool = PLC "工作台落下夹紧(1)" AT %I14.3, 1 s
   "工作台放松顶起(1)" : Bool = PLC "工作台放松顶起(1)" AT %Q11.1, 1 s
   "工作台落下夹紧(2)" : Bool = PLC "工作台落下夹紧(2)" AT %Q11.3, 1 s
   "润滑电机工作指示" : Bool = PLC 润滑电机工作指示 AT %Q12.4, 1 s
   "正转条件" : Bool = PLC 正转条件 AT %M1000.7, 1 s
   "主电机启动指示" : Bool = PLC 主电机启动指示 AT %Q12.0, 1 s
   "主电机启动延时" : Bool = PLC 主电机启动延时 AT %M1100.4, 1 s
   "IEC_Counter_0_DB_4_CV" : Int = PLC 当前产量.CV, 1 s
   "产量到达" : Bool = PLC 产量到达 AT %M30.2, 1 s
   "计数开始" : Bool = PLC 计数开始 AT %M30.0, 1 s
   "计数清零" : Bool = PLC 计数清零 AT %M30.1, 1 s
   "主电机正转运行" : Bool = PLC 主电机正转运行 AT %Q2.0, 1 s
   "横梁1分油器检测" : Bool = PLC 横梁1分油器检测 AT %I5.1, 100 ms
   "平衡器分油器检测" : Bool = PLC 平衡器分油器检测 AT %I5.0, 1 s
   "润滑故障" : Bool = PLC 润滑故障 AT %M15.4, 1 s
   "主电机零速" : Bool = PLC 主电机零速 AT %I2.5, 1 s
   "主电机温度检测(1)" : Bool = PLC "主电机温度检测(1)" AT %I4.1, 1 s
   "主电机调速装置正常" : Bool = PLC 主电机调速装置正常 AT %I2.4, 1 s
   "主电机风扇空开" : Bool = PLC 主电机风扇空开 AT %I2.3, 1 s
   "主电机风扇流量检测(1)" : Bool = PLC "主电机风扇流量检测(1)" AT %I4.0, 1 s
   "按钮站插入" : Bool = PLC 按钮站插入 AT %I15.5, 1 s
   "右前急停按钮" : Bool = PLC 右前急停按钮 AT %I22.4, 1 s
   "左前急停按钮" : Bool = PLC 左前急停按钮 AT %I22.5, 1 s
   "右后急停按钮" : Bool = PLC 右后急停按钮 AT %I22.6, 1 s
   "左后急停按钮" : Bool = PLC 左后急停按钮 AT %I22.7, 1 s
   "前安全栓" : Bool = PLC 前安全栓 AT %I23.1, 1 s
   "后安全栓" : Bool = PLC 后安全栓 AT %I23.0, 1 s
   "气垫调整空开" : Bool = PLC 气垫调整空开 AT %I2.2, 1 s
   "气垫调整上极限" : Bool = PLC 气垫调整上极限 AT %I11.2, 1 s
   "气垫调整下极限" : Bool = PLC 气垫调整下极限 AT %I11.3, 1 s
   "气垫冷却电机过热" : Bool = PLC 气垫冷却电机过热 AT %I13.1, 1 s
   "气垫左落下到位" : Bool = PLC 气垫左落下到位 AT %I11.6, 1 s
   "气垫压力检测" : Bool = PLC 气垫压力检测 AT %I12.1, 1 s
   "工作台顶起左前检测" : Bool = PLC 工作台顶起左前检测 AT %I17.2, 1 s
   "工作台顶起右后检测" : Bool = PLC 工作台顶起右后检测 AT %I17.5, 1 s
   "工作台左前落到为" : Bool = PLC 工作台左前落到为 AT %I16.3, 1 s
   "工作台右前落到为" : Bool = PLC 工作台右前落到为 AT %I16.4, 1 s
   "工作台左后落到为" : Bool = PLC 工作台左后落到为 AT %I16.5, 1 s
   "工作台右后落到位" : Bool = PLC 工作台右后落到位 AT %I16.6, 1 s
   "润滑电机空开" : Bool = PLC 润滑电机空开 AT %I3.0, 1 s
   "润滑油位检测" : Bool = PLC 润滑油位检测 AT %I21.1, 1 s
   "润滑过滤检测" : Bool = PLC 润滑过滤检测 AT %I21.2, 1 s
   "滑块分油器检测" : Bool = PLC 滑块分油器检测 AT %I22.1, 100 ms
   "气垫分油器检测" : Bool = PLC 气垫分油器检测 AT %I22.2, 100 ms
   "液压保护系统空开" : Bool = PLC 液压保护系统空开 AT %I2.7, 1 s
   "50/AR液压保护压力" : Bool = PLC 100液压保护压力 AT %I18.6, 1 s
   "90/AR液压保护压力" : Bool = PLC "90/AR液压保护压力" AT %I18.7, 1 s
   "100/AR液压保护压力" : Bool = PLC "100/AR液压保护压力" AT %I18.4, 1 s
   "135/AR液压保护压力" : Bool = PLC "135/AR液压保护压力" AT %I18.5, 1 s
   "150/AR液压保护压力" : Bool = PLC "150/AR液压保护压力" AT %I19.0, 1 s
   "离制压力检测" : Bool = PLC 离制压力检测 AT %I24.0, 1 s
   "离制油箱油位检测" : Bool = PLC 离制油箱油位检测 AT %I24.2, 1 s
   "离制油箱油温检测" : Bool = PLC 离制油箱油温检测 AT %I24.6, 1 s
   "离制过滤器检测" : Bool = PLC 离制过滤器检测 AT %I23.7, 1 s
   "离制双阀反馈1" : Bool = PLC 离制双阀反馈1 AT %I3.4, 1 s
   "离制双阀反馈2" : Bool = PLC 离制双阀反馈2 AT %I3.5, 1 s
   "离合器油泵空开" : Bool = PLC 离合器油泵空开 AT %I3.6, 1 s
   "离合器运行" : Bool = PLC 离合器运行 AT %I3.7, 1 s
   "离合器准确检测" : Bool = PLC 离合器准确检测 AT %I5.2, 1 s
   "离合冷却过滤器检测" : Bool = PLC 离合冷却过滤器检测 AT %I24.3, 1 s
   "平衡缸进气阀" : Bool = PLC 平衡缸进气阀 AT %Q10.0, 1 s
   "平衡缸排气阀" : Bool = PLC 平衡缸排气阀 AT %Q10.1, 1 s
   "左气垫进气阀" : Bool = PLC 气垫进气阀 AT %Q10.2, 1 s
   "左气垫排气阀" : Bool = PLC 气垫排气阀 AT %Q10.3, 1 s
   "右气垫进气阀" : Bool = PLC 右气垫进气阀 AT %Q10.4, 1 s
   "右气垫气排阀" : Bool = PLC 右气垫气排阀 AT %Q10.5, 1 s
   "气动泵气源阀-1#" : Bool = PLC "气动泵气源阀-1#" AT %Q10.6, 1 s
   "液压保护泵启动（卸载）阀-2#" : Bool = PLC "液压保护泵启动（卸载）阀-2#" AT %Q10.7, 1 s
   "液压保护负荷荷 阀-3#" : Bool = PLC "液压保护负荷荷 阀-3#" AT %Q11.0, 1 s
   "平衡器间歇润滑阀" : Bool = PLC 平衡器间歇润滑阀 AT %Q0.2, 1 s
   "气垫间歇润滑阀" : Bool = PLC 气垫间歇润滑阀 AT %Q11.6, 1 s
   "自动化气压" : Bool = PLC 自动化气压 AT %Q11.7, 1 s
   "飞轮停止指示灯" : Bool = PLC 飞轮停止指示灯 AT %Q12.1, 1 s
   "模具移出指示" : Bool = PLC 模具移出指示 AT %Q12.2, 1 s
   "模具装入指示" : Bool = PLC 模具装入指示 AT %Q12.3, 1 s
   "液压保护正常指示" : Bool = PLC 液压保护正常指示 AT %Q12.5, 1 s
   "液压保护卸荷指示" : Bool = PLC 液压保护卸荷指示 AT %Q12.6, 1 s
   "气垫升" : Bool = PLC 气垫升 AT %Q0.5, 1 s
   "气垫降" : Bool = PLC 气垫降 AT %Q0.6, 1 s
   "飞轮制动阀" : Bool = PLC 飞轮制动阀 AT %Q0.3, 1 s
   "单人操作" : Bool = PLC 单人操作 AT %Q0.4, 1 s
   "气垫升(1)" : Bool = PLC "气垫升(1)" AT %Q0.0, 1 s
   "气垫降(1)" : Bool = PLC "气垫降(1)" AT %Q0.1, 1 s
   "速度控制" : Bool = PLC 速度控制 AT %Q1.0, 1 s
   "主电机反转" : Bool = PLC 主电机反转 AT %Q1.1, 1 s
   "系统泵开始" : Bool = PLC 系统泵开始 AT %Q2.1, 1 s
   "变频器使能" : Bool = PLC 变频器使能 AT %Q2.2, 1 s
   "润滑电机" : Bool = PLC 润滑电机 AT %Q2.6, 1 s
   "工作台电机正转(1)" : Bool = PLC "工作台电机正转(1)" AT %Q2.3, 1 s
   "工作骀电机反转" : Bool = PLC 工作骀电机反转 AT %Q2.4, 1 s
   "工作台变速" : Bool = PLC 工作台变速 AT %Q2.5, 1 s
   "安全正常(1)" : Bool = PLC "安全正常(1)" AT %Q2.7, 1 s
   "压机急停1" : Bool = PLC 压机急停1 AT %Q3.0, 1 s
   "压机急停2" : Bool = PLC 压机急停2 AT %Q3.1, 1 s
   "离合器油泵电机" : Bool = PLC 离合器油泵电机 AT %Q3.2, 1 s
   "单次连续继电器" : Bool = PLC 单次连续继电器 AT %Q3.3, 1 s
   "滑块向上调整" : Bool = PLC 滑块向上调整 AT %Q3.4, 1 s
   "滑块向下调整" : Bool = PLC 滑块向下调整 AT %Q3.5, 1 s
   "主电机风扇运行" : Bool = PLC 主电机风扇运行 AT %Q3.6, 1 s
   "急停故障" : Bool = PLC 急停故障 AT %M6.0, 1 s
   "下死点" : Bool = PLC 下死点 AT %M204.6, 100 ms
   "润滑异常" : Bool = PLC 润滑异常 AT %M1000.6, 1 s
   "离制压力正常" : Bool = PLC 离制压力正常 AT %M3501.0, 1 s
   "气垫编码器数据_气垫高度" : Int = PLC 气垫编码器数据.气垫高度, 100 ms
   "气垫编码器数据_气垫设定值" : Int = PLC 气垫编码器数据.气垫设定值, 100 ms
   "气垫选择开关" : Bool = PLC 气垫选择开关 AT %I10.7, 1 s
   "选择关闭" : Bool = PLC 选择关闭 AT %M330.0, 1 s
   "气垫调整自动" : Bool = PLC 气垫调整自动 AT %M330.3, 1 s
   "气垫上调整" : Bool = PLC 气垫上调整 AT %I17.1, 1 s
   "气垫下降调整" : Bool = PLC 气垫下降调整 AT %I19.2, 1 s
   "液压保护故障(1)" : Bool = PLC "液压保护故障(1)" AT %M208.0, 1 s

HMI tags "辅助中继"
   "辅助中继.横梁润滑故障" : Bool = PLC 辅助中继.横梁润滑故障, 1 s
   "辅助中继.滑块润滑故障" : Bool = PLC 辅助中继.滑块润滑故障 AT %DB1.DBX0.0, 1 s
   "辅助中继.气垫润滑故障" : Bool = PLC 辅助中继.气垫润滑故障 AT %DB1.DBX0.0, 1 s
   "辅助中继.平衡器润滑故障" : Bool = PLC 辅助中继.平衡器润滑故障 AT %DB1.DBX0.0, 1 s
   "辅助中继.润滑空开异常" : Bool = PLC 辅助中继.润滑空开异常 AT %DB1.DBX0.0, 1 s
   "辅助中继.润滑过滤异常" : Bool = PLC 辅助中继.润滑过滤异常 AT %DB1.DBX0.0, 1 s

HMI tags "中间数据"
   "中间数据.横梁润滑检测时长" : Time = PLC 中间数据.横梁润滑检测时长, 1 s
   "中间数据.滑块润滑检测时长" : Time = PLC 中间数据.滑块润滑检测时长 AT %DB1.DBD0, 1 s
   "中间数据.平衡器润滑检测时长" : Time = PLC 中间数据.平衡器润滑检测时长 AT %DB1.DBD0, 1 s
   "中间数据.横梁打油目标次数" : Int = PLC 中间数据.横梁打油目标次数 AT %DB1.DBD0, 1 s
   "中间数据.滑块打油目标次数" : Int = PLC 中间数据.滑块打油目标次数 AT %DB1.DBW0, 1 s
   "中间数据.平衡器打油目标次数" : Int = PLC 中间数据.平衡器打油目标次数 AT %DB1.DBW0, 1 s
   "中间数据.当前打油次数-横梁" : Int = PLC 中间数据.当前打油次数-横梁 AT %DB1.DBW0, 1 s
   "中间数据.当前打油次数-滑块" : Int = PLC 中间数据.当前打油次数-滑块 AT %DB1.DBW0, 1 s
   "中间数据.当前打油次数-平衡器" : Int = PLC 中间数据.当前打油次数-平衡器 AT %DB1.DBW0, 1 s
   "横梁检测当前时间" : Time = PLC "Timer".横梁润滑检测计时.ET AT %DB1.DBW0, 1 s
   "滑块检测当前时间" : Time = PLC "Timer".滑块润滑检测计时.ET AT %DB1.DBW0, 1 s
   "平衡器检测当前时间" : Time = PLC "Timer".平衡器润滑检测计时.ET AT %DB1.DBW0, 1 s

discrete alarms
   1: '急停', class Errors, trigger "PLC报警变量组1" bit 0
   2: '润滑压力异常', class Errors, trigger "PLC报警变量组1" bit 1
   3: '"离合器压力异常', class Errors, trigger "PLC报警变量组1" bit 2
   4: '"平衡器压力异常"', class Errors, trigger "PLC报警变量组1" bit 3
   5: '"液压保护过载"', class Errors, trigger "PLC报警变量组1" bit 4
   6: '"低液位"', class Errors, trigger "PLC报警变量组1" bit 5
   7: '"滑块调整上限位断开"', class Errors, trigger "PLC报警变量组1" bit 6
   8: '"滑块调整下限位断开"', class Errors, trigger "PLC报警变量组1" bit 7
   9: '"双阀粘连1-K3"', class Errors, trigger "PLC报警变量组1" bit 8
   10: '"双阀粘连1-K4"', class Errors, trigger "PLC报警变量组1" bit 9
   11: '"双阀继电器粘连1"', class Errors, trigger "PLC报警变量组1" bit 10
   12: '"双阀继电器粘连2"', class Errors, trigger "PLC报警变量组1" bit 11
   13: '"润滑电机过载"', class Errors, trigger "PLC报警变量组1" bit 12
   14: '"工作台油泵电机过载"', class Errors, trigger "PLC报警变量组1" bit 13
   15: '"主电机过载"', class Errors, trigger "PLC报警变量组1" bit 14
   16: '"润滑异常"', class Errors, trigger "PLC报警变量组1" bit 15
   17: '工作台未夹紧', class Errors, trigger "PLC报警变量组2" bit 0
   18: '"工作台未眠放松"', class Errors, trigger "PLC报警变量组2" bit 1
   19: '"液压保护压力未正常"', class Errors, trigger "PLC报警变量组2" bit 2
   20: '"滑块调整电机过载"', class Errors, trigger "PLC报警变量组2" bit 3
   21: '"超载指示"', class Errors, trigger "PLC报警变量组2" bit 4
   22: '"气压未正常"', class Errors, trigger "PLC报警变量组2" bit 5
   23: '"急停中', class Errors, trigger "PLC报警变量组2" bit 6
   24: '异常报警', class Errors, trigger "PLC报警变量组2" bit 7
   25: '右前工作台未落下到位', class Errors, trigger "PLC报警变量组2" bit 8
   26: '左后工作台未落下到位', class Errors, trigger "PLC报警变量组2" bit 9
   27: '"右前工作台未顶起到位"', class Errors, trigger "PLC报警变量组2" bit 10
   28: '"左前工作台未顶起到位"', class Errors, trigger "PLC报警变量组2" bit 11
   29: '"工作台未开进到位"', class Errors, trigger "PLC报警变量组2" bit 12
   30: '左气垫未落下到位', class Errors, trigger "PLC报警变量组2" bit 13
   31: '中气垫未落下到位', class Errors, trigger "PLC报警变量组2" bit 14
   32: '右气垫未落下到位', class Errors, trigger "PLC报警变量组2" bit 15

graphic list "@DiagnosticsStates": 0 '@Diagnostics_StateGood'; 1 '@Diagnostics_StateBad'

